REGION Network 8: START CYCLE LAMP
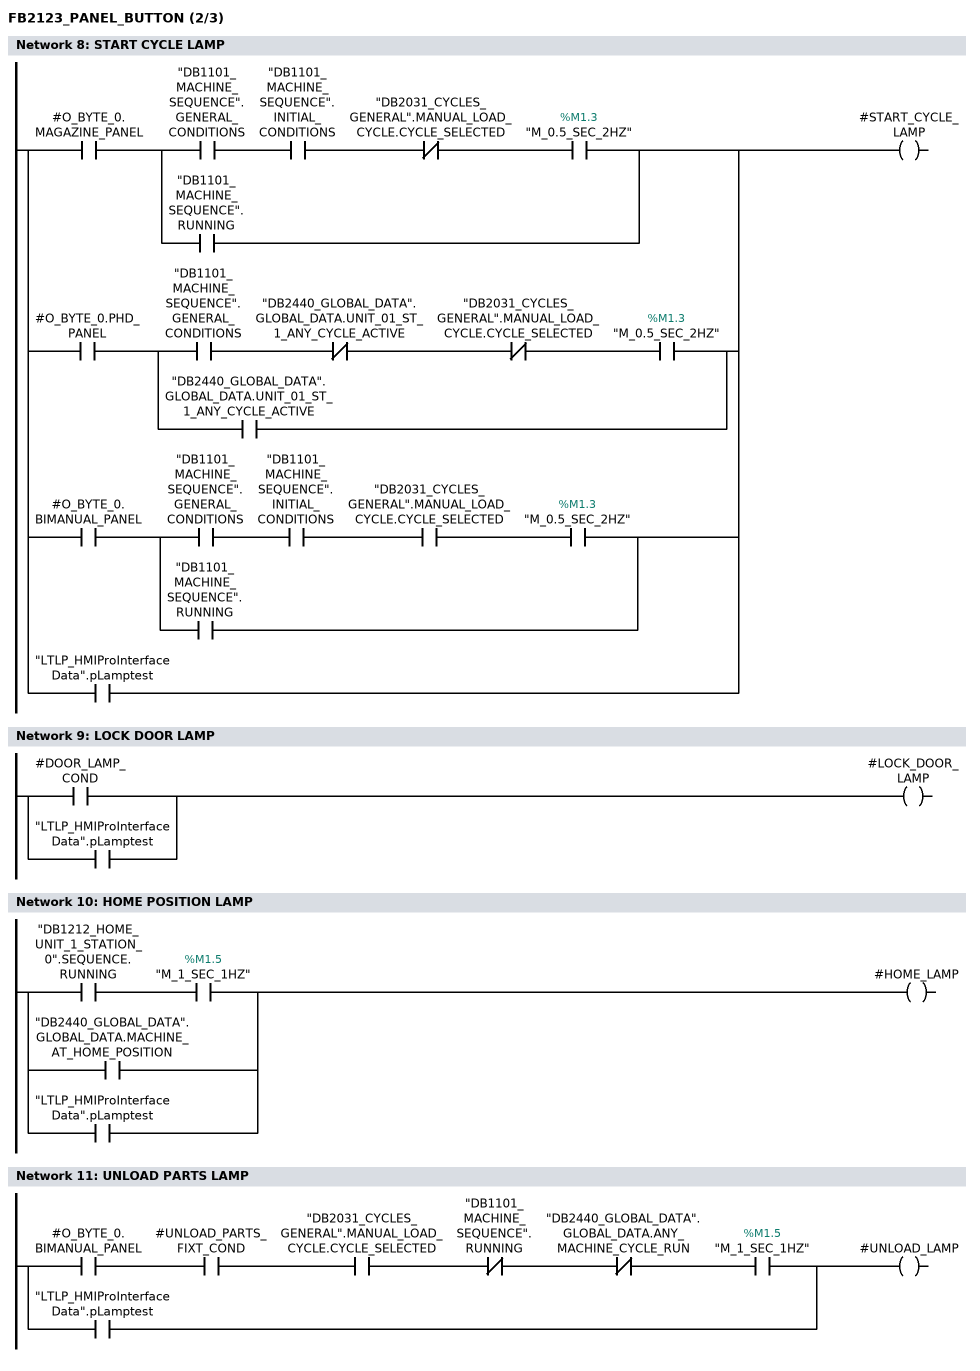
   RUNG wire#powerrail
      Contact( #O_BYTE_0.MAGAZINE_PANEL )
      wire#w1
      Contact( "DB1101_MACHINE_SEQUENCE".GENERAL_CONDITIONS )
      Contact( "DB1101_MACHINE_SEQUENCE".INITIAL_CONDITIONS )
      I_Contact( "DB2031_CYCLES_GENERAL".MANUAL_LOAD_CYCLE.CYCLE_SELECTED )
      Contact( "M_0.5_SEC_2HZ" )
      wire#w2
      Coil( #START_CYCLE_LAMP )
   END_RUNG
   RUNG wire#w1
      Contact( "DB1101_MACHINE_SEQUENCE".RUNNING )
   END_RUNG wire#w2
   RUNG wire#powerrail
      Contact( #O_BYTE_0.PHD_PANEL )
      wire#w3
      Contact( "DB1101_MACHINE_SEQUENCE".GENERAL_CONDITIONS )
      I_Contact( "DB2440_GLOBAL_DATA".GLOBAL_DATA.UNIT_01_ST_1_ANY_CYCLE_ACTIVE )
      I_Contact( "DB2031_CYCLES_GENERAL".MANUAL_LOAD_CYCLE.CYCLE_SELECTED )
      Contact( "M_0.5_SEC_2HZ" )
   END_RUNG wire#w2
   RUNG wire#w3
      Contact( "DB2440_GLOBAL_DATA".GLOBAL_DATA.UNIT_01_ST_1_ANY_CYCLE_ACTIVE )
   END_RUNG wire#w2
   RUNG wire#powerrail
      Contact( #O_BYTE_0.BIMANUAL_PANEL )
      wire#w4
      Contact( "DB1101_MACHINE_SEQUENCE".GENERAL_CONDITIONS )
      Contact( "DB1101_MACHINE_SEQUENCE".INITIAL_CONDITIONS )
      Contact( "DB2031_CYCLES_GENERAL".MANUAL_LOAD_CYCLE.CYCLE_SELECTED )
      Contact( "M_0.5_SEC_2HZ" )
   END_RUNG wire#w2
   RUNG wire#w4
      Contact( "DB1101_MACHINE_SEQUENCE".RUNNING )
   END_RUNG wire#w2
   RUNG wire#powerrail
      Contact( "LTLP_HMIProInterfaceData".pLamptest )
   END_RUNG wire#w2
   // the same network as SCL:
   #START_CYCLE_LAMP := (#O_BYTE_0.MAGAZINE_PANEL AND (("DB1101_MACHINE_SEQUENCE".GENERAL_CONDITIONS AND "DB1101_MACHINE_SEQUENCE".INITIAL_CONDITIONS AND NOT "DB2031_CYCLES_GENERAL".MANUAL_LOAD_CYCLE.CYCLE_SELECTED AND "M_0.5_SEC_2HZ") OR "DB1101_MACHINE_SEQUENCE".RUNNING)) OR (#O_BYTE_0.PHD_PANEL AND (("DB1101_MACHINE_SEQUENCE".GENERAL_CONDITIONS AND NOT "DB2440_GLOBAL_DATA".GLOBAL_DATA.UNIT_01_ST_1_ANY_CYCLE_ACTIVE AND NOT "DB2031_CYCLES_GENERAL".MANUAL_LOAD_CYCLE.CYCLE_SELECTED AND "M_0.5_SEC_2HZ") OR "DB2440_GLOBAL_DATA".GLOBAL_DATA.UNIT_01_ST_1_ANY_CYCLE_ACTIVE)) OR (#O_BYTE_0.BIMANUAL_PANEL AND (("DB1101_MACHINE_SEQUENCE".GENERAL_CONDITIONS AND "DB1101_MACHINE_SEQUENCE".INITIAL_CONDITIONS AND "DB2031_CYCLES_GENERAL".MANUAL_LOAD_CYCLE.CYCLE_SELECTED AND "M_0.5_SEC_2HZ") OR "DB1101_MACHINE_SEQUENCE".RUNNING)) OR "LTLP_HMIProInterfaceData".pLamptest;
END_REGION

REGION Network 9: LOCK DOOR LAMP
   RUNG wire#powerrail
      Contact( #DOOR_LAMP_COND )
      wire#w1
      Coil( #LOCK_DOOR_LAMP )
   END_RUNG
   RUNG wire#powerrail
      Contact( "LTLP_HMIProInterfaceData".pLamptest )
   END_RUNG wire#w1
   // the same network as SCL:
   #LOCK_DOOR_LAMP := #DOOR_LAMP_COND OR "LTLP_HMIProInterfaceData".pLamptest;
END_REGION

REGION Network 10: HOME POSITION LAMP
   RUNG wire#powerrail
      Contact( "DB1212_HOME_UNIT_1_STATION_0".SEQUENCE.RUNNING )
      Contact( "M_1_SEC_1HZ" )
      wire#w1
      Coil( #HOME_LAMP )
   END_RUNG
   RUNG wire#powerrail
      Contact( "DB2440_GLOBAL_DATA".GLOBAL_DATA.MACHINE_AT_HOME_POSITION )
   END_RUNG wire#w1
   RUNG wire#powerrail
      Contact( "LTLP_HMIProInterfaceData".pLamptest )
   END_RUNG wire#w1
   // the same network as SCL:
   #HOME_LAMP := ("DB1212_HOME_UNIT_1_STATION_0".SEQUENCE.RUNNING AND "M_1_SEC_1HZ") OR "DB2440_GLOBAL_DATA".GLOBAL_DATA.MACHINE_AT_HOME_POSITION OR "LTLP_HMIProInterfaceData".pLamptest;
END_REGION

REGION Network 11: UNLOAD PARTS LAMP
   RUNG wire#powerrail
      Contact( #O_BYTE_0.BIMANUAL_PANEL )
      Contact( #UNLOAD_PARTS_FIXT_COND )
      Contact( "DB2031_CYCLES_GENERAL".MANUAL_LOAD_CYCLE.CYCLE_SELECTED )
      I_Contact( "DB1101_MACHINE_SEQUENCE".RUNNING )
      I_Contact( "DB2440_GLOBAL_DATA".GLOBAL_DATA.ANY_MACHINE_CYCLE_RUN )
      Contact( "M_1_SEC_1HZ" )
      wire#w1
      Coil( #UNLOAD_LAMP )
   END_RUNG
   RUNG wire#powerrail
      Contact( "LTLP_HMIProInterfaceData".pLamptest )
   END_RUNG wire#w1
   // the same network as SCL:
   #UNLOAD_LAMP := (#O_BYTE_0.BIMANUAL_PANEL AND #UNLOAD_PARTS_FIXT_COND AND "DB2031_CYCLES_GENERAL".MANUAL_LOAD_CYCLE.CYCLE_SELECTED AND NOT "DB1101_MACHINE_SEQUENCE".RUNNING AND NOT "DB2440_GLOBAL_DATA".GLOBAL_DATA.ANY_MACHINE_CYCLE_RUN AND "M_1_SEC_1HZ") OR "LTLP_HMIProInterfaceData".pLamptest;
END_REGION

REGION Network 12: LOAD PARTS LAMP
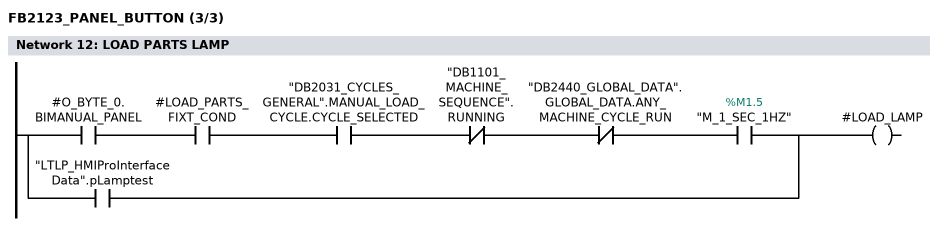
   RUNG wire#powerrail
      Contact( #O_BYTE_0.BIMANUAL_PANEL )
      Contact( #LOAD_PARTS_FIXT_COND )
      Contact( "DB2031_CYCLES_GENERAL".MANUAL_LOAD_CYCLE.CYCLE_SELECTED )
      I_Contact( "DB1101_MACHINE_SEQUENCE".RUNNING )
      I_Contact( "DB2440_GLOBAL_DATA".GLOBAL_DATA.ANY_MACHINE_CYCLE_RUN )
      Contact( "M_1_SEC_1HZ" )
      wire#w1
      Coil( #LOAD_LAMP )
   END_RUNG
   RUNG wire#powerrail
      Contact( "LTLP_HMIProInterfaceData".pLamptest )
   END_RUNG wire#w1
   // the same network as SCL:
   #LOAD_LAMP := (#O_BYTE_0.BIMANUAL_PANEL AND #LOAD_PARTS_FIXT_COND AND "DB2031_CYCLES_GENERAL".MANUAL_LOAD_CYCLE.CYCLE_SELECTED AND NOT "DB1101_MACHINE_SEQUENCE".RUNNING AND NOT "DB2440_GLOBAL_DATA".GLOBAL_DATA.ANY_MACHINE_CYCLE_RUN AND "M_1_SEC_1HZ") OR "LTLP_HMIProInterfaceData".pLamptest;
END_REGION
END_FUNCTION_BLOCK

FUNCTION "FC2101_LINE_CONTACTOR" : Void   // FC2101, LAD
{ S7_Optimized_Access := 'FALSE' }
AUTHOR : ETXETAR
VERSION : 1.0
// stored: AutoNumber false, IsIECCheckEnabled false, SetENOAutomatically false, UDAEnableTagReadback false
   VAR CONSTANT
      FC_NUMBER : DInt := 2101;   // FC NUMBER
   END_VAR
   VAR_TEMP   // added for the SCL form of the ladder/FBD networks
      _w1 : Bool;
      _w2 : Bool;
   END_VAR
BEGIN

REGION Network 1: OPTIONS OFF
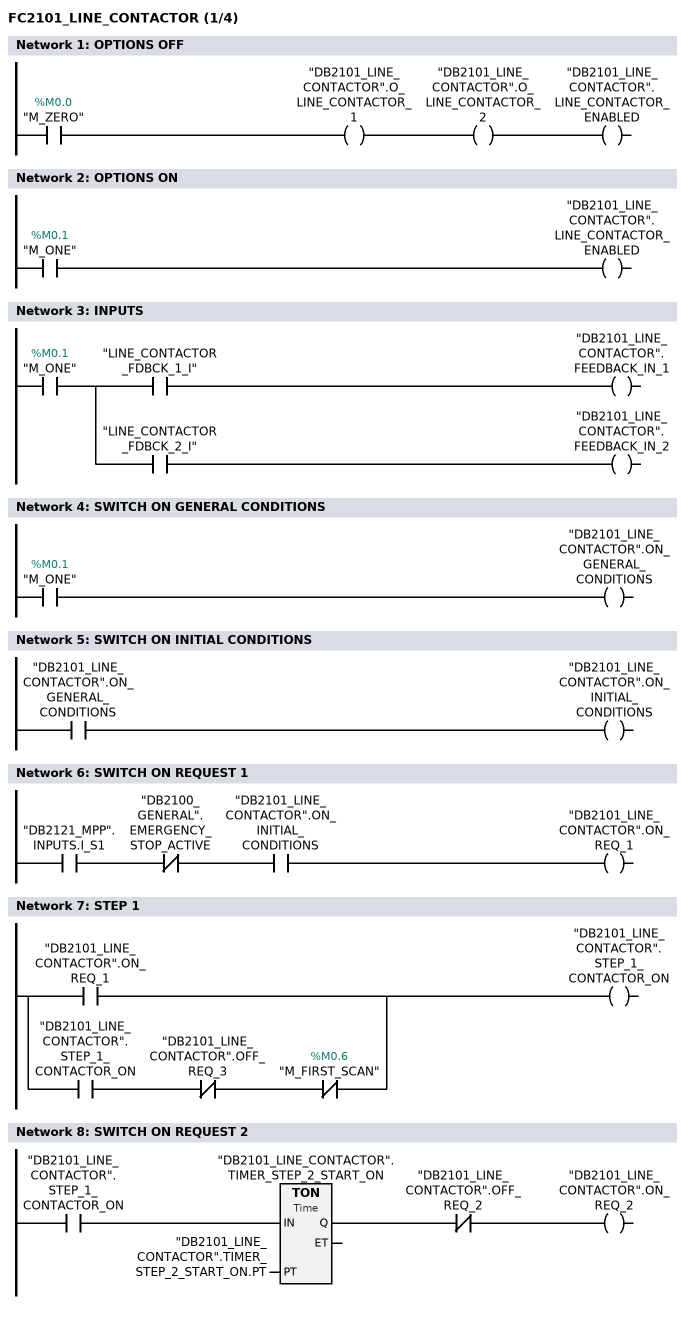
   RUNG wire#powerrail
      Contact( "M_ZERO" )
      Coil( "DB2101_LINE_CONTACTOR".O_LINE_CONTACTOR_1 )
      Coil( "DB2101_LINE_CONTACTOR".O_LINE_CONTACTOR_2 )
      Coil( "DB2101_LINE_CONTACTOR".LINE_CONTACTOR_ENABLED )
   END_RUNG
   // the same network as SCL:
   "DB2101_LINE_CONTACTOR".O_LINE_CONTACTOR_1 := "M_ZERO";
   "DB2101_LINE_CONTACTOR".O_LINE_CONTACTOR_2 := "M_ZERO";
   "DB2101_LINE_CONTACTOR".LINE_CONTACTOR_ENABLED := "M_ZERO";
END_REGION

REGION Network 2: OPTIONS ON
   RUNG wire#powerrail
      Contact( "M_ONE" )
      Coil( "DB2101_LINE_CONTACTOR".LINE_CONTACTOR_ENABLED )
   END_RUNG
   // the same network as SCL:
   "DB2101_LINE_CONTACTOR".LINE_CONTACTOR_ENABLED := "M_ONE";
END_REGION

REGION Network 3: INPUTS
   RUNG wire#powerrail
      Contact( "M_ONE" )
      wire#w1
      Contact( "LINE_CONTACTOR_FDBCK_1_I" )
      Coil( "DB2101_LINE_CONTACTOR".FEEDBACK_IN_1 )
   END_RUNG
   RUNG wire#w1
      Contact( "LINE_CONTACTOR_FDBCK_2_I" )
      Coil( "DB2101_LINE_CONTACTOR".FEEDBACK_IN_2 )
   END_RUNG
   // the same network as SCL:
   "DB2101_LINE_CONTACTOR".FEEDBACK_IN_1 := "M_ONE" AND "LINE_CONTACTOR_FDBCK_1_I";
   "DB2101_LINE_CONTACTOR".FEEDBACK_IN_2 := "M_ONE" AND "LINE_CONTACTOR_FDBCK_2_I";
END_REGION

REGION Network 4: SWITCH ON GENERAL CONDITIONS
   RUNG wire#powerrail
      Contact( "M_ONE" )
      Coil( "DB2101_LINE_CONTACTOR".ON_GENERAL_CONDITIONS )
   END_RUNG
   // the same network as SCL:
   "DB2101_LINE_CONTACTOR".ON_GENERAL_CONDITIONS := "M_ONE";
END_REGION

REGION Network 5: SWITCH ON INITIAL CONDITIONS
   RUNG wire#powerrail
      Contact( "DB2101_LINE_CONTACTOR".ON_GENERAL_CONDITIONS )
      Coil( "DB2101_LINE_CONTACTOR".ON_INITIAL_CONDITIONS )
   END_RUNG
   // the same network as SCL:
   "DB2101_LINE_CONTACTOR".ON_INITIAL_CONDITIONS := "DB2101_LINE_CONTACTOR".ON_GENERAL_CONDITIONS;
END_REGION

REGION Network 6: SWITCH ON REQUEST 1
   RUNG wire#powerrail
      Contact( "DB2121_MPP".INPUTS.I_S1 )
      I_Contact( "DB2100_GENERAL".EMERGENCY_STOP_ACTIVE )
      Contact( "DB2101_LINE_CONTACTOR".ON_INITIAL_CONDITIONS )
      Coil( "DB2101_LINE_CONTACTOR".ON_REQ_1 )
   END_RUNG
   // the same network as SCL:
   "DB2101_LINE_CONTACTOR".ON_REQ_1 := "DB2121_MPP".INPUTS.I_S1 AND NOT "DB2100_GENERAL".EMERGENCY_STOP_ACTIVE AND "DB2101_LINE_CONTACTOR".ON_INITIAL_CONDITIONS;
END_REGION

REGION Network 7: STEP 1
   RUNG wire#powerrail
      Contact( "DB2101_LINE_CONTACTOR".ON_REQ_1 )
      wire#w1
      Coil( "DB2101_LINE_CONTACTOR".STEP_1_CONTACTOR_ON )
   END_RUNG
   RUNG wire#powerrail
      Contact( "DB2101_LINE_CONTACTOR".STEP_1_CONTACTOR_ON )
      I_Contact( "DB2101_LINE_CONTACTOR".OFF_REQ_3 )
      I_Contact( "M_FIRST_SCAN" )
   END_RUNG wire#w1
   // the same network as SCL:
   "DB2101_LINE_CONTACTOR".STEP_1_CONTACTOR_ON := "DB2101_LINE_CONTACTOR".ON_REQ_1 OR ("DB2101_LINE_CONTACTOR".STEP_1_CONTACTOR_ON AND NOT "DB2101_LINE_CONTACTOR".OFF_REQ_3 AND NOT "M_FIRST_SCAN");
END_REGION

REGION Network 8: SWITCH ON REQUEST 2
   RUNG wire#powerrail
      Contact( "DB2101_LINE_CONTACTOR".STEP_1_CONTACTOR_ON )
      { S7_Templates := "time_type := Time" } "DB2101_LINE_CONTACTOR".TIMER_STEP_2_START_ON.TON(pt := "DB2101_LINE_CONTACTOR".TIMER_STEP_2_START_ON.PT, et =>)
      I_Contact( "DB2101_LINE_CONTACTOR".OFF_REQ_2 )
      Coil( "DB2101_LINE_CONTACTOR".ON_REQ_2 )
   END_RUNG
   // the same network as SCL:
   "DB2101_LINE_CONTACTOR".TIMER_STEP_2_START_ON.TON(IN := "DB2101_LINE_CONTACTOR".STEP_1_CONTACTOR_ON,
                           PT := "DB2101_LINE_CONTACTOR".TIMER_STEP_2_START_ON.PT);
   "DB2101_LINE_CONTACTOR".ON_REQ_2 := "DB2101_LINE_CONTACTOR".TIMER_STEP_2_START_ON.Q AND NOT "DB2101_LINE_CONTACTOR".OFF_REQ_2;
END_REGION

REGION Network 9: STEP 2
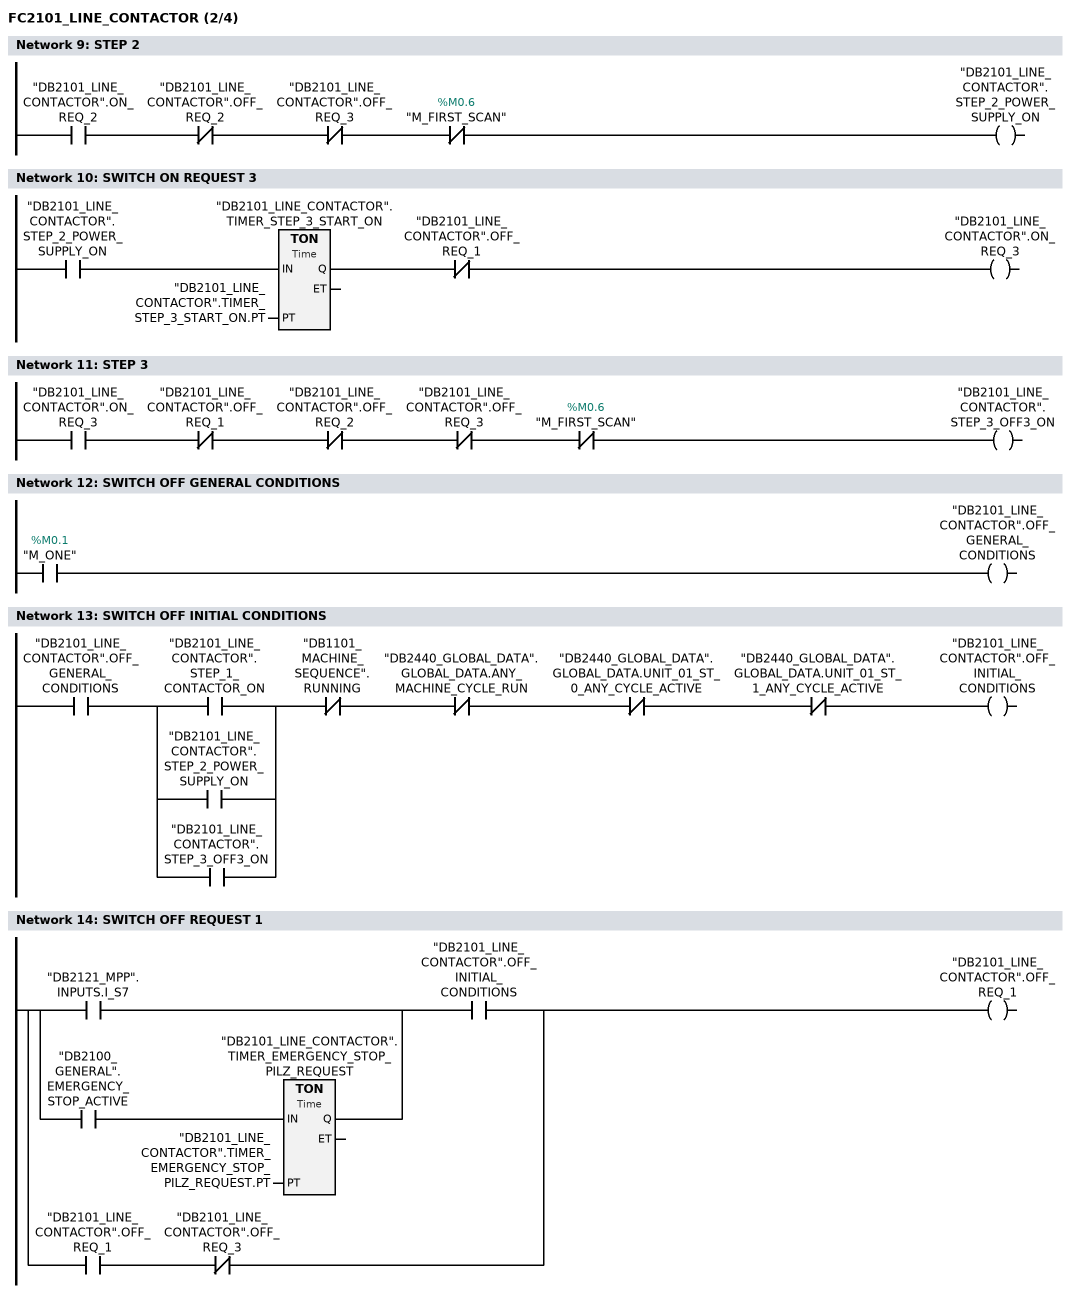
   RUNG wire#powerrail
      Contact( "DB2101_LINE_CONTACTOR".ON_REQ_2 )
      I_Contact( "DB2101_LINE_CONTACTOR".OFF_REQ_2 )
      I_Contact( "DB2101_LINE_CONTACTOR".OFF_REQ_3 )
      I_Contact( "M_FIRST_SCAN" )
      Coil( "DB2101_LINE_CONTACTOR".STEP_2_POWER_SUPPLY_ON )
   END_RUNG
   // the same network as SCL:
   "DB2101_LINE_CONTACTOR".STEP_2_POWER_SUPPLY_ON := "DB2101_LINE_CONTACTOR".ON_REQ_2 AND NOT "DB2101_LINE_CONTACTOR".OFF_REQ_2 AND NOT "DB2101_LINE_CONTACTOR".OFF_REQ_3 AND NOT "M_FIRST_SCAN";
END_REGION

REGION Network 10: SWITCH ON REQUEST 3
   RUNG wire#powerrail
      Contact( "DB2101_LINE_CONTACTOR".STEP_2_POWER_SUPPLY_ON )
      { S7_Templates := "time_type := Time" } "DB2101_LINE_CONTACTOR".TIMER_STEP_3_START_ON.TON(pt := "DB2101_LINE_CONTACTOR".TIMER_STEP_3_START_ON.PT, et =>)
      I_Contact( "DB2101_LINE_CONTACTOR".OFF_REQ_1 )
      Coil( "DB2101_LINE_CONTACTOR".ON_REQ_3 )
   END_RUNG
   // the same network as SCL:
   "DB2101_LINE_CONTACTOR".TIMER_STEP_3_START_ON.TON(IN := "DB2101_LINE_CONTACTOR".STEP_2_POWER_SUPPLY_ON,
                           PT := "DB2101_LINE_CONTACTOR".TIMER_STEP_3_START_ON.PT);
   "DB2101_LINE_CONTACTOR".ON_REQ_3 := "DB2101_LINE_CONTACTOR".TIMER_STEP_3_START_ON.Q AND NOT "DB2101_LINE_CONTACTOR".OFF_REQ_1;
END_REGION

REGION Network 11: STEP 3
   RUNG wire#powerrail
      Contact( "DB2101_LINE_CONTACTOR".ON_REQ_3 )
      I_Contact( "DB2101_LINE_CONTACTOR".OFF_REQ_1 )
      I_Contact( "DB2101_LINE_CONTACTOR".OFF_REQ_2 )
      I_Contact( "DB2101_LINE_CONTACTOR".OFF_REQ_3 )
      I_Contact( "M_FIRST_SCAN" )
      Coil( "DB2101_LINE_CONTACTOR".STEP_3_OFF3_ON )
   END_RUNG
   // the same network as SCL:
   "DB2101_LINE_CONTACTOR".STEP_3_OFF3_ON := "DB2101_LINE_CONTACTOR".ON_REQ_3 AND NOT "DB2101_LINE_CONTACTOR".OFF_REQ_1 AND NOT "DB2101_LINE_CONTACTOR".OFF_REQ_2 AND NOT "DB2101_LINE_CONTACTOR".OFF_REQ_3 AND NOT "M_FIRST_SCAN";
END_REGION

REGION Network 12: SWITCH OFF GENERAL CONDITIONS
   RUNG wire#powerrail
      Contact( "M_ONE" )
      Coil( "DB2101_LINE_CONTACTOR".OFF_GENERAL_CONDITIONS )
   END_RUNG
   // the same network as SCL:
   "DB2101_LINE_CONTACTOR".OFF_GENERAL_CONDITIONS := "M_ONE";
END_REGION

REGION Network 13: SWITCH OFF INITIAL CONDITIONS
   RUNG wire#powerrail
      Contact( "DB2101_LINE_CONTACTOR".OFF_GENERAL_CONDITIONS )
      wire#w1
      Contact( "DB2101_LINE_CONTACTOR".STEP_1_CONTACTOR_ON )
      wire#w2
      I_Contact( "DB1101_MACHINE_SEQUENCE".RUNNING )
      I_Contact( "DB2440_GLOBAL_DATA".GLOBAL_DATA.ANY_MACHINE_CYCLE_RUN )
      I_Contact( "DB2440_GLOBAL_DATA".GLOBAL_DATA.UNIT_01_ST_0_ANY_CYCLE_ACTIVE )
      I_Contact( "DB2440_GLOBAL_DATA".GLOBAL_DATA.UNIT_01_ST_1_ANY_CYCLE_ACTIVE )
      Coil( "DB2101_LINE_CONTACTOR".OFF_INITIAL_CONDITIONS )
   END_RUNG
   RUNG wire#w1
      Contact( "DB2101_LINE_CONTACTOR".STEP_2_POWER_SUPPLY_ON )
   END_RUNG wire#w2
   RUNG wire#w1
      Contact( "DB2101_LINE_CONTACTOR".STEP_3_OFF3_ON )
   END_RUNG wire#w2
   // the same network as SCL:
   "DB2101_LINE_CONTACTOR".OFF_INITIAL_CONDITIONS := "DB2101_LINE_CONTACTOR".OFF_GENERAL_CONDITIONS AND ("DB2101_LINE_CONTACTOR".STEP_1_CONTACTOR_ON OR "DB2101_LINE_CONTACTOR".STEP_2_POWER_SUPPLY_ON OR "DB2101_LINE_CONTACTOR".STEP_3_OFF3_ON) AND NOT "DB1101_MACHINE_SEQUENCE".RUNNING AND NOT "DB2440_GLOBAL_DATA".GLOBAL_DATA.ANY_MACHINE_CYCLE_RUN AND NOT "DB2440_GLOBAL_DATA".GLOBAL_DATA.UNIT_01_ST_0_ANY_CYCLE_ACTIVE AND NOT "DB2440_GLOBAL_DATA".GLOBAL_DATA.UNIT_01_ST_1_ANY_CYCLE_ACTIVE;
END_REGION

REGION Network 14: SWITCH OFF REQUEST 1
   RUNG wire#powerrail
      Contact( "DB2121_MPP".INPUTS.I_S7 )
      wire#w1
      Contact( "DB2101_LINE_CONTACTOR".OFF_INITIAL_CONDITIONS )
      wire#w2
      Coil( "DB2101_LINE_CONTACTOR".OFF_REQ_1 )
   END_RUNG
   RUNG wire#powerrail
      Contact( "DB2100_GENERAL".EMERGENCY_STOP_ACTIVE )
      { S7_Templates := "time_type := Time" } "DB2101_LINE_CONTACTOR".TIMER_EMERGENCY_STOP_PILZ_REQUEST.TON(pt := "DB2101_LINE_CONTACTOR".TIMER_EMERGENCY_STOP_PILZ_REQUEST.PT, et =>)
   END_RUNG wire#w1
   RUNG wire#powerrail
      Contact( "DB2101_LINE_CONTACTOR".OFF_REQ_1 )
      I_Contact( "DB2101_LINE_CONTACTOR".OFF_REQ_3 )
   END_RUNG wire#w2
   // the same network as SCL:
   "DB2101_LINE_CONTACTOR".TIMER_EMERGENCY_STOP_PILZ_REQUEST.TON(IN := "DB2100_GENERAL".EMERGENCY_STOP_ACTIVE,
                           PT := "DB2101_LINE_CONTACTOR".TIMER_EMERGENCY_STOP_PILZ_REQUEST.PT);
   "DB2101_LINE_CONTACTOR".OFF_REQ_1 := (("DB2121_MPP".INPUTS.I_S7 OR "DB2101_LINE_CONTACTOR".TIMER_EMERGENCY_STOP_PILZ_REQUEST.Q) AND "DB2101_LINE_CONTACTOR".OFF_INITIAL_CONDITIONS) OR ("DB2101_LINE_CONTACTOR".OFF_REQ_1 AND NOT "DB2101_LINE_CONTACTOR".OFF_REQ_3);
END_REGION

REGION Network 15: SWITCH OFF REQUEST 2
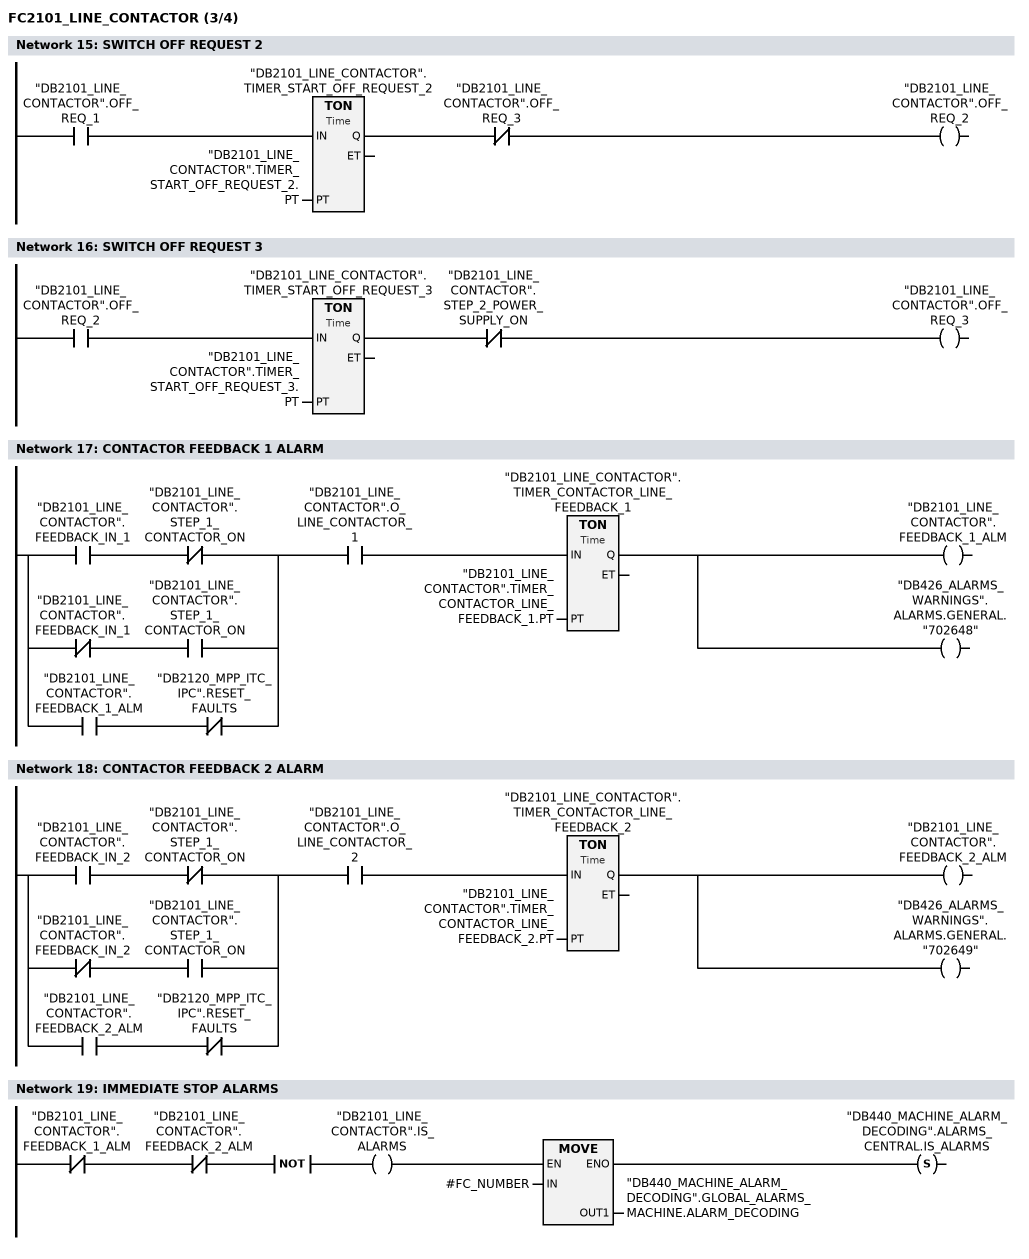
   RUNG wire#powerrail
      Contact( "DB2101_LINE_CONTACTOR".OFF_REQ_1 )
      { S7_Templates := "time_type := Time" } "DB2101_LINE_CONTACTOR".TIMER_START_OFF_REQUEST_2.TON(pt := "DB2101_LINE_CONTACTOR".TIMER_START_OFF_REQUEST_2.PT, et =>)
      I_Contact( "DB2101_LINE_CONTACTOR".OFF_REQ_3 )
      Coil( "DB2101_LINE_CONTACTOR".OFF_REQ_2 )
   END_RUNG
   // the same network as SCL:
   "DB2101_LINE_CONTACTOR".TIMER_START_OFF_REQUEST_2.TON(IN := "DB2101_LINE_CONTACTOR".OFF_REQ_1,
                           PT := "DB2101_LINE_CONTACTOR".TIMER_START_OFF_REQUEST_2.PT);
   "DB2101_LINE_CONTACTOR".OFF_REQ_2 := "DB2101_LINE_CONTACTOR".TIMER_START_OFF_REQUEST_2.Q AND NOT "DB2101_LINE_CONTACTOR".OFF_REQ_3;
END_REGION

REGION Network 16: SWITCH OFF REQUEST 3
   RUNG wire#powerrail
      Contact( "DB2101_LINE_CONTACTOR".OFF_REQ_2 )
      { S7_Templates := "time_type := Time" } "DB2101_LINE_CONTACTOR".TIMER_START_OFF_REQUEST_3.TON(pt := "DB2101_LINE_CONTACTOR".TIMER_START_OFF_REQUEST_3.PT, et =>)
      I_Contact( "DB2101_LINE_CONTACTOR".STEP_2_POWER_SUPPLY_ON )
      Coil( "DB2101_LINE_CONTACTOR".OFF_REQ_3 )
   END_RUNG
   // the same network as SCL:
   "DB2101_LINE_CONTACTOR".TIMER_START_OFF_REQUEST_3.TON(IN := "DB2101_LINE_CONTACTOR".OFF_REQ_2,
                           PT := "DB2101_LINE_CONTACTOR".TIMER_START_OFF_REQUEST_3.PT);
   "DB2101_LINE_CONTACTOR".OFF_REQ_3 := "DB2101_LINE_CONTACTOR".TIMER_START_OFF_REQUEST_3.Q AND NOT "DB2101_LINE_CONTACTOR".STEP_2_POWER_SUPPLY_ON;
END_REGION

REGION Network 17: CONTACTOR FEEDBACK 1 ALARM
   RUNG wire#powerrail
      Contact( "DB2101_LINE_CONTACTOR".FEEDBACK_IN_1 )
      I_Contact( "DB2101_LINE_CONTACTOR".STEP_1_CONTACTOR_ON )
      wire#w1
      Contact( "DB2101_LINE_CONTACTOR".O_LINE_CONTACTOR_1 )
      { S7_Templates := "time_type := Time" } "DB2101_LINE_CONTACTOR".TIMER_CONTACTOR_LINE_FEEDBACK_1.TON(pt := "DB2101_LINE_CONTACTOR".TIMER_CONTACTOR_LINE_FEEDBACK_1.PT, et =>)
      wire#w2
      Coil( "DB2101_LINE_CONTACTOR".FEEDBACK_1_ALM )
   END_RUNG
   RUNG wire#powerrail
      I_Contact( "DB2101_LINE_CONTACTOR".FEEDBACK_IN_1 )
      Contact( "DB2101_LINE_CONTACTOR".STEP_1_CONTACTOR_ON )
   END_RUNG wire#w1
   RUNG wire#powerrail
      Contact( "DB2101_LINE_CONTACTOR".FEEDBACK_1_ALM )
      I_Contact( "DB2120_MPP_ITC_IPC".RESET_FAULTS )
   END_RUNG wire#w1
   RUNG wire#w2
      Coil( "DB426_ALARMS_WARNINGS".ALARMS.GENERAL."702648" )
   END_RUNG
   // the same network as SCL:
   "DB2101_LINE_CONTACTOR".TIMER_CONTACTOR_LINE_FEEDBACK_1.TON(IN := (("DB2101_LINE_CONTACTOR".FEEDBACK_IN_1 AND NOT "DB2101_LINE_CONTACTOR".STEP_1_CONTACTOR_ON) OR (NOT "DB2101_LINE_CONTACTOR".FEEDBACK_IN_1 AND "DB2101_LINE_CONTACTOR".STEP_1_CONTACTOR_ON) OR ("DB2101_LINE_CONTACTOR".FEEDBACK_1_ALM AND NOT "DB2120_MPP_ITC_IPC".RESET_FAULTS)) AND "DB2101_LINE_CONTACTOR".O_LINE_CONTACTOR_1,
                           PT := "DB2101_LINE_CONTACTOR".TIMER_CONTACTOR_LINE_FEEDBACK_1.PT);
   "DB2101_LINE_CONTACTOR".FEEDBACK_1_ALM := "DB2101_LINE_CONTACTOR".TIMER_CONTACTOR_LINE_FEEDBACK_1.Q;
   "DB426_ALARMS_WARNINGS".ALARMS.GENERAL."702648" := "DB2101_LINE_CONTACTOR".TIMER_CONTACTOR_LINE_FEEDBACK_1.Q;
END_REGION

REGION Network 18: CONTACTOR FEEDBACK 2 ALARM
   RUNG wire#powerrail
      Contact( "DB2101_LINE_CONTACTOR".FEEDBACK_IN_2 )
      I_Contact( "DB2101_LINE_CONTACTOR".STEP_1_CONTACTOR_ON )
      wire#w1
      Contact( "DB2101_LINE_CONTACTOR".O_LINE_CONTACTOR_2 )
      { S7_Templates := "time_type := Time" } "DB2101_LINE_CONTACTOR".TIMER_CONTACTOR_LINE_FEEDBACK_2.TON(pt := "DB2101_LINE_CONTACTOR".TIMER_CONTACTOR_LINE_FEEDBACK_2.PT, et =>)
      wire#w2
      Coil( "DB2101_LINE_CONTACTOR".FEEDBACK_2_ALM )
   END_RUNG
   RUNG wire#powerrail
      I_Contact( "DB2101_LINE_CONTACTOR".FEEDBACK_IN_2 )
      Contact( "DB2101_LINE_CONTACTOR".STEP_1_CONTACTOR_ON )
   END_RUNG wire#w1
   RUNG wire#powerrail
      Contact( "DB2101_LINE_CONTACTOR".FEEDBACK_2_ALM )
      I_Contact( "DB2120_MPP_ITC_IPC".RESET_FAULTS )
   END_RUNG wire#w1
   RUNG wire#w2
      Coil( "DB426_ALARMS_WARNINGS".ALARMS.GENERAL."702649" )
   END_RUNG
   // the same network as SCL:
   "DB2101_LINE_CONTACTOR".TIMER_CONTACTOR_LINE_FEEDBACK_2.TON(IN := (("DB2101_LINE_CONTACTOR".FEEDBACK_IN_2 AND NOT "DB2101_LINE_CONTACTOR".STEP_1_CONTACTOR_ON) OR (NOT "DB2101_LINE_CONTACTOR".FEEDBACK_IN_2 AND "DB2101_LINE_CONTACTOR".STEP_1_CONTACTOR_ON) OR ("DB2101_LINE_CONTACTOR".FEEDBACK_2_ALM AND NOT "DB2120_MPP_ITC_IPC".RESET_FAULTS)) AND "DB2101_LINE_CONTACTOR".O_LINE_CONTACTOR_2,
                           PT := "DB2101_LINE_CONTACTOR".TIMER_CONTACTOR_LINE_FEEDBACK_2.PT);
   "DB2101_LINE_CONTACTOR".FEEDBACK_2_ALM := "DB2101_LINE_CONTACTOR".TIMER_CONTACTOR_LINE_FEEDBACK_2.Q;
   "DB426_ALARMS_WARNINGS".ALARMS.GENERAL."702649" := "DB2101_LINE_CONTACTOR".TIMER_CONTACTOR_LINE_FEEDBACK_2.Q;
END_REGION

REGION Network 19: IMMEDIATE STOP ALARMS
   RUNG wire#powerrail
      I_Contact( "DB2101_LINE_CONTACTOR".FEEDBACK_1_ALM )
      I_Contact( "DB2101_LINE_CONTACTOR".FEEDBACK_2_ALM )
      Not()
      Coil( "DB2101_LINE_CONTACTOR".IS_ALARMS )
      Move(in := #FC_NUMBER, out1 => "DB440_MACHINE_ALARM_DECODING".GLOBAL_ALARMS_MACHINE.ALARM_DECODING)
      S_Coil( "DB440_MACHINE_ALARM_DECODING".ALARMS_CENTRAL.IS_ALARMS )
   END_RUNG
   // the same network as SCL:
   "DB2101_LINE_CONTACTOR".IS_ALARMS := NOT (NOT "DB2101_LINE_CONTACTOR".FEEDBACK_1_ALM AND NOT "DB2101_LINE_CONTACTOR".FEEDBACK_2_ALM);
   IF "DB2101_LINE_CONTACTOR".IS_ALARMS THEN
       "DB440_MACHINE_ALARM_DECODING".GLOBAL_ALARMS_MACHINE.ALARM_DECODING := #FC_NUMBER;
       "DB440_MACHINE_ALARM_DECODING".ALARMS_CENTRAL.IS_ALARMS := TRUE;
   END_IF;
END_REGION

REGION Network 20: PROGRESSIVE STOP POWDER ALARMS
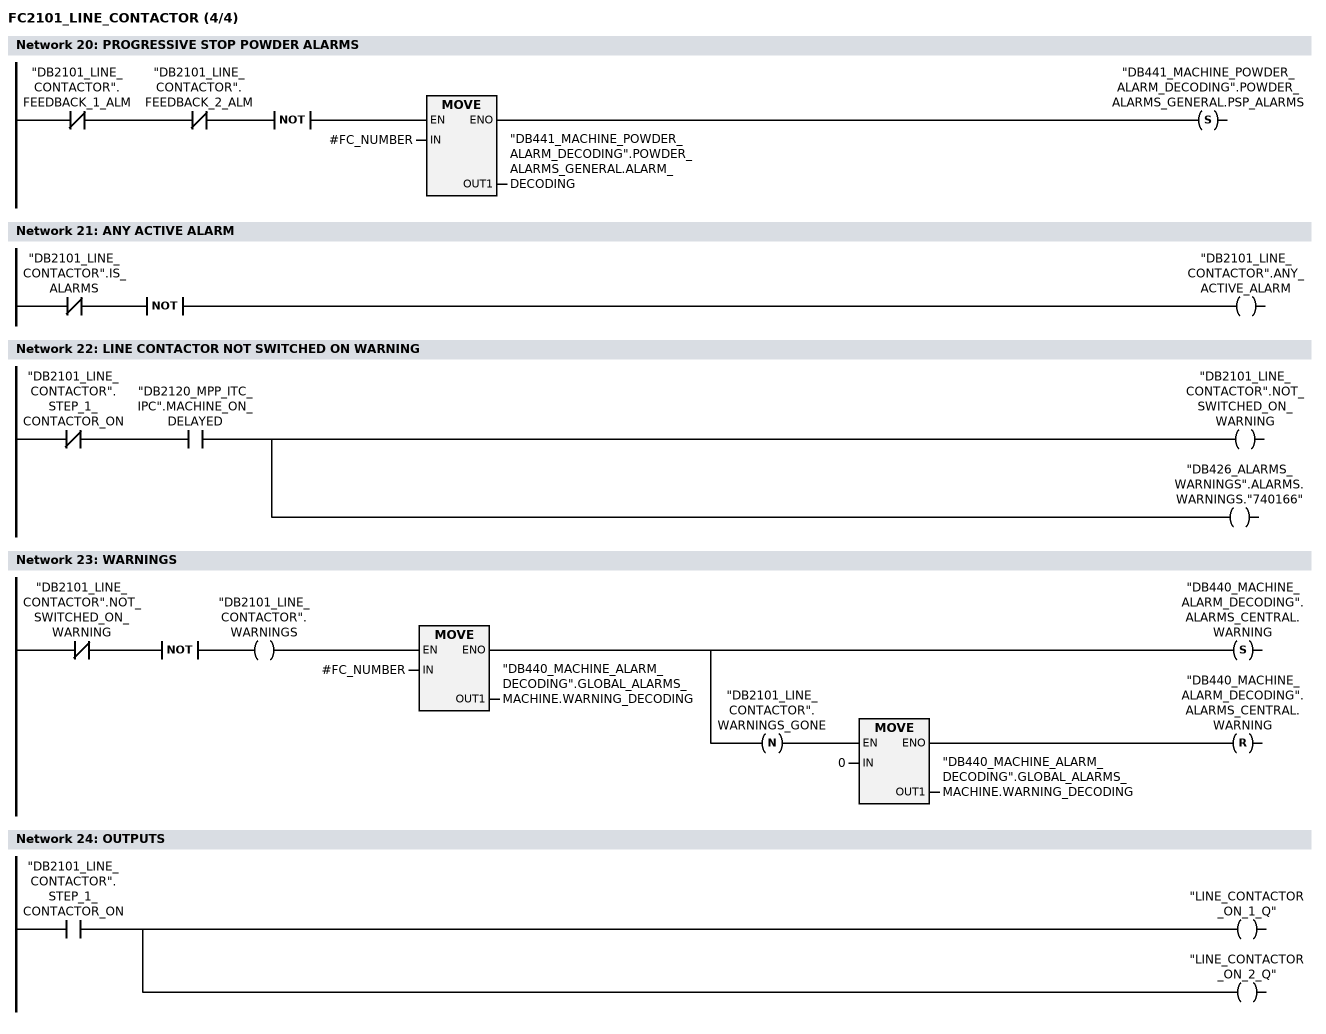
   RUNG wire#powerrail
      I_Contact( "DB2101_LINE_CONTACTOR".FEEDBACK_1_ALM )
      I_Contact( "DB2101_LINE_CONTACTOR".FEEDBACK_2_ALM )
      Not()
      Move(in := #FC_NUMBER, out1 => "DB441_MACHINE_POWDER_ALARM_DECODING".POWDER_ALARMS_GENERAL.ALARM_DECODING)
      S_Coil( "DB441_MACHINE_POWDER_ALARM_DECODING".POWDER_ALARMS_GENERAL.PSP_ALARMS )
   END_RUNG
   // the same network as SCL:
   IF NOT (NOT "DB2101_LINE_CONTACTOR".FEEDBACK_1_ALM AND NOT "DB2101_LINE_CONTACTOR".FEEDBACK_2_ALM) THEN
       "DB441_MACHINE_POWDER_ALARM_DECODING".POWDER_ALARMS_GENERAL.ALARM_DECODING := #FC_NUMBER;
       "DB441_MACHINE_POWDER_ALARM_DECODING".POWDER_ALARMS_GENERAL.PSP_ALARMS := TRUE;
   END_IF;
END_REGION

REGION Network 21: ANY ACTIVE ALARM
   RUNG wire#powerrail
      I_Contact( "DB2101_LINE_CONTACTOR".IS_ALARMS )
      Not()
      Coil( "DB2101_LINE_CONTACTOR".ANY_ACTIVE_ALARM )
   END_RUNG
   // the same network as SCL:
   "DB2101_LINE_CONTACTOR".ANY_ACTIVE_ALARM := NOT (NOT "DB2101_LINE_CONTACTOR".IS_ALARMS);
END_REGION

REGION Network 22: LINE CONTACTOR NOT SWITCHED ON WARNING
   RUNG wire#powerrail
      I_Contact( "DB2101_LINE_CONTACTOR".STEP_1_CONTACTOR_ON )
      Contact( "DB2120_MPP_ITC_IPC".MACHINE_ON_DELAYED )
      wire#w1
      Coil( "DB2101_LINE_CONTACTOR".NOT_SWITCHED_ON_WARNING )
   END_RUNG
   RUNG wire#w1
      Coil( "DB426_ALARMS_WARNINGS".ALARMS.WARNINGS."740166" )
   END_RUNG
   // the same network as SCL:
   "DB2101_LINE_CONTACTOR".NOT_SWITCHED_ON_WARNING := NOT "DB2101_LINE_CONTACTOR".STEP_1_CONTACTOR_ON AND "DB2120_MPP_ITC_IPC".MACHINE_ON_DELAYED;
   "DB426_ALARMS_WARNINGS".ALARMS.WARNINGS."740166" := "DB2101_LINE_CONTACTOR".NOT_SWITCHED_ON_WARNING;
END_REGION

REGION Network 23: WARNINGS
   RUNG wire#powerrail
      I_Contact( "DB2101_LINE_CONTACTOR".NOT_SWITCHED_ON_WARNING )
      Not()
      Coil( "DB2101_LINE_CONTACTOR".WARNINGS )
      Move(in := #FC_NUMBER, out1 => "DB440_MACHINE_ALARM_DECODING".GLOBAL_ALARMS_MACHINE.WARNING_DECODING)
      wire#w1
      S_Coil( "DB440_MACHINE_ALARM_DECODING".ALARMS_CENTRAL.WARNING )
   END_RUNG
   RUNG wire#w1
      N_Trig( "DB2101_LINE_CONTACTOR".WARNINGS_GONE )
      Move(in := 0, out1 => "DB440_MACHINE_ALARM_DECODING".GLOBAL_ALARMS_MACHINE.WARNING_DECODING)
      R_Coil( "DB440_MACHINE_ALARM_DECODING".ALARMS_CENTRAL.WARNING )
   END_RUNG
   // the same network as SCL:
   "DB2101_LINE_CONTACTOR".WARNINGS := NOT (NOT "DB2101_LINE_CONTACTOR".NOT_SWITCHED_ON_WARNING);
   #_w1 := NOT (NOT "DB2101_LINE_CONTACTOR".NOT_SWITCHED_ON_WARNING);
   IF #_w1 THEN
       "DB440_MACHINE_ALARM_DECODING".GLOBAL_ALARMS_MACHINE.WARNING_DECODING := #FC_NUMBER;
       "DB440_MACHINE_ALARM_DECODING".ALARMS_CENTRAL.WARNING := TRUE;
   END_IF;
   #_w2 := NOT #_w1 AND "DB2101_LINE_CONTACTOR".WARNINGS_GONE;   // falling edge
   "DB2101_LINE_CONTACTOR".WARNINGS_GONE := #_w1;
   IF #_w2 THEN
       "DB440_MACHINE_ALARM_DECODING".GLOBAL_ALARMS_MACHINE.WARNING_DECODING := 0;
       "DB440_MACHINE_ALARM_DECODING".ALARMS_CENTRAL.WARNING := FALSE;
   END_IF;
END_REGION

REGION Network 24: OUTPUTS
   RUNG wire#powerrail
      Contact( "DB2101_LINE_CONTACTOR".STEP_1_CONTACTOR_ON )
      wire#w1
      Coil( "LINE_CONTACTOR_ON_1_Q" )
   END_RUNG
   RUNG wire#w1
      Coil( "LINE_CONTACTOR_ON_2_Q" )
   END_RUNG
   // the same network as SCL:
   "LINE_CONTACTOR_ON_1_Q" := "DB2101_LINE_CONTACTOR".STEP_1_CONTACTOR_ON;
   "LINE_CONTACTOR_ON_2_Q" := "DB2101_LINE_CONTACTOR".STEP_1_CONTACTOR_ON;
END_REGION
END_FUNCTION

FUNCTION "FC2102_INFEED_MODULE" : Void   // FC2102, LAD
{ S7_Optimized_Access := 'FALSE' }
AUTHOR : ETXETAR
VERSION : 1.0
// stored: AutoNumber false, IsIECCheckEnabled false, SetENOAutomatically false, UDAEnableTagReadback false
   VAR_TEMP
      O_BYTE_0 : Struct   // OPTIONS BYTE 0
         POWER_SUPPLY_2 : Bool;   // POWER SUPPLY 2 OPTION
      END_STRUCT;
   END_VAR
   VAR CONSTANT
      FC_NUMBER : DInt := 2102;
   END_VAR
   VAR_TEMP   // added for the SCL form of the ladder/FBD networks
      _w1 : Bool;
   END_VAR
BEGIN

REGION Network 1: OPTIONS OFF
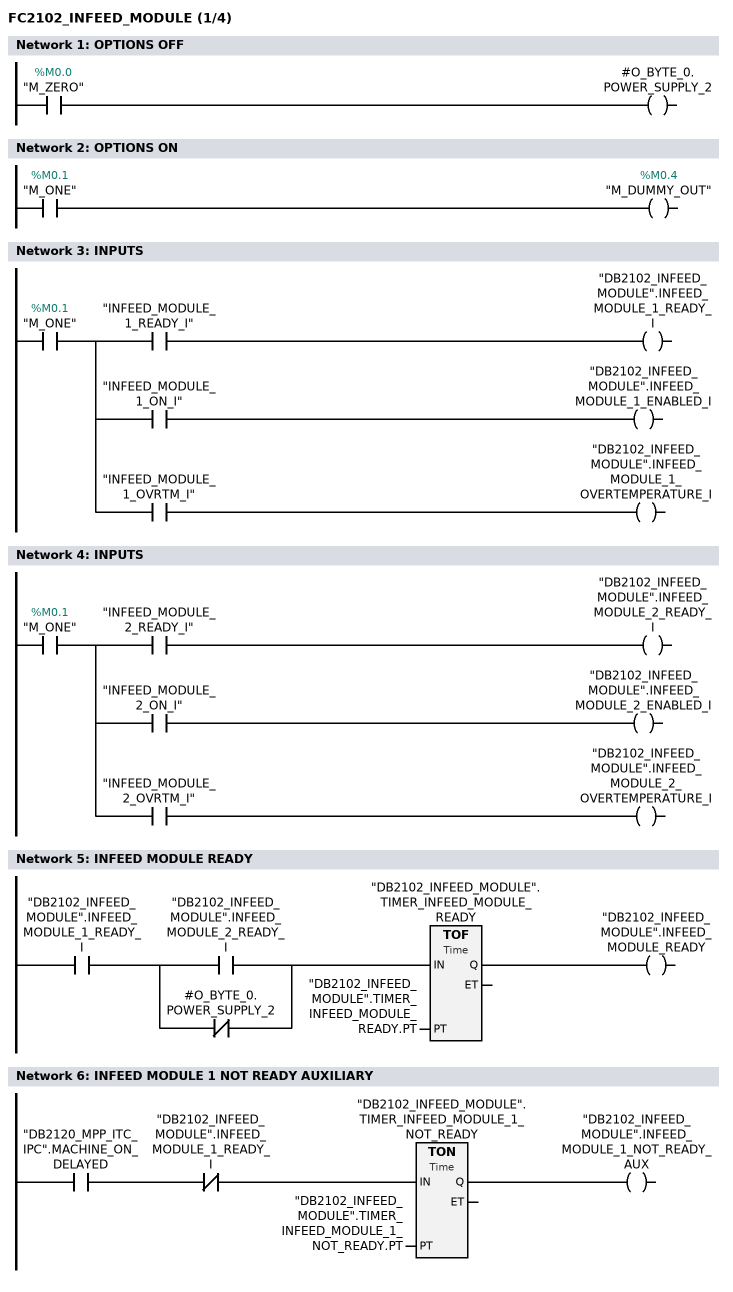
   RUNG wire#powerrail
      Contact( "M_ZERO" )
      Coil( #O_BYTE_0.POWER_SUPPLY_2 )
   END_RUNG
   // the same network as SCL:
   #O_BYTE_0.POWER_SUPPLY_2 := "M_ZERO";
END_REGION

REGION Network 2: OPTIONS ON
   RUNG wire#powerrail
      Contact( "M_ONE" )
      Coil( "M_DUMMY_OUT" )
   END_RUNG
   // the same network as SCL:
   "M_DUMMY_OUT" := "M_ONE";
END_REGION

REGION Network 3: INPUTS
   RUNG wire#powerrail
      Contact( "M_ONE" )
      wire#w1
      Contact( "INFEED_MODULE_1_READY_I" )
      Coil( "DB2102_INFEED_MODULE".INFEED_MODULE_1_READY_I )
   END_RUNG
   RUNG wire#w1
      Contact( "INFEED_MODULE_1_ON_I" )
      Coil( "DB2102_INFEED_MODULE".INFEED_MODULE_1_ENABLED_I )
   END_RUNG
   RUNG wire#w1
      Contact( "INFEED_MODULE_1_OVRTM_I" )
      Coil( "DB2102_INFEED_MODULE".INFEED_MODULE_1_OVERTEMPERATURE_I )
   END_RUNG
   // the same network as SCL:
   "DB2102_INFEED_MODULE".INFEED_MODULE_1_READY_I := "M_ONE" AND "INFEED_MODULE_1_READY_I";
   "DB2102_INFEED_MODULE".INFEED_MODULE_1_ENABLED_I := "M_ONE" AND "INFEED_MODULE_1_ON_I";
   "DB2102_INFEED_MODULE".INFEED_MODULE_1_OVERTEMPERATURE_I := "M_ONE" AND "INFEED_MODULE_1_OVRTM_I";
END_REGION

REGION Network 4: INPUTS
   RUNG wire#powerrail
      Contact( "M_ONE" )
      wire#w1
      Contact( "INFEED_MODULE_2_READY_I" )
      Coil( "DB2102_INFEED_MODULE".INFEED_MODULE_2_READY_I )
   END_RUNG
   RUNG wire#w1
      Contact( "INFEED_MODULE_2_ON_I" )
      Coil( "DB2102_INFEED_MODULE".INFEED_MODULE_2_ENABLED_I )
   END_RUNG
   RUNG wire#w1
      Contact( "INFEED_MODULE_2_OVRTM_I" )
      Coil( "DB2102_INFEED_MODULE".INFEED_MODULE_2_OVERTEMPERATURE_I )
   END_RUNG
   // the same network as SCL:
   "DB2102_INFEED_MODULE".INFEED_MODULE_2_READY_I := "M_ONE" AND "INFEED_MODULE_2_READY_I";
   "DB2102_INFEED_MODULE".INFEED_MODULE_2_ENABLED_I := "M_ONE" AND "INFEED_MODULE_2_ON_I";
   "DB2102_INFEED_MODULE".INFEED_MODULE_2_OVERTEMPERATURE_I := "M_ONE" AND "INFEED_MODULE_2_OVRTM_I";
END_REGION

REGION Network 5: INFEED MODULE READY
   RUNG wire#powerrail
      Contact( "DB2102_INFEED_MODULE".INFEED_MODULE_1_READY_I )
      wire#w1
      Contact( "DB2102_INFEED_MODULE".INFEED_MODULE_2_READY_I )
      wire#w2
      { S7_Templates := "time_type := Time" } "DB2102_INFEED_MODULE".TIMER_INFEED_MODULE_READY.TOF(pt := "DB2102_INFEED_MODULE".TIMER_INFEED_MODULE_READY.PT, et =>)
      Coil( "DB2102_INFEED_MODULE".INFEED_MODULE_READY )
   END_RUNG
   RUNG wire#w1
      I_Contact( #O_BYTE_0.POWER_SUPPLY_2 )
   END_RUNG wire#w2
   // the same network as SCL:
   "DB2102_INFEED_MODULE".TIMER_INFEED_MODULE_READY.TOF(IN := "DB2102_INFEED_MODULE".INFEED_MODULE_1_READY_I AND ("DB2102_INFEED_MODULE".INFEED_MODULE_2_READY_I OR NOT #O_BYTE_0.POWER_SUPPLY_2),
                           PT := "DB2102_INFEED_MODULE".TIMER_INFEED_MODULE_READY.PT);
   "DB2102_INFEED_MODULE".INFEED_MODULE_READY := "DB2102_INFEED_MODULE".TIMER_INFEED_MODULE_READY.Q;
END_REGION

REGION Network 6: INFEED MODULE 1 NOT READY AUXILIARY
   RUNG wire#powerrail
      Contact( "DB2120_MPP_ITC_IPC".MACHINE_ON_DELAYED )
      I_Contact( "DB2102_INFEED_MODULE".INFEED_MODULE_1_READY_I )
      { S7_Templates := "time_type := Time" } "DB2102_INFEED_MODULE".TIMER_INFEED_MODULE_1_NOT_READY.TON(pt := "DB2102_INFEED_MODULE".TIMER_INFEED_MODULE_1_NOT_READY.PT, et =>)
      Coil( "DB2102_INFEED_MODULE".INFEED_MODULE_1_NOT_READY_AUX )
   END_RUNG
   // the same network as SCL:
   "DB2102_INFEED_MODULE".TIMER_INFEED_MODULE_1_NOT_READY.TON(IN := "DB2120_MPP_ITC_IPC".MACHINE_ON_DELAYED AND NOT "DB2102_INFEED_MODULE".INFEED_MODULE_1_READY_I,
                           PT := "DB2102_INFEED_MODULE".TIMER_INFEED_MODULE_1_NOT_READY.PT);
   "DB2102_INFEED_MODULE".INFEED_MODULE_1_NOT_READY_AUX := "DB2102_INFEED_MODULE".TIMER_INFEED_MODULE_1_NOT_READY.Q;
END_REGION

REGION Network 7: INFEED MODULE 1 NOT READY ALARM
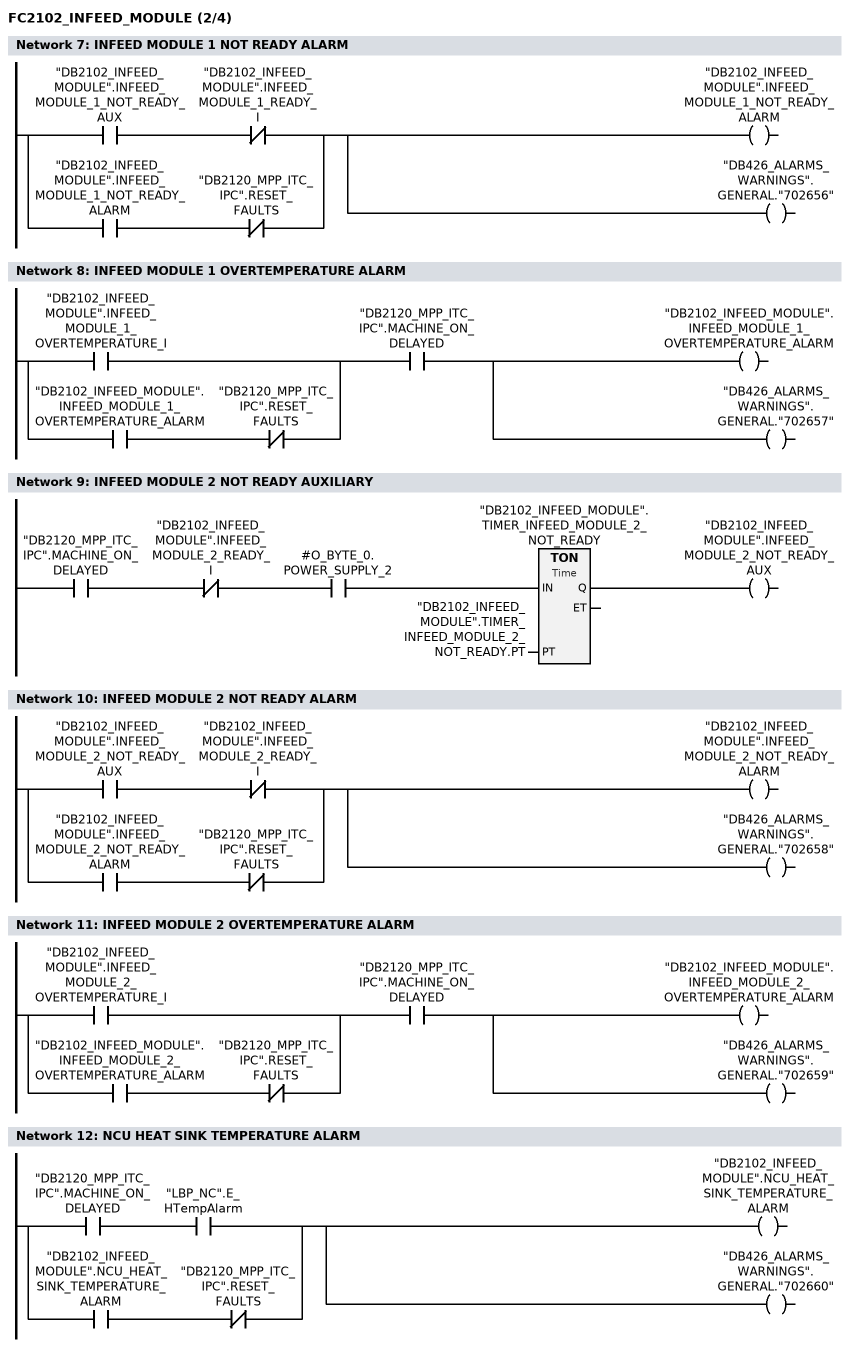
   RUNG wire#powerrail
      Contact( "DB2102_INFEED_MODULE".INFEED_MODULE_1_NOT_READY_AUX )
      I_Contact( "DB2102_INFEED_MODULE".INFEED_MODULE_1_READY_I )
      wire#w1
      Coil( "DB2102_INFEED_MODULE".INFEED_MODULE_1_NOT_READY_ALARM )
   END_RUNG
   RUNG wire#powerrail
      Contact( "DB2102_INFEED_MODULE".INFEED_MODULE_1_NOT_READY_ALARM )
      I_Contact( "DB2120_MPP_ITC_IPC".RESET_FAULTS )
   END_RUNG wire#w1
   RUNG wire#w1
      Coil( "DB426_ALARMS_WARNINGS".GENERAL."702656" )
   END_RUNG
   // the same network as SCL:
   "DB2102_INFEED_MODULE".INFEED_MODULE_1_NOT_READY_ALARM := ("DB2102_INFEED_MODULE".INFEED_MODULE_1_NOT_READY_AUX AND NOT "DB2102_INFEED_MODULE".INFEED_MODULE_1_READY_I) OR ("DB2102_INFEED_MODULE".INFEED_MODULE_1_NOT_READY_ALARM AND NOT "DB2120_MPP_ITC_IPC".RESET_FAULTS);
   "DB426_ALARMS_WARNINGS".GENERAL."702656" := "DB2102_INFEED_MODULE".INFEED_MODULE_1_NOT_READY_ALARM;
END_REGION

REGION Network 8: INFEED MODULE 1 OVERTEMPERATURE ALARM
   RUNG wire#powerrail
      Contact( "DB2102_INFEED_MODULE".INFEED_MODULE_1_OVERTEMPERATURE_I )
      wire#w1
      Contact( "DB2120_MPP_ITC_IPC".MACHINE_ON_DELAYED )
      wire#w2
      Coil( "DB2102_INFEED_MODULE".INFEED_MODULE_1_OVERTEMPERATURE_ALARM )
   END_RUNG
   RUNG wire#powerrail
      Contact( "DB2102_INFEED_MODULE".INFEED_MODULE_1_OVERTEMPERATURE_ALARM )
      I_Contact( "DB2120_MPP_ITC_IPC".RESET_FAULTS )
   END_RUNG wire#w1
   RUNG wire#w2
      Coil( "DB426_ALARMS_WARNINGS".GENERAL."702657" )
   END_RUNG
   // the same network as SCL:
   "DB2102_INFEED_MODULE".INFEED_MODULE_1_OVERTEMPERATURE_ALARM := ("DB2102_INFEED_MODULE".INFEED_MODULE_1_OVERTEMPERATURE_I OR ("DB2102_INFEED_MODULE".INFEED_MODULE_1_OVERTEMPERATURE_ALARM AND NOT "DB2120_MPP_ITC_IPC".RESET_FAULTS)) AND "DB2120_MPP_ITC_IPC".MACHINE_ON_DELAYED;
   "DB426_ALARMS_WARNINGS".GENERAL."702657" := "DB2102_INFEED_MODULE".INFEED_MODULE_1_OVERTEMPERATURE_ALARM;
END_REGION

REGION Network 9: INFEED MODULE 2 NOT READY AUXILIARY
   RUNG wire#powerrail
      Contact( "DB2120_MPP_ITC_IPC".MACHINE_ON_DELAYED )
      I_Contact( "DB2102_INFEED_MODULE".INFEED_MODULE_2_READY_I )
      Contact( #O_BYTE_0.POWER_SUPPLY_2 )
      { S7_Templates := "time_type := Time" } "DB2102_INFEED_MODULE".TIMER_INFEED_MODULE_2_NOT_READY.TON(pt := "DB2102_INFEED_MODULE".TIMER_INFEED_MODULE_2_NOT_READY.PT, et =>)
      Coil( "DB2102_INFEED_MODULE".INFEED_MODULE_2_NOT_READY_AUX )
   END_RUNG
   // the same network as SCL:
   "DB2102_INFEED_MODULE".TIMER_INFEED_MODULE_2_NOT_READY.TON(IN := "DB2120_MPP_ITC_IPC".MACHINE_ON_DELAYED AND NOT "DB2102_INFEED_MODULE".INFEED_MODULE_2_READY_I AND #O_BYTE_0.POWER_SUPPLY_2,
                           PT := "DB2102_INFEED_MODULE".TIMER_INFEED_MODULE_2_NOT_READY.PT);
   "DB2102_INFEED_MODULE".INFEED_MODULE_2_NOT_READY_AUX := "DB2102_INFEED_MODULE".TIMER_INFEED_MODULE_2_NOT_READY.Q;
END_REGION

REGION Network 10: INFEED MODULE 2 NOT READY ALARM
   RUNG wire#powerrail
      Contact( "DB2102_INFEED_MODULE".INFEED_MODULE_2_NOT_READY_AUX )
      I_Contact( "DB2102_INFEED_MODULE".INFEED_MODULE_2_READY_I )
      wire#w1
      Coil( "DB2102_INFEED_MODULE".INFEED_MODULE_2_NOT_READY_ALARM )
   END_RUNG
   RUNG wire#powerrail
      Contact( "DB2102_INFEED_MODULE".INFEED_MODULE_2_NOT_READY_ALARM )
      I_Contact( "DB2120_MPP_ITC_IPC".RESET_FAULTS )
   END_RUNG wire#w1
   RUNG wire#w1
      Coil( "DB426_ALARMS_WARNINGS".GENERAL."702658" )
   END_RUNG
   // the same network as SCL:
   "DB2102_INFEED_MODULE".INFEED_MODULE_2_NOT_READY_ALARM := ("DB2102_INFEED_MODULE".INFEED_MODULE_2_NOT_READY_AUX AND NOT "DB2102_INFEED_MODULE".INFEED_MODULE_2_READY_I) OR ("DB2102_INFEED_MODULE".INFEED_MODULE_2_NOT_READY_ALARM AND NOT "DB2120_MPP_ITC_IPC".RESET_FAULTS);
   "DB426_ALARMS_WARNINGS".GENERAL."702658" := "DB2102_INFEED_MODULE".INFEED_MODULE_2_NOT_READY_ALARM;
END_REGION

REGION Network 11: INFEED MODULE 2 OVERTEMPERATURE ALARM
   RUNG wire#powerrail
      Contact( "DB2102_INFEED_MODULE".INFEED_MODULE_2_OVERTEMPERATURE_I )
      wire#w1
      Contact( "DB2120_MPP_ITC_IPC".MACHINE_ON_DELAYED )
      wire#w2
      Coil( "DB2102_INFEED_MODULE".INFEED_MODULE_2_OVERTEMPERATURE_ALARM )
   END_RUNG
   RUNG wire#powerrail
      Contact( "DB2102_INFEED_MODULE".INFEED_MODULE_2_OVERTEMPERATURE_ALARM )
      I_Contact( "DB2120_MPP_ITC_IPC".RESET_FAULTS )
   END_RUNG wire#w1
   RUNG wire#w2
      Coil( "DB426_ALARMS_WARNINGS".GENERAL."702659" )
   END_RUNG
   // the same network as SCL:
   "DB2102_INFEED_MODULE".INFEED_MODULE_2_OVERTEMPERATURE_ALARM := ("DB2102_INFEED_MODULE".INFEED_MODULE_2_OVERTEMPERATURE_I OR ("DB2102_INFEED_MODULE".INFEED_MODULE_2_OVERTEMPERATURE_ALARM AND NOT "DB2120_MPP_ITC_IPC".RESET_FAULTS)) AND "DB2120_MPP_ITC_IPC".MACHINE_ON_DELAYED;
   "DB426_ALARMS_WARNINGS".GENERAL."702659" := "DB2102_INFEED_MODULE".INFEED_MODULE_2_OVERTEMPERATURE_ALARM;
END_REGION

REGION Network 12: NCU HEAT SINK TEMPERATURE ALARM
   RUNG wire#powerrail
      Contact( "DB2120_MPP_ITC_IPC".MACHINE_ON_DELAYED )
      Contact( "LBP_NC".E_HTempAlarm )
      wire#w1
      Coil( "DB2102_INFEED_MODULE".NCU_HEAT_SINK_TEMPERATURE_ALARM )
   END_RUNG
   RUNG wire#powerrail
      Contact( "DB2102_INFEED_MODULE".NCU_HEAT_SINK_TEMPERATURE_ALARM )
      I_Contact( "DB2120_MPP_ITC_IPC".RESET_FAULTS )
   END_RUNG wire#w1
   RUNG wire#w1
      Coil( "DB426_ALARMS_WARNINGS".GENERAL."702660" )
   END_RUNG
   // the same network as SCL:
   "DB2102_INFEED_MODULE".NCU_HEAT_SINK_TEMPERATURE_ALARM := ("DB2120_MPP_ITC_IPC".MACHINE_ON_DELAYED AND "LBP_NC".E_HTempAlarm) OR ("DB2102_INFEED_MODULE".NCU_HEAT_SINK_TEMPERATURE_ALARM AND NOT "DB2120_MPP_ITC_IPC".RESET_FAULTS);
   "DB426_ALARMS_WARNINGS".GENERAL."702660" := "DB2102_INFEED_MODULE".NCU_HEAT_SINK_TEMPERATURE_ALARM;
END_REGION

REGION Network 13: NCU LOW BATTERY ALARM
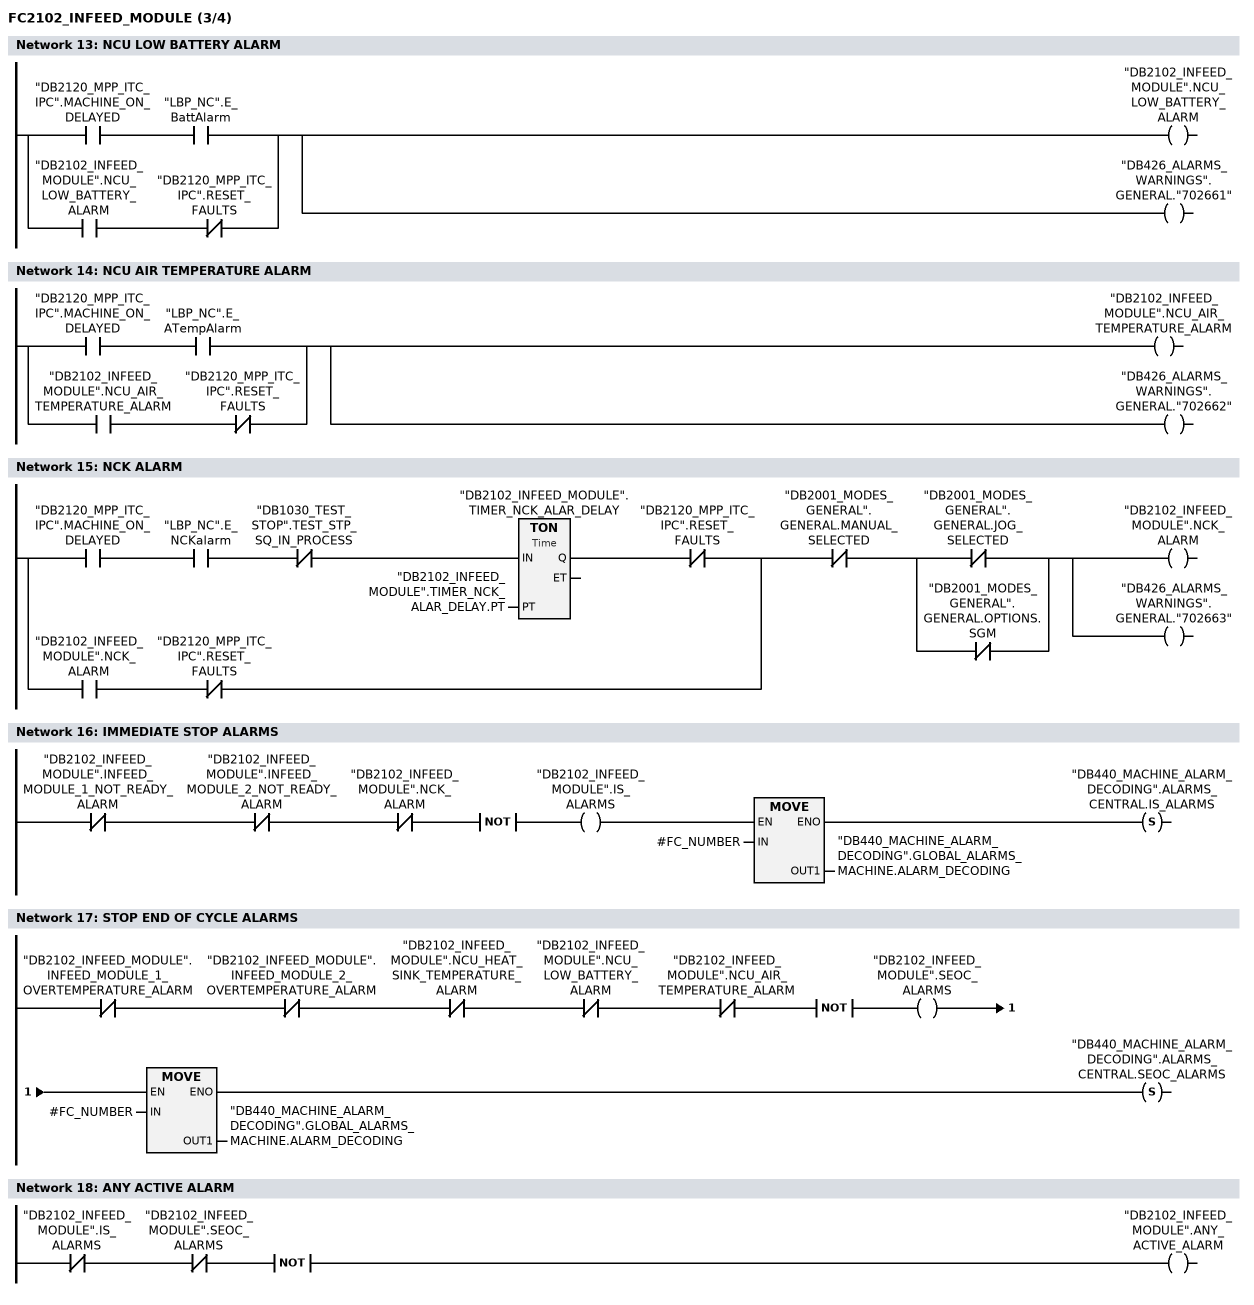
   RUNG wire#powerrail
      Contact( "DB2120_MPP_ITC_IPC".MACHINE_ON_DELAYED )
      Contact( "LBP_NC".E_BattAlarm )
      wire#w1
      Coil( "DB2102_INFEED_MODULE".NCU_LOW_BATTERY_ALARM )
   END_RUNG
   RUNG wire#powerrail
      Contact( "DB2102_INFEED_MODULE".NCU_LOW_BATTERY_ALARM )
      I_Contact( "DB2120_MPP_ITC_IPC".RESET_FAULTS )
   END_RUNG wire#w1
   RUNG wire#w1
      Coil( "DB426_ALARMS_WARNINGS".GENERAL."702661" )
   END_RUNG
   // the same network as SCL:
   "DB2102_INFEED_MODULE".NCU_LOW_BATTERY_ALARM := ("DB2120_MPP_ITC_IPC".MACHINE_ON_DELAYED AND "LBP_NC".E_BattAlarm) OR ("DB2102_INFEED_MODULE".NCU_LOW_BATTERY_ALARM AND NOT "DB2120_MPP_ITC_IPC".RESET_FAULTS);
   "DB426_ALARMS_WARNINGS".GENERAL."702661" := "DB2102_INFEED_MODULE".NCU_LOW_BATTERY_ALARM;
END_REGION

REGION Network 14: NCU AIR TEMPERATURE ALARM
   RUNG wire#powerrail
      Contact( "DB2120_MPP_ITC_IPC".MACHINE_ON_DELAYED )
      Contact( "LBP_NC".E_ATempAlarm )
      wire#w1
      Coil( "DB2102_INFEED_MODULE".NCU_AIR_TEMPERATURE_ALARM )
   END_RUNG
   RUNG wire#powerrail
      Contact( "DB2102_INFEED_MODULE".NCU_AIR_TEMPERATURE_ALARM )
      I_Contact( "DB2120_MPP_ITC_IPC".RESET_FAULTS )
   END_RUNG wire#w1
   RUNG wire#w1
      Coil( "DB426_ALARMS_WARNINGS".GENERAL."702662" )
   END_RUNG
   // the same network as SCL:
   "DB2102_INFEED_MODULE".NCU_AIR_TEMPERATURE_ALARM := ("DB2120_MPP_ITC_IPC".MACHINE_ON_DELAYED AND "LBP_NC".E_ATempAlarm) OR ("DB2102_INFEED_MODULE".NCU_AIR_TEMPERATURE_ALARM AND NOT "DB2120_MPP_ITC_IPC".RESET_FAULTS);
   "DB426_ALARMS_WARNINGS".GENERAL."702662" := "DB2102_INFEED_MODULE".NCU_AIR_TEMPERATURE_ALARM;
END_REGION

REGION Network 15: NCK ALARM
   RUNG wire#powerrail
      Contact( "DB2120_MPP_ITC_IPC".MACHINE_ON_DELAYED )
      Contact( "LBP_NC".E_NCKalarm )
      I_Contact( "DB1030_TEST_STOP".TEST_STP_SQ_IN_PROCESS )
      { S7_Templates := "time_type := Time" } "DB2102_INFEED_MODULE".TIMER_NCK_ALAR_DELAY.TON(pt := "DB2102_INFEED_MODULE".TIMER_NCK_ALAR_DELAY.PT, et =>)
      I_Contact( "DB2120_MPP_ITC_IPC".RESET_FAULTS )
      wire#w1
      I_Contact( "DB2001_MODES_GENERAL".GENERAL.MANUAL_SELECTED )
      wire#w2
      I_Contact( "DB2001_MODES_GENERAL".GENERAL.JOG_SELECTED )
      wire#w3
      Coil( "DB2102_INFEED_MODULE".NCK_ALARM )
   END_RUNG
   RUNG wire#powerrail
      Contact( "DB2102_INFEED_MODULE".NCK_ALARM )
      I_Contact( "DB2120_MPP_ITC_IPC".RESET_FAULTS )
   END_RUNG wire#w1
   RUNG wire#w2
      I_Contact( "DB2001_MODES_GENERAL".GENERAL.OPTIONS.SGM )
   END_RUNG wire#w3
   RUNG wire#w3
      Coil( "DB426_ALARMS_WARNINGS".GENERAL."702663" )
   END_RUNG
   // the same network as SCL:
   "DB2102_INFEED_MODULE".TIMER_NCK_ALAR_DELAY.TON(IN := "DB2120_MPP_ITC_IPC".MACHINE_ON_DELAYED AND "LBP_NC".E_NCKalarm AND NOT "DB1030_TEST_STOP".TEST_STP_SQ_IN_PROCESS,
                           PT := "DB2102_INFEED_MODULE".TIMER_NCK_ALAR_DELAY.PT);
   "DB2102_INFEED_MODULE".NCK_ALARM := (("DB2102_INFEED_MODULE".TIMER_NCK_ALAR_DELAY.Q AND NOT "DB2120_MPP_ITC_IPC".RESET_FAULTS) OR ("DB2102_INFEED_MODULE".NCK_ALARM AND NOT "DB2120_MPP_ITC_IPC".RESET_FAULTS)) AND NOT "DB2001_MODES_GENERAL".GENERAL.MANUAL_SELECTED AND (NOT "DB2001_MODES_GENERAL".GENERAL.JOG_SELECTED OR NOT "DB2001_MODES_GENERAL".GENERAL.OPTIONS.SGM);
   "DB426_ALARMS_WARNINGS".GENERAL."702663" := "DB2102_INFEED_MODULE".NCK_ALARM;
END_REGION

REGION Network 16: IMMEDIATE STOP ALARMS
   RUNG wire#powerrail
      I_Contact( "DB2102_INFEED_MODULE".INFEED_MODULE_1_NOT_READY_ALARM )
      I_Contact( "DB2102_INFEED_MODULE".INFEED_MODULE_2_NOT_READY_ALARM )
      I_Contact( "DB2102_INFEED_MODULE".NCK_ALARM )
      Not()
      Coil( "DB2102_INFEED_MODULE".IS_ALARMS )
      { S7_GenerateENO := "TRUE" } Move(in := #FC_NUMBER, out1 => "DB440_MACHINE_ALARM_DECODING".GLOBAL_ALARMS_MACHINE.ALARM_DECODING)
      S_Coil( "DB440_MACHINE_ALARM_DECODING".ALARMS_CENTRAL.IS_ALARMS )
   END_RUNG
   // the same network as SCL:
   // ENO of a box is taken as its EN; it also drops when the box reports an error
   "DB2102_INFEED_MODULE".IS_ALARMS := NOT (NOT "DB2102_INFEED_MODULE".INFEED_MODULE_1_NOT_READY_ALARM AND NOT "DB2102_INFEED_MODULE".INFEED_MODULE_2_NOT_READY_ALARM AND NOT "DB2102_INFEED_MODULE".NCK_ALARM);
   IF "DB2102_INFEED_MODULE".IS_ALARMS THEN
       "DB440_MACHINE_ALARM_DECODING".GLOBAL_ALARMS_MACHINE.ALARM_DECODING := #FC_NUMBER;
       "DB440_MACHINE_ALARM_DECODING".ALARMS_CENTRAL.IS_ALARMS := TRUE;
   END_IF;
END_REGION

REGION Network 17: STOP END OF CYCLE ALARMS
   RUNG wire#powerrail
      I_Contact( "DB2102_INFEED_MODULE".INFEED_MODULE_1_OVERTEMPERATURE_ALARM )
      I_Contact( "DB2102_INFEED_MODULE".INFEED_MODULE_2_OVERTEMPERATURE_ALARM )
      I_Contact( "DB2102_INFEED_MODULE".NCU_HEAT_SINK_TEMPERATURE_ALARM )
      I_Contact( "DB2102_INFEED_MODULE".NCU_LOW_BATTERY_ALARM )
      I_Contact( "DB2102_INFEED_MODULE".NCU_AIR_TEMPERATURE_ALARM )
      Not()
      Coil( "DB2102_INFEED_MODULE".SEOC_ALARMS )
      { S7_GenerateENO := "TRUE" } Move(in := #FC_NUMBER, out1 => "DB440_MACHINE_ALARM_DECODING".GLOBAL_ALARMS_MACHINE.ALARM_DECODING)
      S_Coil( "DB440_MACHINE_ALARM_DECODING".ALARMS_CENTRAL.SEOC_ALARMS )
   END_RUNG
   // the same network as SCL:
   // ENO of a box is taken as its EN; it also drops when the box reports an error
   "DB2102_INFEED_MODULE".SEOC_ALARMS := NOT (NOT "DB2102_INFEED_MODULE".INFEED_MODULE_1_OVERTEMPERATURE_ALARM AND NOT "DB2102_INFEED_MODULE".INFEED_MODULE_2_OVERTEMPERATURE_ALARM AND NOT "DB2102_INFEED_MODULE".NCU_HEAT_SINK_TEMPERATURE_ALARM AND NOT "DB2102_INFEED_MODULE".NCU_LOW_BATTERY_ALARM AND NOT "DB2102_INFEED_MODULE".NCU_AIR_TEMPERATURE_ALARM);
   IF "DB2102_INFEED_MODULE".SEOC_ALARMS THEN
       "DB440_MACHINE_ALARM_DECODING".GLOBAL_ALARMS_MACHINE.ALARM_DECODING := #FC_NUMBER;
       "DB440_MACHINE_ALARM_DECODING".ALARMS_CENTRAL.SEOC_ALARMS := TRUE;
   END_IF;
END_REGION

REGION Network 18: ANY ACTIVE ALARM
   RUNG wire#powerrail
      I_Contact( "DB2102_INFEED_MODULE".IS_ALARMS )
      I_Contact( "DB2102_INFEED_MODULE".SEOC_ALARMS )
      Not()
      Coil( "DB2102_INFEED_MODULE".ANY_ACTIVE_ALARM )
   END_RUNG
   // the same network as SCL:
   "DB2102_INFEED_MODULE".ANY_ACTIVE_ALARM := NOT (NOT "DB2102_INFEED_MODULE".IS_ALARMS AND NOT "DB2102_INFEED_MODULE".SEOC_ALARMS);
END_REGION

REGION Network 19: INFEED MODULE OFF 3 OUTPUT
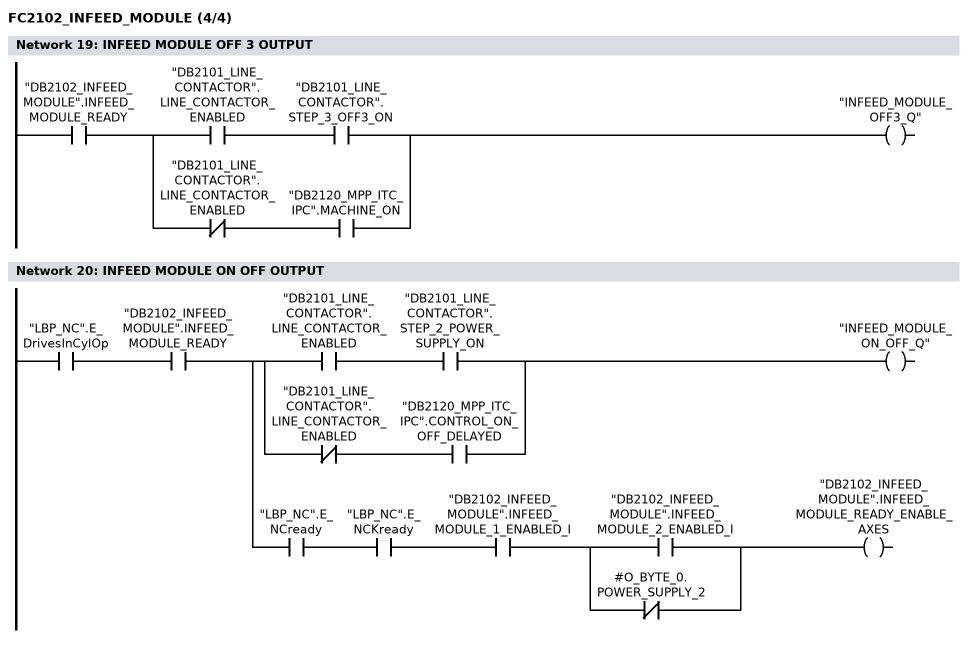
   RUNG wire#powerrail
      Contact( "DB2102_INFEED_MODULE".INFEED_MODULE_READY )
      wire#w1
      Contact( "DB2101_LINE_CONTACTOR".LINE_CONTACTOR_ENABLED )
      Contact( "DB2101_LINE_CONTACTOR".STEP_3_OFF3_ON )
      wire#w2
      Coil( "INFEED_MODULE_OFF3_Q" )
   END_RUNG
   RUNG wire#w1
      I_Contact( "DB2101_LINE_CONTACTOR".LINE_CONTACTOR_ENABLED )
      Contact( "DB2120_MPP_ITC_IPC".MACHINE_ON )
   END_RUNG wire#w2
   // the same network as SCL:
   "INFEED_MODULE_OFF3_Q" := "DB2102_INFEED_MODULE".INFEED_MODULE_READY AND (("DB2101_LINE_CONTACTOR".LINE_CONTACTOR_ENABLED AND "DB2101_LINE_CONTACTOR".STEP_3_OFF3_ON) OR (NOT "DB2101_LINE_CONTACTOR".LINE_CONTACTOR_ENABLED AND "DB2120_MPP_ITC_IPC".MACHINE_ON));
END_REGION

REGION Network 20: INFEED MODULE ON OFF OUTPUT
   RUNG wire#powerrail
      Contact( "LBP_NC".E_DrivesInCylOp )
      Contact( "DB2102_INFEED_MODULE".INFEED_MODULE_READY )
      wire#w1
      Contact( "DB2101_LINE_CONTACTOR".LINE_CONTACTOR_ENABLED )
      Contact( "DB2101_LINE_CONTACTOR".STEP_2_POWER_SUPPLY_ON )
      wire#w2
      Coil( "INFEED_MODULE_ON_OFF_Q" )
   END_RUNG
   RUNG wire#w1
      I_Contact( "DB2101_LINE_CONTACTOR".LINE_CONTACTOR_ENABLED )
      Contact( "DB2120_MPP_ITC_IPC".CONTROL_ON_OFF_DELAYED )
   END_RUNG wire#w2
   RUNG wire#w1
      Contact( "LBP_NC".E_NCready )
      Contact( "LBP_NC".E_NCKready )
      Contact( "DB2102_INFEED_MODULE".INFEED_MODULE_1_ENABLED_I )
      wire#w3
      Contact( "DB2102_INFEED_MODULE".INFEED_MODULE_2_ENABLED_I )
      wire#w4
      Coil( "DB2102_INFEED_MODULE".INFEED_MODULE_READY_ENABLE_AXES )
   END_RUNG
   RUNG wire#w3
      I_Contact( #O_BYTE_0.POWER_SUPPLY_2 )
   END_RUNG wire#w4
   // the same network as SCL:
   #_w1 := "LBP_NC".E_DrivesInCylOp AND "DB2102_INFEED_MODULE".INFEED_MODULE_READY;
   "INFEED_MODULE_ON_OFF_Q" := #_w1 AND (("DB2101_LINE_CONTACTOR".LINE_CONTACTOR_ENABLED AND "DB2101_LINE_CONTACTOR".STEP_2_POWER_SUPPLY_ON) OR (NOT "DB2101_LINE_CONTACTOR".LINE_CONTACTOR_ENABLED AND "DB2120_MPP_ITC_IPC".CONTROL_ON_OFF_DELAYED));
   "DB2102_INFEED_MODULE".INFEED_MODULE_READY_ENABLE_AXES := #_w1 AND "LBP_NC".E_NCready AND "LBP_NC".E_NCKready AND "DB2102_INFEED_MODULE".INFEED_MODULE_1_ENABLED_I AND ("DB2102_INFEED_MODULE".INFEED_MODULE_2_ENABLED_I OR NOT #O_BYTE_0.POWER_SUPPLY_2);
END_REGION
END_FUNCTION

FUNCTION "FC2106_SIGNAL_TOWER" : Void   // FC2106, LAD
{ S7_Optimized_Access := 'FALSE' }
AUTHOR : ETXETAR
VERSION : 1.0
// stored: AutoNumber false, IsIECCheckEnabled false, SetENOAutomatically false, UDAEnableTagReadback false
BEGIN

REGION Network 1: SIGNAL TOWER GREEN LIGHT OUTPUT / SIGNAL TOWER, GREEN LIGHT
   // GREEN LIGHT
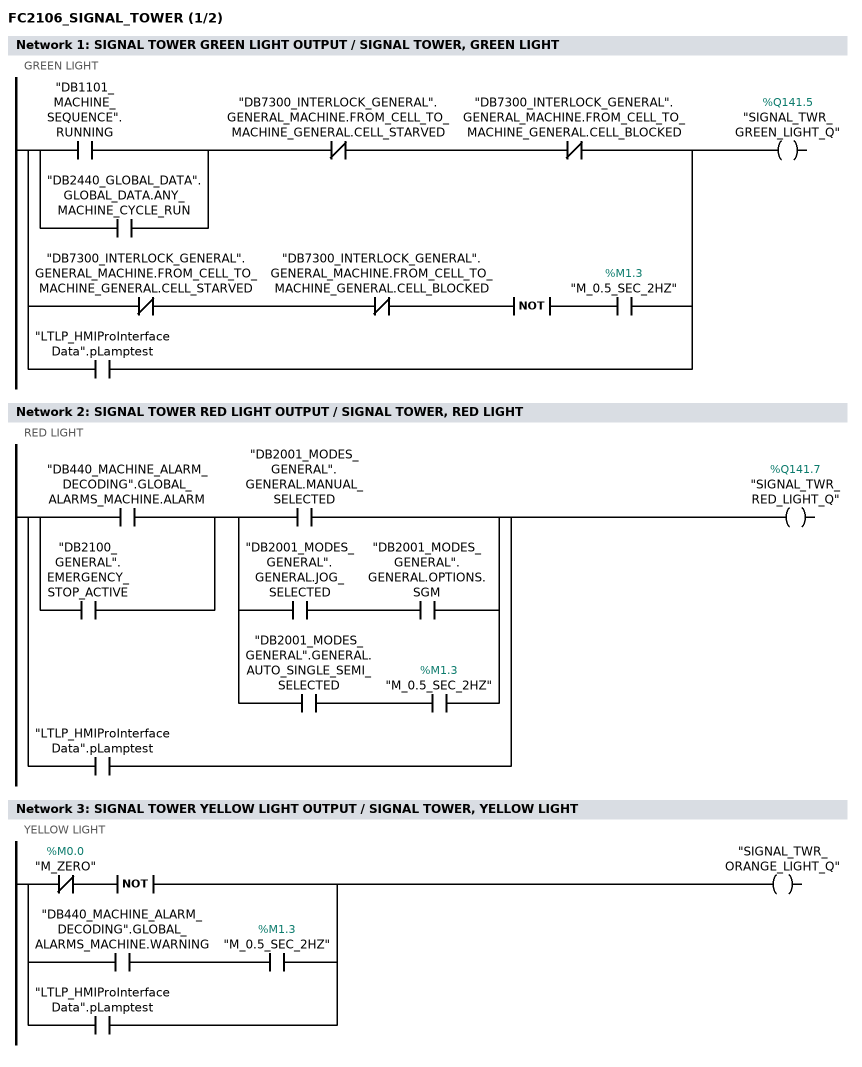
   RUNG wire#powerrail
      Contact( "DB1101_MACHINE_SEQUENCE".RUNNING )
      wire#w1
      I_Contact( "DB7300_INTERLOCK_GENERAL".GENERAL_MACHINE.FROM_CELL_TO_MACHINE_GENERAL.CELL_STARVED )
      I_Contact( "DB7300_INTERLOCK_GENERAL".GENERAL_MACHINE.FROM_CELL_TO_MACHINE_GENERAL.CELL_BLOCKED )
      wire#w2
      Coil( "SIGNAL_TWR_GREEN_LIGHT_Q" )
   END_RUNG
   RUNG wire#powerrail
      Contact( "DB2440_GLOBAL_DATA".GLOBAL_DATA.ANY_MACHINE_CYCLE_RUN )
   END_RUNG wire#w1
   RUNG wire#powerrail
      I_Contact( "DB7300_INTERLOCK_GENERAL".GENERAL_MACHINE.FROM_CELL_TO_MACHINE_GENERAL.CELL_STARVED )
      I_Contact( "DB7300_INTERLOCK_GENERAL".GENERAL_MACHINE.FROM_CELL_TO_MACHINE_GENERAL.CELL_BLOCKED )
      Not()
      Contact( "M_0.5_SEC_2HZ" )
   END_RUNG wire#w2
   RUNG wire#powerrail
      Contact( "LTLP_HMIProInterfaceData".pLamptest )
   END_RUNG wire#w2
   // the same network as SCL:
   "SIGNAL_TWR_GREEN_LIGHT_Q" := (("DB1101_MACHINE_SEQUENCE".RUNNING OR "DB2440_GLOBAL_DATA".GLOBAL_DATA.ANY_MACHINE_CYCLE_RUN) AND NOT "DB7300_INTERLOCK_GENERAL".GENERAL_MACHINE.FROM_CELL_TO_MACHINE_GENERAL.CELL_STARVED AND NOT "DB7300_INTERLOCK_GENERAL".GENERAL_MACHINE.FROM_CELL_TO_MACHINE_GENERAL.CELL_BLOCKED) OR (NOT (NOT "DB7300_INTERLOCK_GENERAL".GENERAL_MACHINE.FROM_CELL_TO_MACHINE_GENERAL.CELL_STARVED AND NOT "DB7300_INTERLOCK_GENERAL".GENERAL_MACHINE.FROM_CELL_TO_MACHINE_GENERAL.CELL_BLOCKED) AND "M_0.5_SEC_2HZ") OR "LTLP_HMIProInterfaceData".pLamptest;
END_REGION

REGION Network 2: SIGNAL TOWER RED LIGHT OUTPUT / SIGNAL TOWER, RED LIGHT
   // RED LIGHT
   RUNG wire#powerrail
      Contact( "DB440_MACHINE_ALARM_DECODING".GLOBAL_ALARMS_MACHINE.ALARM )
      wire#w1
      Contact( "DB2001_MODES_GENERAL".GENERAL.MANUAL_SELECTED )
      wire#w2
      Coil( "SIGNAL_TWR_RED_LIGHT_Q" )
   END_RUNG
   RUNG wire#powerrail
      Contact( "DB2100_GENERAL".EMERGENCY_STOP_ACTIVE )
   END_RUNG wire#w1
   RUNG wire#w1
      Contact( "DB2001_MODES_GENERAL".GENERAL.JOG_SELECTED )
      Contact( "DB2001_MODES_GENERAL".GENERAL.OPTIONS.SGM )
   END_RUNG wire#w2
   RUNG wire#w1
      Contact( "DB2001_MODES_GENERAL".GENERAL.AUTO_SINGLE_SEMI_SELECTED )
      Contact( "M_0.5_SEC_2HZ" )
   END_RUNG wire#w2
   RUNG wire#powerrail
      Contact( "LTLP_HMIProInterfaceData".pLamptest )
   END_RUNG wire#w2
   // the same network as SCL:
   "SIGNAL_TWR_RED_LIGHT_Q" := (("DB440_MACHINE_ALARM_DECODING".GLOBAL_ALARMS_MACHINE.ALARM OR "DB2100_GENERAL".EMERGENCY_STOP_ACTIVE) AND ("DB2001_MODES_GENERAL".GENERAL.MANUAL_SELECTED OR ("DB2001_MODES_GENERAL".GENERAL.JOG_SELECTED AND "DB2001_MODES_GENERAL".GENERAL.OPTIONS.SGM) OR ("DB2001_MODES_GENERAL".GENERAL.AUTO_SINGLE_SEMI_SELECTED AND "M_0.5_SEC_2HZ"))) OR "LTLP_HMIProInterfaceData".pLamptest;
END_REGION

REGION Network 3: SIGNAL TOWER YELLOW LIGHT OUTPUT / SIGNAL TOWER, YELLOW LIGHT
   // YELLOW LIGHT
   RUNG wire#powerrail
      I_Contact( "M_ZERO" )
      Not()
      wire#w1
      Coil( "SIGNAL_TWR_ORANGE_LIGHT_Q" )
   END_RUNG
   RUNG wire#powerrail
      Contact( "DB440_MACHINE_ALARM_DECODING".GLOBAL_ALARMS_MACHINE.WARNING )
      Contact( "M_0.5_SEC_2HZ" )
   END_RUNG wire#w1
   RUNG wire#powerrail
      Contact( "LTLP_HMIProInterfaceData".pLamptest )
   END_RUNG wire#w1
   // the same network as SCL:
   "SIGNAL_TWR_ORANGE_LIGHT_Q" := NOT (NOT "M_ZERO") OR ("DB440_MACHINE_ALARM_DECODING".GLOBAL_ALARMS_MACHINE.WARNING AND "M_0.5_SEC_2HZ") OR "LTLP_HMIProInterfaceData".pLamptest;
END_REGION

REGION Network 4: SIGNAL TOWER BLUE LIGHT OUTPUT / SIGNAL TOWER, BLUE LED
   // Blue Light
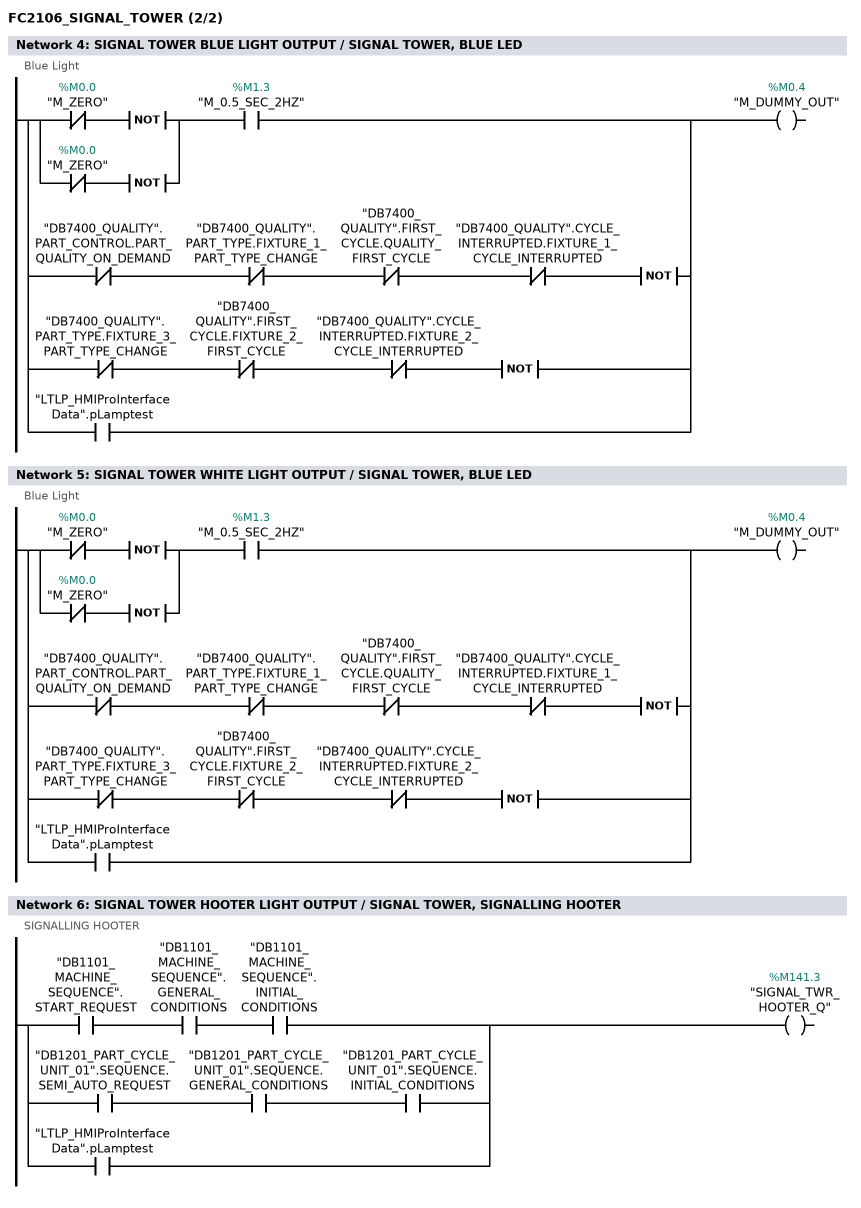
   RUNG wire#powerrail
      I_Contact( "M_ZERO" )
      Not()
      wire#w1
      Contact( "M_0.5_SEC_2HZ" )
      wire#w2
      Coil( "M_DUMMY_OUT" )
   END_RUNG
   RUNG wire#powerrail
      I_Contact( "M_ZERO" )
      Not()
   END_RUNG wire#w1
   RUNG wire#powerrail
      I_Contact( "DB7400_QUALITY".PART_CONTROL.PART_QUALITY_ON_DEMAND )
      I_Contact( "DB7400_QUALITY".PART_TYPE.FIXTURE_1_PART_TYPE_CHANGE )
      I_Contact( "DB7400_QUALITY".FIRST_CYCLE.QUALITY_FIRST_CYCLE )
      I_Contact( "DB7400_QUALITY".CYCLE_INTERRUPTED.FIXTURE_1_CYCLE_INTERRUPTED )
      Not()
   END_RUNG wire#w2
   RUNG wire#powerrail
      I_Contact( "DB7400_QUALITY".PART_TYPE.FIXTURE_3_PART_TYPE_CHANGE )
      I_Contact( "DB7400_QUALITY".FIRST_CYCLE.FIXTURE_2_FIRST_CYCLE )
      I_Contact( "DB7400_QUALITY".CYCLE_INTERRUPTED.FIXTURE_2_CYCLE_INTERRUPTED )
      Not()
   END_RUNG wire#w2
   RUNG wire#powerrail
      Contact( "LTLP_HMIProInterfaceData".pLamptest )
   END_RUNG wire#w2
   // the same network as SCL:
   "M_DUMMY_OUT" := ((NOT (NOT "M_ZERO") OR NOT (NOT "M_ZERO")) AND "M_0.5_SEC_2HZ") OR NOT (NOT "DB7400_QUALITY".PART_CONTROL.PART_QUALITY_ON_DEMAND AND NOT "DB7400_QUALITY".PART_TYPE.FIXTURE_1_PART_TYPE_CHANGE AND NOT "DB7400_QUALITY".FIRST_CYCLE.QUALITY_FIRST_CYCLE AND NOT "DB7400_QUALITY".CYCLE_INTERRUPTED.FIXTURE_1_CYCLE_INTERRUPTED) OR NOT (NOT "DB7400_QUALITY".PART_TYPE.FIXTURE_3_PART_TYPE_CHANGE AND NOT "DB7400_QUALITY".FIRST_CYCLE.FIXTURE_2_FIRST_CYCLE AND NOT "DB7400_QUALITY".CYCLE_INTERRUPTED.FIXTURE_2_CYCLE_INTERRUPTED) OR "LTLP_HMIProInterfaceData".pLamptest;
END_REGION

REGION Network 5: SIGNAL TOWER WHITE LIGHT OUTPUT / SIGNAL TOWER, BLUE LED
   // Blue Light
   RUNG wire#powerrail
      I_Contact( "M_ZERO" )
      Not()
      wire#w1
      Contact( "M_0.5_SEC_2HZ" )
      wire#w2
      Coil( "M_DUMMY_OUT" )
   END_RUNG
   RUNG wire#powerrail
      I_Contact( "M_ZERO" )
      Not()
   END_RUNG wire#w1
   RUNG wire#powerrail
      I_Contact( "DB7400_QUALITY".PART_CONTROL.PART_QUALITY_ON_DEMAND )
      I_Contact( "DB7400_QUALITY".PART_TYPE.FIXTURE_1_PART_TYPE_CHANGE )
      I_Contact( "DB7400_QUALITY".FIRST_CYCLE.QUALITY_FIRST_CYCLE )
      I_Contact( "DB7400_QUALITY".CYCLE_INTERRUPTED.FIXTURE_1_CYCLE_INTERRUPTED )
      Not()
   END_RUNG wire#w2
   RUNG wire#powerrail
      I_Contact( "DB7400_QUALITY".PART_TYPE.FIXTURE_3_PART_TYPE_CHANGE )
      I_Contact( "DB7400_QUALITY".FIRST_CYCLE.FIXTURE_2_FIRST_CYCLE )
      I_Contact( "DB7400_QUALITY".CYCLE_INTERRUPTED.FIXTURE_2_CYCLE_INTERRUPTED )
      Not()
   END_RUNG wire#w2
   RUNG wire#powerrail
      Contact( "LTLP_HMIProInterfaceData".pLamptest )
   END_RUNG wire#w2
   // the same network as SCL:
   "M_DUMMY_OUT" := ((NOT (NOT "M_ZERO") OR NOT (NOT "M_ZERO")) AND "M_0.5_SEC_2HZ") OR NOT (NOT "DB7400_QUALITY".PART_CONTROL.PART_QUALITY_ON_DEMAND AND NOT "DB7400_QUALITY".PART_TYPE.FIXTURE_1_PART_TYPE_CHANGE AND NOT "DB7400_QUALITY".FIRST_CYCLE.QUALITY_FIRST_CYCLE AND NOT "DB7400_QUALITY".CYCLE_INTERRUPTED.FIXTURE_1_CYCLE_INTERRUPTED) OR NOT (NOT "DB7400_QUALITY".PART_TYPE.FIXTURE_3_PART_TYPE_CHANGE AND NOT "DB7400_QUALITY".FIRST_CYCLE.FIXTURE_2_FIRST_CYCLE AND NOT "DB7400_QUALITY".CYCLE_INTERRUPTED.FIXTURE_2_CYCLE_INTERRUPTED) OR "LTLP_HMIProInterfaceData".pLamptest;
END_REGION

REGION Network 6: SIGNAL TOWER HOOTER LIGHT OUTPUT / SIGNAL TOWER, SIGNALLING HOOTER
   // SIGNALLING HOOTER
   RUNG wire#powerrail
      Contact( "DB1101_MACHINE_SEQUENCE".START_REQUEST )
      Contact( "DB1101_MACHINE_SEQUENCE".GENERAL_CONDITIONS )
      Contact( "DB1101_MACHINE_SEQUENCE".INITIAL_CONDITIONS )
      wire#w1
      Coil( "SIGNAL_TWR_HOOTER_Q" )
   END_RUNG
   RUNG wire#powerrail
      Contact( "DB1201_PART_CYCLE_UNIT_01".SEQUENCE.SEMI_AUTO_REQUEST )
      Contact( "DB1201_PART_CYCLE_UNIT_01".SEQUENCE.GENERAL_CONDITIONS )
      Contact( "DB1201_PART_CYCLE_UNIT_01".SEQUENCE.INITIAL_CONDITIONS )
   END_RUNG wire#w1
   RUNG wire#powerrail
      Contact( "LTLP_HMIProInterfaceData".pLamptest )
   END_RUNG wire#w1
   // the same network as SCL:
   "SIGNAL_TWR_HOOTER_Q" := ("DB1101_MACHINE_SEQUENCE".START_REQUEST AND "DB1101_MACHINE_SEQUENCE".GENERAL_CONDITIONS AND "DB1101_MACHINE_SEQUENCE".INITIAL_CONDITIONS) OR ("DB1201_PART_CYCLE_UNIT_01".SEQUENCE.SEMI_AUTO_REQUEST AND "DB1201_PART_CYCLE_UNIT_01".SEQUENCE.GENERAL_CONDITIONS AND "DB1201_PART_CYCLE_UNIT_01".SEQUENCE.INITIAL_CONDITIONS) OR "LTLP_HMIProInterfaceData".pLamptest;
END_REGION
END_FUNCTION

FUNCTION "FC2107_MACHINE_LIGHT" : Void   // FC2107, LAD
{ S7_Optimized_Access := 'FALSE' }
AUTHOR : ETXETAR
VERSION : 1.0
// stored: AutoNumber false, IsIECCheckEnabled false, SetENOAutomatically false, UDAEnableTagReadback false
BEGIN

REGION Network 1: MACHINE LIGHT
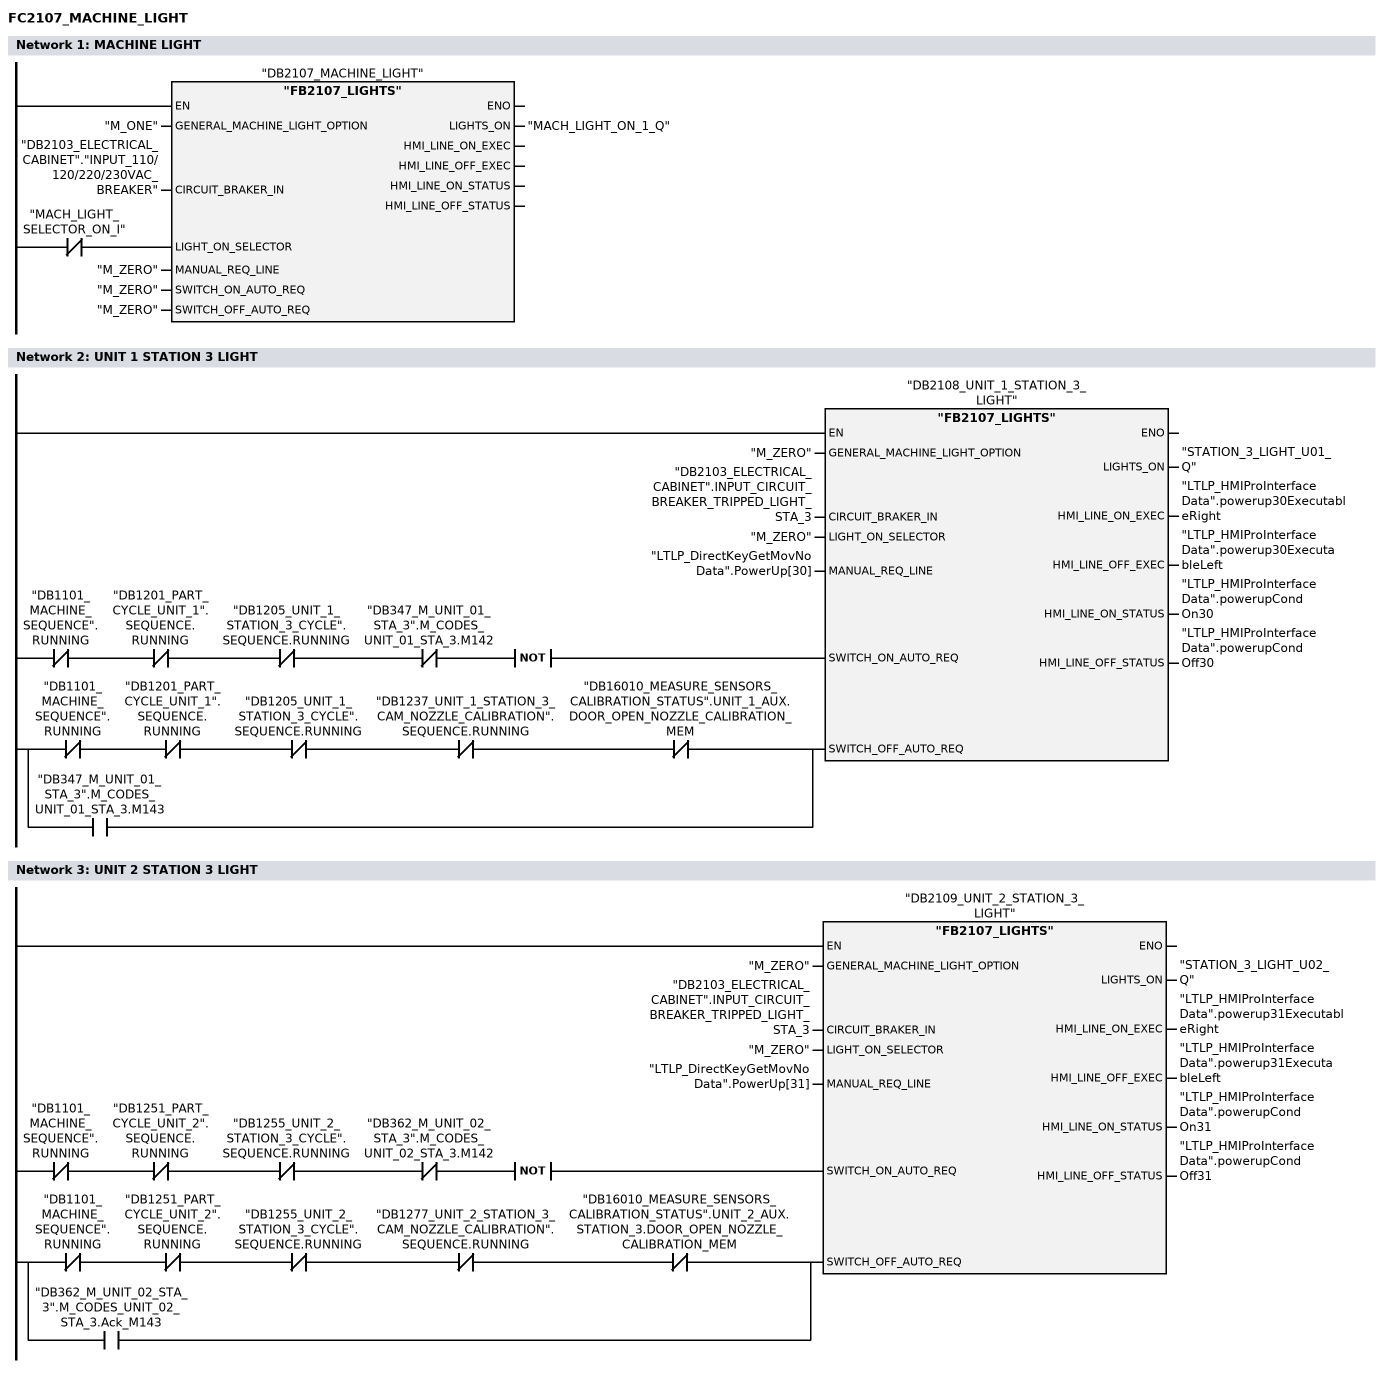
   RUNG wire#powerrail
      "DB2107_MACHINE_LIGHT"(LIGHT_ON_SELECTOR := wire#w1, GENERAL_MACHINE_LIGHT_OPTION := "M_ONE", CIRCUIT_BRAKER_IN := "DB2103_ELECTRICAL_CABINET"."INPUT_110/120/220/230VAC_BREAKER", MANUAL_REQ_LINE := "M_ZERO", SWITCH_ON_AUTO_REQ := "M_ZERO", SWITCH_OFF_AUTO_REQ := "M_ZERO", LIGHTS_ON => "MACH_LIGHT_ON_1_Q", HMI_LINE_ON_EXEC =>, HMI_LINE_OFF_EXEC =>, HMI_LINE_ON_STATUS =>, HMI_LINE_OFF_STATUS =>)
   END_RUNG
   RUNG wire#powerrail
      I_Contact( "MACH_LIGHT_SELECTOR_ON_I" )
   END_RUNG wire#w1
   // the same network as SCL:
   "DB2107_MACHINE_LIGHT"(GENERAL_MACHINE_LIGHT_OPTION := "M_ONE",   // "FB2107_LIGHTS"
                          CIRCUIT_BRAKER_IN := "DB2103_ELECTRICAL_CABINET"."INPUT_110/120/220/230VAC_BREAKER",
                          LIGHT_ON_SELECTOR := NOT "MACH_LIGHT_SELECTOR_ON_I",
                          MANUAL_REQ_LINE := "M_ZERO",
                          SWITCH_ON_AUTO_REQ := "M_ZERO",
                          SWITCH_OFF_AUTO_REQ := "M_ZERO",
                          LIGHTS_ON => "MACH_LIGHT_ON_1_Q");
END_REGION

REGION Network 2: UNIT 1 STATION 3 LIGHT
   RUNG wire#powerrail
      "DB2108_UNIT_1_STATION_3_LIGHT"(SWITCH_ON_AUTO_REQ := wire#w1, SWITCH_OFF_AUTO_REQ := wire#w2, GENERAL_MACHINE_LIGHT_OPTION := "M_ZERO", CIRCUIT_BRAKER_IN := "DB2103_ELECTRICAL_CABINET".INPUT_CIRCUIT_BREAKER_TRIPPED_LIGHT_STA_3, LIGHT_ON_SELECTOR := "M_ZERO", MANUAL_REQ_LINE := "LTLP_DirectKeyGetMovNoData".PowerUp[30], LIGHTS_ON => "STATION_3_LIGHT_U01_Q", HMI_LINE_ON_EXEC => "LTLP_HMIProInterfaceData".powerup30ExecutableRight, HMI_LINE_OFF_EXEC => "LTLP_HMIProInterfaceData".powerup30ExecutableLeft, HMI_LINE_ON_STATUS => "LTLP_HMIProInterfaceData".powerupCondOn30, HMI_LINE_OFF_STATUS => "LTLP_HMIProInterfaceData".powerupCondOff30)
   END_RUNG
   RUNG wire#powerrail
      I_Contact( "DB1101_MACHINE_SEQUENCE".RUNNING )
      I_Contact( "DB1201_PART_CYCLE_UNIT_1".SEQUENCE.RUNNING )
      I_Contact( "DB1205_UNIT_1_STATION_3_CYCLE".SEQUENCE.RUNNING )
      I_Contact( "DB347_M_UNIT_01_STA_3".M_CODES_UNIT_01_STA_3.M142 )
      Not()
   END_RUNG wire#w1
   RUNG wire#powerrail
      I_Contact( "DB1101_MACHINE_SEQUENCE".RUNNING )
      I_Contact( "DB1201_PART_CYCLE_UNIT_1".SEQUENCE.RUNNING )
      I_Contact( "DB1205_UNIT_1_STATION_3_CYCLE".SEQUENCE.RUNNING )
      I_Contact( "DB1237_UNIT_1_STATION_3_CAM_NOZZLE_CALIBRATION".SEQUENCE.RUNNING )
      I_Contact( "DB16010_MEASURE_SENSORS_CALIBRATION_STATUS".UNIT_1_AUX.DOOR_OPEN_NOZZLE_CALIBRATION_MEM )
   END_RUNG wire#w2
   RUNG wire#powerrail
      Contact( "DB347_M_UNIT_01_STA_3".M_CODES_UNIT_01_STA_3.M143 )
   END_RUNG wire#w2
   // the same network as SCL:
   "DB2108_UNIT_1_STATION_3_LIGHT"(GENERAL_MACHINE_LIGHT_OPTION := "M_ZERO",   // "FB2107_LIGHTS"
                           CIRCUIT_BRAKER_IN := "DB2103_ELECTRICAL_CABINET".INPUT_CIRCUIT_BREAKER_TRIPPED_LIGHT_STA_3,
                           LIGHT_ON_SELECTOR := "M_ZERO",
                           MANUAL_REQ_LINE := "LTLP_DirectKeyGetMovNoData".PowerUp[30],
                           SWITCH_ON_AUTO_REQ := NOT (NOT "DB1101_MACHINE_SEQUENCE".RUNNING AND NOT "DB1201_PART_CYCLE_UNIT_1".SEQUENCE.RUNNING AND NOT "DB1205_UNIT_1_STATION_3_CYCLE".SEQUENCE.RUNNING AND NOT "DB347_M_UNIT_01_STA_3".M_CODES_UNIT_01_STA_3.M142),
                           SWITCH_OFF_AUTO_REQ := (NOT "DB1101_MACHINE_SEQUENCE".RUNNING AND NOT "DB1201_PART_CYCLE_UNIT_1".SEQUENCE.RUNNING AND NOT "DB1205_UNIT_1_STATION_3_CYCLE".SEQUENCE.RUNNING AND NOT "DB1237_UNIT_1_STATION_3_CAM_NOZZLE_CALIBRATION".SEQUENCE.RUNNING AND NOT "DB16010_MEASURE_SENSORS_CALIBRATION_STATUS".UNIT_1_AUX.DOOR_OPEN_NOZZLE_CALIBRATION_MEM) OR "DB347_M_UNIT_01_STA_3".M_CODES_UNIT_01_STA_3.M143,
                           LIGHTS_ON => "STATION_3_LIGHT_U01_Q",
                           HMI_LINE_ON_EXEC => "LTLP_HMIProInterfaceData".powerup30ExecutableRight,
                           HMI_LINE_OFF_EXEC => "LTLP_HMIProInterfaceData".powerup30ExecutableLeft,
                           HMI_LINE_ON_STATUS => "LTLP_HMIProInterfaceData".powerupCondOn30,
                           HMI_LINE_OFF_STATUS => "LTLP_HMIProInterfaceData".powerupCondOff30);
END_REGION

REGION Network 3: UNIT 2 STATION 3 LIGHT
   RUNG wire#powerrail
      "DB2109_UNIT_2_STATION_3_LIGHT"(SWITCH_ON_AUTO_REQ := wire#w1, SWITCH_OFF_AUTO_REQ := wire#w2, GENERAL_MACHINE_LIGHT_OPTION := "M_ZERO", CIRCUIT_BRAKER_IN := "DB2103_ELECTRICAL_CABINET".INPUT_CIRCUIT_BREAKER_TRIPPED_LIGHT_STA_3, LIGHT_ON_SELECTOR := "M_ZERO", MANUAL_REQ_LINE := "LTLP_DirectKeyGetMovNoData".PowerUp[31], LIGHTS_ON => "STATION_3_LIGHT_U02_Q", HMI_LINE_ON_EXEC => "LTLP_HMIProInterfaceData".powerup31ExecutableRight, HMI_LINE_OFF_EXEC => "LTLP_HMIProInterfaceData".powerup31ExecutableLeft, HMI_LINE_ON_STATUS => "LTLP_HMIProInterfaceData".powerupCondOn31, HMI_LINE_OFF_STATUS => "LTLP_HMIProInterfaceData".powerupCondOff31)
   END_RUNG
   RUNG wire#powerrail
      I_Contact( "DB1101_MACHINE_SEQUENCE".RUNNING )
      I_Contact( "DB1251_PART_CYCLE_UNIT_2".SEQUENCE.RUNNING )
      I_Contact( "DB1255_UNIT_2_STATION_3_CYCLE".SEQUENCE.RUNNING )
      I_Contact( "DB362_M_UNIT_02_STA_3".M_CODES_UNIT_02_STA_3.M142 )
      Not()
   END_RUNG wire#w1
   RUNG wire#powerrail
      I_Contact( "DB1101_MACHINE_SEQUENCE".RUNNING )
      I_Contact( "DB1251_PART_CYCLE_UNIT_2".SEQUENCE.RUNNING )
      I_Contact( "DB1255_UNIT_2_STATION_3_CYCLE".SEQUENCE.RUNNING )
      I_Contact( "DB1277_UNIT_2_STATION_3_CAM_NOZZLE_CALIBRATION".SEQUENCE.RUNNING )
      I_Contact( "DB16010_MEASURE_SENSORS_CALIBRATION_STATUS".UNIT_2_AUX.STATION_3.DOOR_OPEN_NOZZLE_CALIBRATION_MEM )
   END_RUNG wire#w2
   RUNG wire#powerrail
      Contact( "DB362_M_UNIT_02_STA_3".M_CODES_UNIT_02_STA_3.Ack_M143 )
   END_RUNG wire#w2
   // the same network as SCL:
   "DB2109_UNIT_2_STATION_3_LIGHT"(GENERAL_MACHINE_LIGHT_OPTION := "M_ZERO",   // "FB2107_LIGHTS"
                           CIRCUIT_BRAKER_IN := "DB2103_ELECTRICAL_CABINET".INPUT_CIRCUIT_BREAKER_TRIPPED_LIGHT_STA_3,
                           LIGHT_ON_SELECTOR := "M_ZERO",
                           MANUAL_REQ_LINE := "LTLP_DirectKeyGetMovNoData".PowerUp[31],
                           SWITCH_ON_AUTO_REQ := NOT (NOT "DB1101_MACHINE_SEQUENCE".RUNNING AND NOT "DB1251_PART_CYCLE_UNIT_2".SEQUENCE.RUNNING AND NOT "DB1255_UNIT_2_STATION_3_CYCLE".SEQUENCE.RUNNING AND NOT "DB362_M_UNIT_02_STA_3".M_CODES_UNIT_02_STA_3.M142),
                           SWITCH_OFF_AUTO_REQ := (NOT "DB1101_MACHINE_SEQUENCE".RUNNING AND NOT "DB1251_PART_CYCLE_UNIT_2".SEQUENCE.RUNNING AND NOT "DB1255_UNIT_2_STATION_3_CYCLE".SEQUENCE.RUNNING AND NOT "DB1277_UNIT_2_STATION_3_CAM_NOZZLE_CALIBRATION".SEQUENCE.RUNNING AND NOT "DB16010_MEASURE_SENSORS_CALIBRATION_STATUS".UNIT_2_AUX.STATION_3.DOOR_OPEN_NOZZLE_CALIBRATION_MEM) OR "DB362_M_UNIT_02_STA_3".M_CODES_UNIT_02_STA_3.Ack_M143,
                           LIGHTS_ON => "STATION_3_LIGHT_U02_Q",
                           HMI_LINE_ON_EXEC => "LTLP_HMIProInterfaceData".powerup31ExecutableRight,
                           HMI_LINE_OFF_EXEC => "LTLP_HMIProInterfaceData".powerup31ExecutableLeft,
                           HMI_LINE_ON_STATUS => "LTLP_HMIProInterfaceData".powerupCondOn31,
                           HMI_LINE_OFF_STATUS => "LTLP_HMIProInterfaceData".powerupCondOff31);
END_REGION
END_FUNCTION

FUNCTION "FC2108_MACHINE_CONTROL_ON" : Void   // FC2108, LAD
{ S7_Optimized_Access := 'FALSE' }
AUTHOR : ETXETAR
VERSION : 1.0
// stored: AutoNumber false, IsIECCheckEnabled false, SetENOAutomatically false, UDAEnableTagReadback false
   VAR_TEMP
      O_BYTE_0 : Struct   // OPTIONS BYTE 0
         GM_COOLANT_PUMP_OFF_DELAY : Bool;   // GM COOLANT PUMP POWER OFF DELAY OPTION
      END_STRUCT;
   END_VAR
   VAR CONSTANT
      FC_NUMBER : DInt := 2108;   // FC NUMBER
   END_VAR
   VAR_TEMP   // added for the SCL form of the ladder/FBD networks
      _w1 : Bool;
   END_VAR
BEGIN

REGION Network 1: OPTIONS
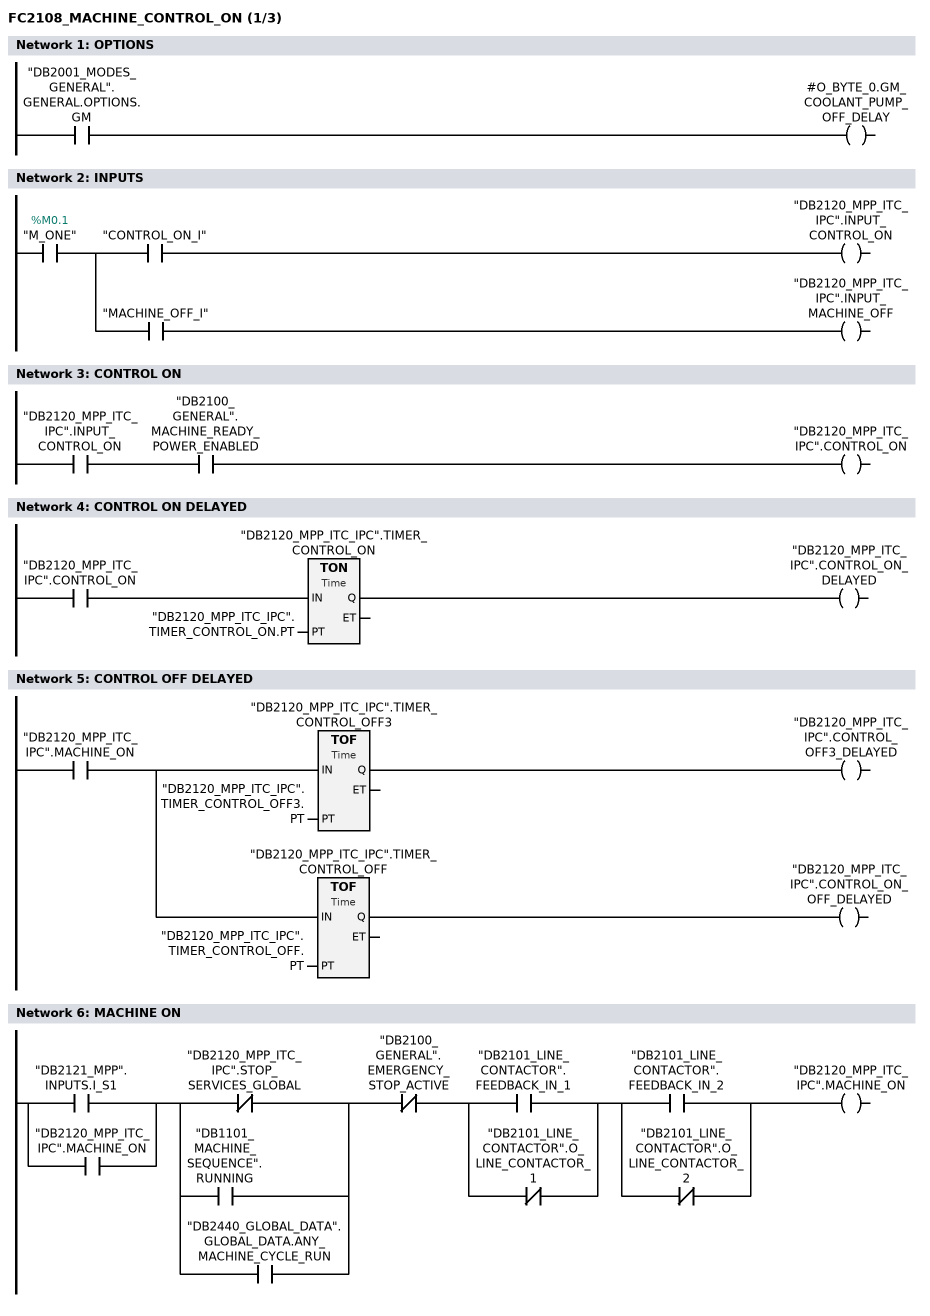
   RUNG wire#powerrail
      Contact( "DB2001_MODES_GENERAL".GENERAL.OPTIONS.GM )
      Coil( #O_BYTE_0.GM_COOLANT_PUMP_OFF_DELAY )
   END_RUNG
   // the same network as SCL:
   #O_BYTE_0.GM_COOLANT_PUMP_OFF_DELAY := "DB2001_MODES_GENERAL".GENERAL.OPTIONS.GM;
END_REGION

REGION Network 2: INPUTS
   RUNG wire#powerrail
      Contact( "M_ONE" )
      wire#w1
      Contact( "CONTROL_ON_I" )
      Coil( "DB2120_MPP_ITC_IPC".INPUT_CONTROL_ON )
   END_RUNG
   RUNG wire#w1
      Contact( "MACHINE_OFF_I" )
      Coil( "DB2120_MPP_ITC_IPC".INPUT_MACHINE_OFF )
   END_RUNG
   // the same network as SCL:
   "DB2120_MPP_ITC_IPC".INPUT_CONTROL_ON := "M_ONE" AND "CONTROL_ON_I";
   "DB2120_MPP_ITC_IPC".INPUT_MACHINE_OFF := "M_ONE" AND "MACHINE_OFF_I";
END_REGION

REGION Network 3: CONTROL ON
   RUNG wire#powerrail
      Contact( "DB2120_MPP_ITC_IPC".INPUT_CONTROL_ON )
      Contact( "DB2100_GENERAL".MACHINE_READY_POWER_ENABLED )
      Coil( "DB2120_MPP_ITC_IPC".CONTROL_ON )
   END_RUNG
   // the same network as SCL:
   "DB2120_MPP_ITC_IPC".CONTROL_ON := "DB2120_MPP_ITC_IPC".INPUT_CONTROL_ON AND "DB2100_GENERAL".MACHINE_READY_POWER_ENABLED;
END_REGION

REGION Network 4: CONTROL ON DELAYED
   RUNG wire#powerrail
      Contact( "DB2120_MPP_ITC_IPC".CONTROL_ON )
      { S7_Templates := "time_type := Time" } "DB2120_MPP_ITC_IPC".TIMER_CONTROL_ON.TON(pt := "DB2120_MPP_ITC_IPC".TIMER_CONTROL_ON.PT, et =>)
      Coil( "DB2120_MPP_ITC_IPC".CONTROL_ON_DELAYED )
   END_RUNG
   // the same network as SCL:
   "DB2120_MPP_ITC_IPC".TIMER_CONTROL_ON.TON(IN := "DB2120_MPP_ITC_IPC".CONTROL_ON,
                           PT := "DB2120_MPP_ITC_IPC".TIMER_CONTROL_ON.PT);
   "DB2120_MPP_ITC_IPC".CONTROL_ON_DELAYED := "DB2120_MPP_ITC_IPC".TIMER_CONTROL_ON.Q;
END_REGION

REGION Network 5: CONTROL OFF DELAYED
   RUNG wire#powerrail
      Contact( "DB2120_MPP_ITC_IPC".MACHINE_ON )
      wire#w1
      { S7_Templates := "time_type := Time" } "DB2120_MPP_ITC_IPC".TIMER_CONTROL_OFF3.TOF(pt := "DB2120_MPP_ITC_IPC".TIMER_CONTROL_OFF3.PT, et =>)
      Coil( "DB2120_MPP_ITC_IPC".CONTROL_OFF3_DELAYED )
   END_RUNG
   RUNG wire#w1
      { S7_Templates := "time_type := Time" } "DB2120_MPP_ITC_IPC".TIMER_CONTROL_OFF.TOF(pt := "DB2120_MPP_ITC_IPC".TIMER_CONTROL_OFF.PT, et =>)
      Coil( "DB2120_MPP_ITC_IPC".CONTROL_ON_OFF_DELAYED )
   END_RUNG
   // the same network as SCL:
   "DB2120_MPP_ITC_IPC".TIMER_CONTROL_OFF3.TOF(IN := "DB2120_MPP_ITC_IPC".MACHINE_ON,
                           PT := "DB2120_MPP_ITC_IPC".TIMER_CONTROL_OFF3.PT);
   "DB2120_MPP_ITC_IPC".CONTROL_OFF3_DELAYED := "DB2120_MPP_ITC_IPC".TIMER_CONTROL_OFF3.Q;
   "DB2120_MPP_ITC_IPC".TIMER_CONTROL_OFF.TOF(IN := "DB2120_MPP_ITC_IPC".MACHINE_ON,
                           PT := "DB2120_MPP_ITC_IPC".TIMER_CONTROL_OFF.PT);
   "DB2120_MPP_ITC_IPC".CONTROL_ON_OFF_DELAYED := "DB2120_MPP_ITC_IPC".TIMER_CONTROL_OFF.Q;
END_REGION

REGION Network 6: MACHINE ON
   RUNG wire#powerrail
      Contact( "DB2121_MPP".INPUTS.I_S1 )
      wire#w1
      I_Contact( "DB2120_MPP_ITC_IPC".STOP_SERVICES_GLOBAL )
      wire#w2
      I_Contact( "DB2100_GENERAL".EMERGENCY_STOP_ACTIVE )
      wire#w3
      Contact( "DB2101_LINE_CONTACTOR".FEEDBACK_IN_1 )
      wire#w4
      Contact( "DB2101_LINE_CONTACTOR".FEEDBACK_IN_2 )
      wire#w5
      Coil( "DB2120_MPP_ITC_IPC".MACHINE_ON )
   END_RUNG
   RUNG wire#powerrail
      Contact( "DB2120_MPP_ITC_IPC".MACHINE_ON )
   END_RUNG wire#w1
   RUNG wire#w1
      Contact( "DB1101_MACHINE_SEQUENCE".RUNNING )
   END_RUNG wire#w2
   RUNG wire#w1
      Contact( "DB2440_GLOBAL_DATA".GLOBAL_DATA.ANY_MACHINE_CYCLE_RUN )
   END_RUNG wire#w2
   RUNG wire#w3
      I_Contact( "DB2101_LINE_CONTACTOR".O_LINE_CONTACTOR_1 )
   END_RUNG wire#w4
   RUNG wire#w4
      I_Contact( "DB2101_LINE_CONTACTOR".O_LINE_CONTACTOR_2 )
   END_RUNG wire#w5
   // the same network as SCL:
   "DB2120_MPP_ITC_IPC".MACHINE_ON := ("DB2121_MPP".INPUTS.I_S1 OR "DB2120_MPP_ITC_IPC".MACHINE_ON) AND (NOT "DB2120_MPP_ITC_IPC".STOP_SERVICES_GLOBAL OR "DB1101_MACHINE_SEQUENCE".RUNNING OR "DB2440_GLOBAL_DATA".GLOBAL_DATA.ANY_MACHINE_CYCLE_RUN) AND NOT "DB2100_GENERAL".EMERGENCY_STOP_ACTIVE AND ("DB2101_LINE_CONTACTOR".FEEDBACK_IN_1 OR NOT "DB2101_LINE_CONTACTOR".O_LINE_CONTACTOR_1) AND ("DB2101_LINE_CONTACTOR".FEEDBACK_IN_2 OR NOT "DB2101_LINE_CONTACTOR".O_LINE_CONTACTOR_2);
END_REGION

REGION Network 7: MACHINE ON DELAYED
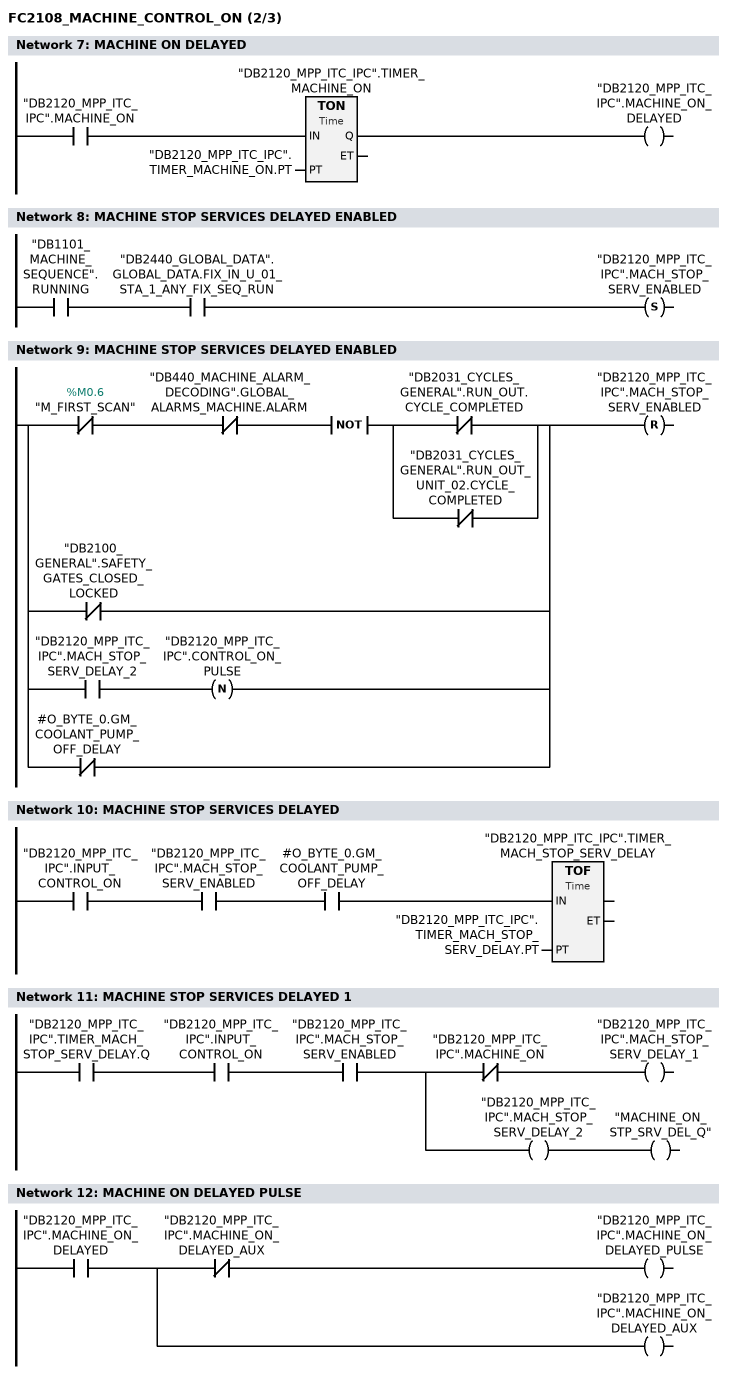
   RUNG wire#powerrail
      Contact( "DB2120_MPP_ITC_IPC".MACHINE_ON )
      { S7_Templates := "time_type := Time" } "DB2120_MPP_ITC_IPC".TIMER_MACHINE_ON.TON(pt := "DB2120_MPP_ITC_IPC".TIMER_MACHINE_ON.PT, et =>)
      Coil( "DB2120_MPP_ITC_IPC".MACHINE_ON_DELAYED )
   END_RUNG
   // the same network as SCL:
   "DB2120_MPP_ITC_IPC".TIMER_MACHINE_ON.TON(IN := "DB2120_MPP_ITC_IPC".MACHINE_ON,
                           PT := "DB2120_MPP_ITC_IPC".TIMER_MACHINE_ON.PT);
   "DB2120_MPP_ITC_IPC".MACHINE_ON_DELAYED := "DB2120_MPP_ITC_IPC".TIMER_MACHINE_ON.Q;
END_REGION

REGION Network 8: MACHINE STOP SERVICES DELAYED ENABLED
   RUNG wire#powerrail
      Contact( "DB1101_MACHINE_SEQUENCE".RUNNING )
      Contact( "DB2440_GLOBAL_DATA".GLOBAL_DATA.FIX_IN_U_01_STA_1_ANY_FIX_SEQ_RUN )
      S_Coil( "DB2120_MPP_ITC_IPC".MACH_STOP_SERV_ENABLED )
   END_RUNG
   // the same network as SCL:
   IF "DB1101_MACHINE_SEQUENCE".RUNNING AND "DB2440_GLOBAL_DATA".GLOBAL_DATA.FIX_IN_U_01_STA_1_ANY_FIX_SEQ_RUN THEN
       "DB2120_MPP_ITC_IPC".MACH_STOP_SERV_ENABLED := TRUE;
   END_IF;
END_REGION

REGION Network 9: MACHINE STOP SERVICES DELAYED ENABLED
   RUNG wire#powerrail
      I_Contact( "M_FIRST_SCAN" )
      I_Contact( "DB440_MACHINE_ALARM_DECODING".GLOBAL_ALARMS_MACHINE.ALARM )
      Not()
      wire#w1
      I_Contact( "DB2031_CYCLES_GENERAL".RUN_OUT.CYCLE_COMPLETED )
      wire#w2
      R_Coil( "DB2120_MPP_ITC_IPC".MACH_STOP_SERV_ENABLED )
   END_RUNG
   RUNG wire#w1
      I_Contact( "DB2031_CYCLES_GENERAL".RUN_OUT_UNIT_02.CYCLE_COMPLETED )
   END_RUNG wire#w2
   RUNG wire#powerrail
      I_Contact( "DB2100_GENERAL".SAFETY_GATES_CLOSED_LOCKED )
   END_RUNG wire#w2
   RUNG wire#powerrail
      Contact( "DB2120_MPP_ITC_IPC".MACH_STOP_SERV_DELAY_2 )
      N_Trig( "DB2120_MPP_ITC_IPC".CONTROL_ON_PULSE )
   END_RUNG wire#w2
   RUNG wire#powerrail
      I_Contact( #O_BYTE_0.GM_COOLANT_PUMP_OFF_DELAY )
   END_RUNG wire#w2
   // the same network as SCL:
   #_w1 := NOT "DB2120_MPP_ITC_IPC".MACH_STOP_SERV_DELAY_2 AND "DB2120_MPP_ITC_IPC".CONTROL_ON_PULSE;   // falling edge
   "DB2120_MPP_ITC_IPC".CONTROL_ON_PULSE := "DB2120_MPP_ITC_IPC".MACH_STOP_SERV_DELAY_2;
   IF (NOT (NOT "M_FIRST_SCAN" AND NOT "DB440_MACHINE_ALARM_DECODING".GLOBAL_ALARMS_MACHINE.ALARM) AND (NOT "DB2031_CYCLES_GENERAL".RUN_OUT.CYCLE_COMPLETED OR NOT "DB2031_CYCLES_GENERAL".RUN_OUT_UNIT_02.CYCLE_COMPLETED)) OR NOT "DB2100_GENERAL".SAFETY_GATES_CLOSED_LOCKED OR #_w1 OR NOT #O_BYTE_0.GM_COOLANT_PUMP_OFF_DELAY THEN
       "DB2120_MPP_ITC_IPC".MACH_STOP_SERV_ENABLED := FALSE;
   END_IF;
END_REGION

REGION Network 10: MACHINE STOP SERVICES DELAYED
   RUNG wire#powerrail
      Contact( "DB2120_MPP_ITC_IPC".INPUT_CONTROL_ON )
      Contact( "DB2120_MPP_ITC_IPC".MACH_STOP_SERV_ENABLED )
      Contact( #O_BYTE_0.GM_COOLANT_PUMP_OFF_DELAY )
      { S7_Templates := "time_type := Time" } "DB2120_MPP_ITC_IPC".TIMER_MACH_STOP_SERV_DELAY.TOF(pt := "DB2120_MPP_ITC_IPC".TIMER_MACH_STOP_SERV_DELAY.PT, et =>)
   END_RUNG
   // the same network as SCL:
   "DB2120_MPP_ITC_IPC".TIMER_MACH_STOP_SERV_DELAY.TOF(IN := "DB2120_MPP_ITC_IPC".INPUT_CONTROL_ON AND "DB2120_MPP_ITC_IPC".MACH_STOP_SERV_ENABLED AND #O_BYTE_0.GM_COOLANT_PUMP_OFF_DELAY,
                           PT := "DB2120_MPP_ITC_IPC".TIMER_MACH_STOP_SERV_DELAY.PT);
END_REGION

REGION Network 11: MACHINE STOP SERVICES DELAYED 1
   RUNG wire#powerrail
      Contact( "DB2120_MPP_ITC_IPC".TIMER_MACH_STOP_SERV_DELAY.Q )
      Contact( "DB2120_MPP_ITC_IPC".INPUT_CONTROL_ON )
      Contact( "DB2120_MPP_ITC_IPC".MACH_STOP_SERV_ENABLED )
      wire#w1
      I_Contact( "DB2120_MPP_ITC_IPC".MACHINE_ON )
      Coil( "DB2120_MPP_ITC_IPC".MACH_STOP_SERV_DELAY_1 )
   END_RUNG
   RUNG wire#w1
      Coil( "DB2120_MPP_ITC_IPC".MACH_STOP_SERV_DELAY_2 )
      Coil( "MACHINE_ON_STP_SRV_DEL_Q" )
   END_RUNG
   // the same network as SCL:
   #_w1 := "DB2120_MPP_ITC_IPC".TIMER_MACH_STOP_SERV_DELAY.Q AND "DB2120_MPP_ITC_IPC".INPUT_CONTROL_ON AND "DB2120_MPP_ITC_IPC".MACH_STOP_SERV_ENABLED;
   "DB2120_MPP_ITC_IPC".MACH_STOP_SERV_DELAY_1 := #_w1 AND NOT "DB2120_MPP_ITC_IPC".MACHINE_ON;
   "DB2120_MPP_ITC_IPC".MACH_STOP_SERV_DELAY_2 := #_w1;
   "MACHINE_ON_STP_SRV_DEL_Q" := #_w1;
END_REGION

REGION Network 12: MACHINE ON DELAYED PULSE
   RUNG wire#powerrail
      Contact( "DB2120_MPP_ITC_IPC".MACHINE_ON_DELAYED )
      wire#w1
      I_Contact( "DB2120_MPP_ITC_IPC".MACHINE_ON_DELAYED_AUX )
      Coil( "DB2120_MPP_ITC_IPC".MACHINE_ON_DELAYED_PULSE )
   END_RUNG
   RUNG wire#w1
      Coil( "DB2120_MPP_ITC_IPC".MACHINE_ON_DELAYED_AUX )
   END_RUNG
   // the same network as SCL:
   "DB2120_MPP_ITC_IPC".MACHINE_ON_DELAYED_PULSE := "DB2120_MPP_ITC_IPC".MACHINE_ON_DELAYED AND NOT "DB2120_MPP_ITC_IPC".MACHINE_ON_DELAYED_AUX;
   "DB2120_MPP_ITC_IPC".MACHINE_ON_DELAYED_AUX := "DB2120_MPP_ITC_IPC".MACHINE_ON_DELAYED;
END_REGION

REGION Network 13: MACHINE OFF DELAYED
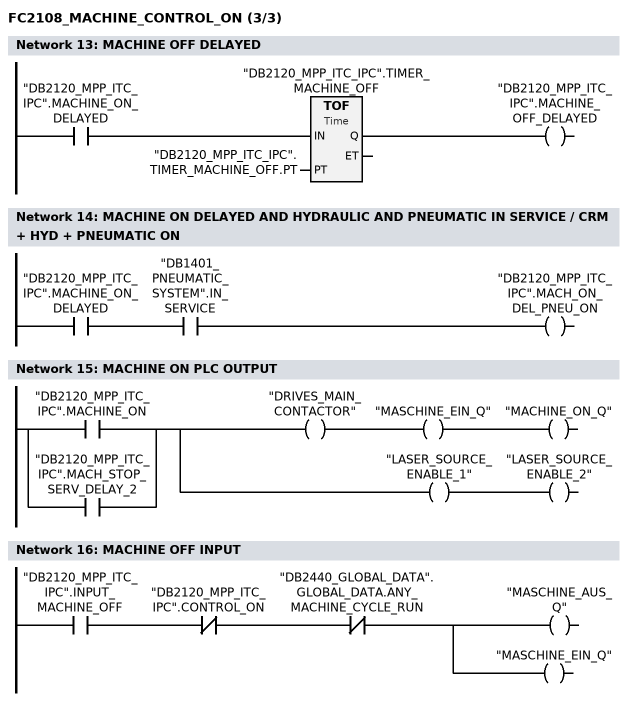
   RUNG wire#powerrail
      Contact( "DB2120_MPP_ITC_IPC".MACHINE_ON_DELAYED )
      { S7_Templates := "time_type := Time" } "DB2120_MPP_ITC_IPC".TIMER_MACHINE_OFF.TOF(pt := "DB2120_MPP_ITC_IPC".TIMER_MACHINE_OFF.PT, et =>)
      Coil( "DB2120_MPP_ITC_IPC".MACHINE_OFF_DELAYED )
   END_RUNG
   // the same network as SCL:
   "DB2120_MPP_ITC_IPC".TIMER_MACHINE_OFF.TOF(IN := "DB2120_MPP_ITC_IPC".MACHINE_ON_DELAYED,
                           PT := "DB2120_MPP_ITC_IPC".TIMER_MACHINE_OFF.PT);
   "DB2120_MPP_ITC_IPC".MACHINE_OFF_DELAYED := "DB2120_MPP_ITC_IPC".TIMER_MACHINE_OFF.Q;
END_REGION

REGION Network 14: MACHINE ON DELAYED AND HYDRAULIC AND PNEUMATIC IN SERVICE / CRM + HYD + PNEUMATIC ON
   RUNG wire#powerrail
      Contact( "DB2120_MPP_ITC_IPC".MACHINE_ON_DELAYED )
      Contact( "DB1401_PNEUMATIC_SYSTEM".IN_SERVICE )
      Coil( "DB2120_MPP_ITC_IPC".MACH_ON_DEL_PNEU_ON )
   END_RUNG
   // the same network as SCL:
   "DB2120_MPP_ITC_IPC".MACH_ON_DEL_PNEU_ON := "DB2120_MPP_ITC_IPC".MACHINE_ON_DELAYED AND "DB1401_PNEUMATIC_SYSTEM".IN_SERVICE;
END_REGION

REGION Network 15: MACHINE ON PLC OUTPUT
   RUNG wire#powerrail
      Contact( "DB2120_MPP_ITC_IPC".MACHINE_ON )
      wire#w1
      Coil( "DRIVES_MAIN_CONTACTOR" )
      Coil( "MASCHINE_EIN_Q" )
      Coil( "MACHINE_ON_Q" )
   END_RUNG
   RUNG wire#powerrail
      Contact( "DB2120_MPP_ITC_IPC".MACH_STOP_SERV_DELAY_2 )
   END_RUNG wire#w1
   RUNG wire#w1
      Coil( "LASER_SOURCE_ENABLE_1" )
      Coil( "LASER_SOURCE_ENABLE_2" )
   END_RUNG
   // the same network as SCL:
   "DRIVES_MAIN_CONTACTOR" := "DB2120_MPP_ITC_IPC".MACHINE_ON OR "DB2120_MPP_ITC_IPC".MACH_STOP_SERV_DELAY_2;
   "MASCHINE_EIN_Q" := "DRIVES_MAIN_CONTACTOR";
   "MACHINE_ON_Q" := "DRIVES_MAIN_CONTACTOR";
   "LASER_SOURCE_ENABLE_1" := "DRIVES_MAIN_CONTACTOR";
   "LASER_SOURCE_ENABLE_2" := "DRIVES_MAIN_CONTACTOR";
END_REGION

REGION Network 16: MACHINE OFF INPUT
   RUNG wire#powerrail
      Contact( "DB2120_MPP_ITC_IPC".INPUT_MACHINE_OFF )
      I_Contact( "DB2120_MPP_ITC_IPC".CONTROL_ON )
      I_Contact( "DB2440_GLOBAL_DATA".GLOBAL_DATA.ANY_MACHINE_CYCLE_RUN )
      wire#w1
      Coil( "MASCHINE_AUS_Q" )
   END_RUNG
   RUNG wire#w1
      Coil( "MASCHINE_EIN_Q" )
   END_RUNG
   // the same network as SCL:
   "MASCHINE_AUS_Q" := "DB2120_MPP_ITC_IPC".INPUT_MACHINE_OFF AND NOT "DB2120_MPP_ITC_IPC".CONTROL_ON AND NOT "DB2440_GLOBAL_DATA".GLOBAL_DATA.ANY_MACHINE_CYCLE_RUN;
   "MASCHINE_EIN_Q" := "MASCHINE_AUS_Q";
END_REGION
END_FUNCTION

FUNCTION "FC2109_STATION_3_LIGHT_U01" : Void   // FC2109, LAD
{ S7_Optimized_Access := 'FALSE' }
AUTHOR : ETXETAR
VERSION : 1.0
// stored: AutoNumber false, IsIECCheckEnabled false, SetENOAutomatically false, UDAEnableTagReadback false
   VAR_TEMP   // added for the SCL form of the ladder/FBD networks
      _w1 : Bool;
   END_VAR
BEGIN

REGION Network 1: INPUTS
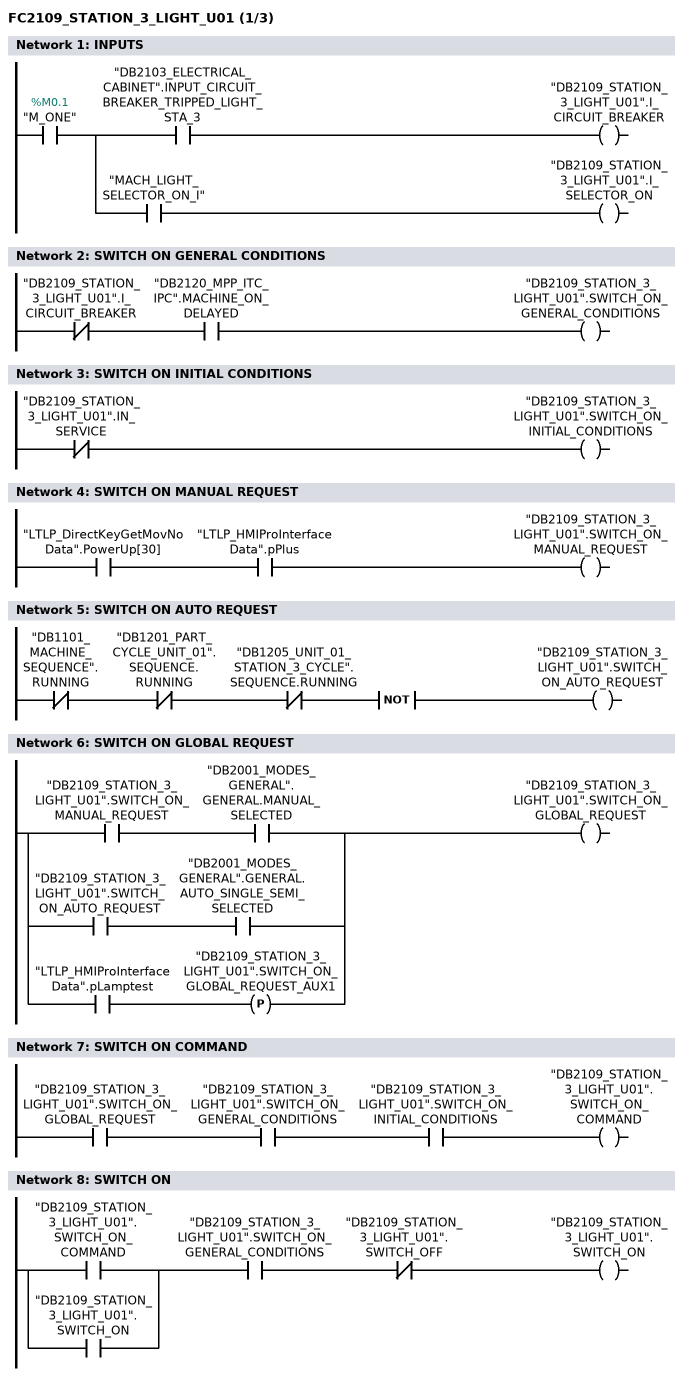
   RUNG wire#powerrail
      Contact( "M_ONE" )
      wire#w1
      Contact( "DB2103_ELECTRICAL_CABINET".INPUT_CIRCUIT_BREAKER_TRIPPED_LIGHT_STA_3 )
      Coil( "DB2109_STATION_3_LIGHT_U01".I_CIRCUIT_BREAKER )
   END_RUNG
   RUNG wire#w1
      Contact( "MACH_LIGHT_SELECTOR_ON_I" )
      Coil( "DB2109_STATION_3_LIGHT_U01".I_SELECTOR_ON )
   END_RUNG
   // the same network as SCL:
   "DB2109_STATION_3_LIGHT_U01".I_CIRCUIT_BREAKER := "M_ONE" AND "DB2103_ELECTRICAL_CABINET".INPUT_CIRCUIT_BREAKER_TRIPPED_LIGHT_STA_3;
   "DB2109_STATION_3_LIGHT_U01".I_SELECTOR_ON := "M_ONE" AND "MACH_LIGHT_SELECTOR_ON_I";
END_REGION

REGION Network 2: SWITCH ON GENERAL CONDITIONS
   RUNG wire#powerrail
      I_Contact( "DB2109_STATION_3_LIGHT_U01".I_CIRCUIT_BREAKER )
      Contact( "DB2120_MPP_ITC_IPC".MACHINE_ON_DELAYED )
      Coil( "DB2109_STATION_3_LIGHT_U01".SWITCH_ON_GENERAL_CONDITIONS )
   END_RUNG
   // the same network as SCL:
   "DB2109_STATION_3_LIGHT_U01".SWITCH_ON_GENERAL_CONDITIONS := NOT "DB2109_STATION_3_LIGHT_U01".I_CIRCUIT_BREAKER AND "DB2120_MPP_ITC_IPC".MACHINE_ON_DELAYED;
END_REGION

REGION Network 3: SWITCH ON INITIAL CONDITIONS
   RUNG wire#powerrail
      I_Contact( "DB2109_STATION_3_LIGHT_U01".IN_SERVICE )
      Coil( "DB2109_STATION_3_LIGHT_U01".SWITCH_ON_INITIAL_CONDITIONS )
   END_RUNG
   // the same network as SCL:
   "DB2109_STATION_3_LIGHT_U01".SWITCH_ON_INITIAL_CONDITIONS := NOT "DB2109_STATION_3_LIGHT_U01".IN_SERVICE;
END_REGION

REGION Network 4: SWITCH ON MANUAL REQUEST
   RUNG wire#powerrail
      Contact( "LTLP_DirectKeyGetMovNoData".PowerUp[30] )
      Contact( "LTLP_HMIProInterfaceData".pPlus )
      Coil( "DB2109_STATION_3_LIGHT_U01".SWITCH_ON_MANUAL_REQUEST )
   END_RUNG
   // the same network as SCL:
   "DB2109_STATION_3_LIGHT_U01".SWITCH_ON_MANUAL_REQUEST := "LTLP_DirectKeyGetMovNoData".PowerUp[30] AND "LTLP_HMIProInterfaceData".pPlus;
END_REGION

REGION Network 5: SWITCH ON AUTO REQUEST
   RUNG wire#powerrail
      I_Contact( "DB1101_MACHINE_SEQUENCE".RUNNING )
      I_Contact( "DB1201_PART_CYCLE_UNIT_01".SEQUENCE.RUNNING )
      I_Contact( "DB1205_UNIT_01_STATION_3_CYCLE".SEQUENCE.RUNNING )
      Not()
      Coil( "DB2109_STATION_3_LIGHT_U01".SWITCH_ON_AUTO_REQUEST )
   END_RUNG
   // the same network as SCL:
   "DB2109_STATION_3_LIGHT_U01".SWITCH_ON_AUTO_REQUEST := NOT (NOT "DB1101_MACHINE_SEQUENCE".RUNNING AND NOT "DB1201_PART_CYCLE_UNIT_01".SEQUENCE.RUNNING AND NOT "DB1205_UNIT_01_STATION_3_CYCLE".SEQUENCE.RUNNING);
END_REGION

REGION Network 6: SWITCH ON GLOBAL REQUEST
   RUNG wire#powerrail
      Contact( "DB2109_STATION_3_LIGHT_U01".SWITCH_ON_MANUAL_REQUEST )
      Contact( "DB2001_MODES_GENERAL".GENERAL.MANUAL_SELECTED )
      wire#w1
      Coil( "DB2109_STATION_3_LIGHT_U01".SWITCH_ON_GLOBAL_REQUEST )
   END_RUNG
   RUNG wire#powerrail
      Contact( "DB2109_STATION_3_LIGHT_U01".SWITCH_ON_AUTO_REQUEST )
      Contact( "DB2001_MODES_GENERAL".GENERAL.AUTO_SINGLE_SEMI_SELECTED )
   END_RUNG wire#w1
   RUNG wire#powerrail
      Contact( "LTLP_HMIProInterfaceData".pLamptest )
      P_Trig( "DB2109_STATION_3_LIGHT_U01".SWITCH_ON_GLOBAL_REQUEST_AUX1 )
   END_RUNG wire#w1
   // the same network as SCL:
   #_w1 := "LTLP_HMIProInterfaceData".pLamptest AND NOT "DB2109_STATION_3_LIGHT_U01".SWITCH_ON_GLOBAL_REQUEST_AUX1;   // rising edge
   "DB2109_STATION_3_LIGHT_U01".SWITCH_ON_GLOBAL_REQUEST_AUX1 := "LTLP_HMIProInterfaceData".pLamptest;
   "DB2109_STATION_3_LIGHT_U01".SWITCH_ON_GLOBAL_REQUEST := ("DB2109_STATION_3_LIGHT_U01".SWITCH_ON_MANUAL_REQUEST AND "DB2001_MODES_GENERAL".GENERAL.MANUAL_SELECTED) OR ("DB2109_STATION_3_LIGHT_U01".SWITCH_ON_AUTO_REQUEST AND "DB2001_MODES_GENERAL".GENERAL.AUTO_SINGLE_SEMI_SELECTED) OR #_w1;
END_REGION

REGION Network 7: SWITCH ON COMMAND
   RUNG wire#powerrail
      Contact( "DB2109_STATION_3_LIGHT_U01".SWITCH_ON_GLOBAL_REQUEST )
      Contact( "DB2109_STATION_3_LIGHT_U01".SWITCH_ON_GENERAL_CONDITIONS )
      Contact( "DB2109_STATION_3_LIGHT_U01".SWITCH_ON_INITIAL_CONDITIONS )
      Coil( "DB2109_STATION_3_LIGHT_U01".SWITCH_ON_COMMAND )
   END_RUNG
   // the same network as SCL:
   "DB2109_STATION_3_LIGHT_U01".SWITCH_ON_COMMAND := "DB2109_STATION_3_LIGHT_U01".SWITCH_ON_GLOBAL_REQUEST AND "DB2109_STATION_3_LIGHT_U01".SWITCH_ON_GENERAL_CONDITIONS AND "DB2109_STATION_3_LIGHT_U01".SWITCH_ON_INITIAL_CONDITIONS;
END_REGION

REGION Network 8: SWITCH ON
   RUNG wire#powerrail
      Contact( "DB2109_STATION_3_LIGHT_U01".SWITCH_ON_COMMAND )
      wire#w1
      Contact( "DB2109_STATION_3_LIGHT_U01".SWITCH_ON_GENERAL_CONDITIONS )
      I_Contact( "DB2109_STATION_3_LIGHT_U01".SWITCH_OFF )
      Coil( "DB2109_STATION_3_LIGHT_U01".SWITCH_ON )
   END_RUNG
   RUNG wire#powerrail
      Contact( "DB2109_STATION_3_LIGHT_U01".SWITCH_ON )
   END_RUNG wire#w1
   // the same network as SCL:
   "DB2109_STATION_3_LIGHT_U01".SWITCH_ON := ("DB2109_STATION_3_LIGHT_U01".SWITCH_ON_COMMAND OR "DB2109_STATION_3_LIGHT_U01".SWITCH_ON) AND "DB2109_STATION_3_LIGHT_U01".SWITCH_ON_GENERAL_CONDITIONS AND NOT "DB2109_STATION_3_LIGHT_U01".SWITCH_OFF;
END_REGION

REGION Network 9: IN SERVICE
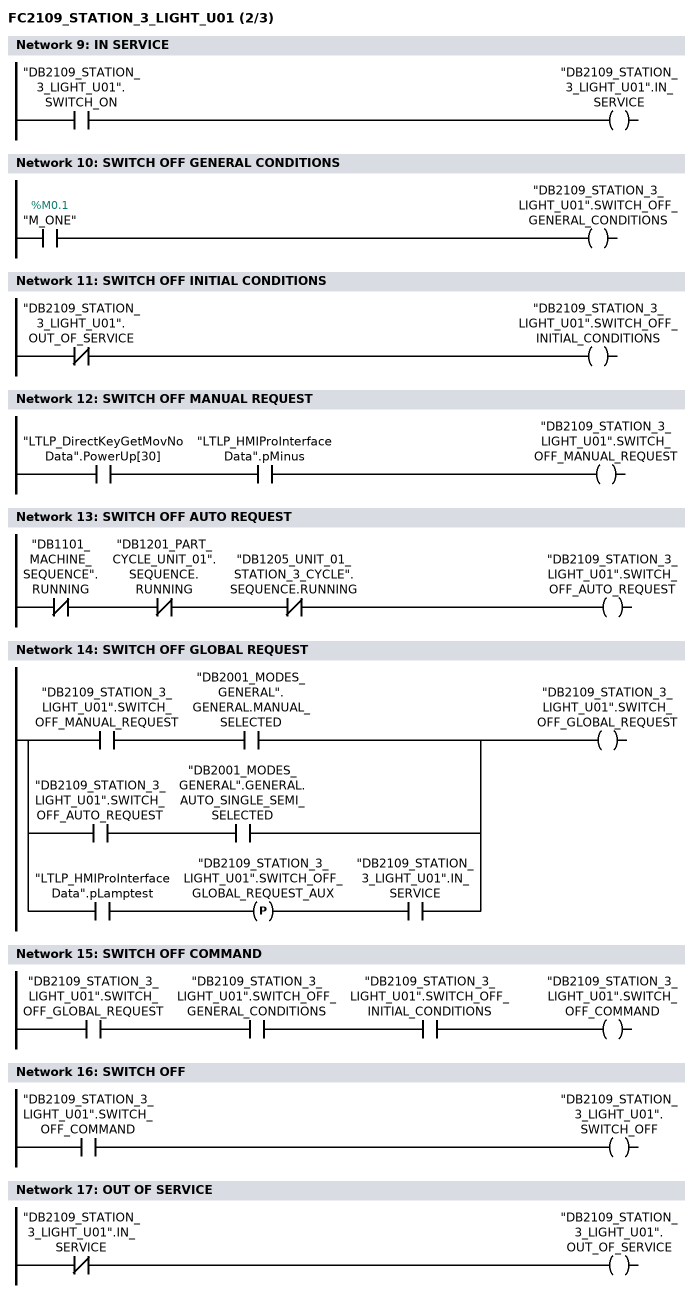
   RUNG wire#powerrail
      Contact( "DB2109_STATION_3_LIGHT_U01".SWITCH_ON )
      Coil( "DB2109_STATION_3_LIGHT_U01".IN_SERVICE )
   END_RUNG
   // the same network as SCL:
   "DB2109_STATION_3_LIGHT_U01".IN_SERVICE := "DB2109_STATION_3_LIGHT_U01".SWITCH_ON;
END_REGION

REGION Network 10: SWITCH OFF GENERAL CONDITIONS
   RUNG wire#powerrail
      Contact( "M_ONE" )
      Coil( "DB2109_STATION_3_LIGHT_U01".SWITCH_OFF_GENERAL_CONDITIONS )
   END_RUNG
   // the same network as SCL:
   "DB2109_STATION_3_LIGHT_U01".SWITCH_OFF_GENERAL_CONDITIONS := "M_ONE";
END_REGION

REGION Network 11: SWITCH OFF INITIAL CONDITIONS
   RUNG wire#powerrail
      I_Contact( "DB2109_STATION_3_LIGHT_U01".OUT_OF_SERVICE )
      Coil( "DB2109_STATION_3_LIGHT_U01".SWITCH_OFF_INITIAL_CONDITIONS )
   END_RUNG
   // the same network as SCL:
   "DB2109_STATION_3_LIGHT_U01".SWITCH_OFF_INITIAL_CONDITIONS := NOT "DB2109_STATION_3_LIGHT_U01".OUT_OF_SERVICE;
END_REGION

REGION Network 12: SWITCH OFF MANUAL REQUEST
   RUNG wire#powerrail
      Contact( "LTLP_DirectKeyGetMovNoData".PowerUp[30] )
      Contact( "LTLP_HMIProInterfaceData".pMinus )
      Coil( "DB2109_STATION_3_LIGHT_U01".SWITCH_OFF_MANUAL_REQUEST )
   END_RUNG
   // the same network as SCL:
   "DB2109_STATION_3_LIGHT_U01".SWITCH_OFF_MANUAL_REQUEST := "LTLP_DirectKeyGetMovNoData".PowerUp[30] AND "LTLP_HMIProInterfaceData".pMinus;
END_REGION

REGION Network 13: SWITCH OFF AUTO REQUEST
   RUNG wire#powerrail
      I_Contact( "DB1101_MACHINE_SEQUENCE".RUNNING )
      I_Contact( "DB1201_PART_CYCLE_UNIT_01".SEQUENCE.RUNNING )
      I_Contact( "DB1205_UNIT_01_STATION_3_CYCLE".SEQUENCE.RUNNING )
      Coil( "DB2109_STATION_3_LIGHT_U01".SWITCH_OFF_AUTO_REQUEST )
   END_RUNG
   // the same network as SCL:
   "DB2109_STATION_3_LIGHT_U01".SWITCH_OFF_AUTO_REQUEST := NOT "DB1101_MACHINE_SEQUENCE".RUNNING AND NOT "DB1201_PART_CYCLE_UNIT_01".SEQUENCE.RUNNING AND NOT "DB1205_UNIT_01_STATION_3_CYCLE".SEQUENCE.RUNNING;
END_REGION

REGION Network 14: SWITCH OFF GLOBAL REQUEST
   RUNG wire#powerrail
      Contact( "DB2109_STATION_3_LIGHT_U01".SWITCH_OFF_MANUAL_REQUEST )
      Contact( "DB2001_MODES_GENERAL".GENERAL.MANUAL_SELECTED )
      wire#w1
      Coil( "DB2109_STATION_3_LIGHT_U01".SWITCH_OFF_GLOBAL_REQUEST )
   END_RUNG
   RUNG wire#powerrail
      Contact( "DB2109_STATION_3_LIGHT_U01".SWITCH_OFF_AUTO_REQUEST )
      Contact( "DB2001_MODES_GENERAL".GENERAL.AUTO_SINGLE_SEMI_SELECTED )
   END_RUNG wire#w1
   RUNG wire#powerrail
      Contact( "LTLP_HMIProInterfaceData".pLamptest )
      P_Trig( "DB2109_STATION_3_LIGHT_U01".SWITCH_OFF_GLOBAL_REQUEST_AUX )
      Contact( "DB2109_STATION_3_LIGHT_U01".IN_SERVICE )
   END_RUNG wire#w1
   // the same network as SCL:
   #_w1 := "LTLP_HMIProInterfaceData".pLamptest AND NOT "DB2109_STATION_3_LIGHT_U01".SWITCH_OFF_GLOBAL_REQUEST_AUX;   // rising edge
   "DB2109_STATION_3_LIGHT_U01".SWITCH_OFF_GLOBAL_REQUEST_AUX := "LTLP_HMIProInterfaceData".pLamptest;
   "DB2109_STATION_3_LIGHT_U01".SWITCH_OFF_GLOBAL_REQUEST := ("DB2109_STATION_3_LIGHT_U01".SWITCH_OFF_MANUAL_REQUEST AND "DB2001_MODES_GENERAL".GENERAL.MANUAL_SELECTED) OR ("DB2109_STATION_3_LIGHT_U01".SWITCH_OFF_AUTO_REQUEST AND "DB2001_MODES_GENERAL".GENERAL.AUTO_SINGLE_SEMI_SELECTED) OR (#_w1 AND "DB2109_STATION_3_LIGHT_U01".IN_SERVICE);
END_REGION

REGION Network 15: SWITCH OFF COMMAND
   RUNG wire#powerrail
      Contact( "DB2109_STATION_3_LIGHT_U01".SWITCH_OFF_GLOBAL_REQUEST )
      Contact( "DB2109_STATION_3_LIGHT_U01".SWITCH_OFF_GENERAL_CONDITIONS )
      Contact( "DB2109_STATION_3_LIGHT_U01".SWITCH_OFF_INITIAL_CONDITIONS )
      Coil( "DB2109_STATION_3_LIGHT_U01".SWITCH_OFF_COMMAND )
   END_RUNG
   // the same network as SCL:
   "DB2109_STATION_3_LIGHT_U01".SWITCH_OFF_COMMAND := "DB2109_STATION_3_LIGHT_U01".SWITCH_OFF_GLOBAL_REQUEST AND "DB2109_STATION_3_LIGHT_U01".SWITCH_OFF_GENERAL_CONDITIONS AND "DB2109_STATION_3_LIGHT_U01".SWITCH_OFF_INITIAL_CONDITIONS;
END_REGION

REGION Network 16: SWITCH OFF
   RUNG wire#powerrail
      Contact( "DB2109_STATION_3_LIGHT_U01".SWITCH_OFF_COMMAND )
      Coil( "DB2109_STATION_3_LIGHT_U01".SWITCH_OFF )
   END_RUNG
   // the same network as SCL:
   "DB2109_STATION_3_LIGHT_U01".SWITCH_OFF := "DB2109_STATION_3_LIGHT_U01".SWITCH_OFF_COMMAND;
END_REGION

REGION Network 17: OUT OF SERVICE
   RUNG wire#powerrail
      I_Contact( "DB2109_STATION_3_LIGHT_U01".IN_SERVICE )
      Coil( "DB2109_STATION_3_LIGHT_U01".OUT_OF_SERVICE )
   END_RUNG
   // the same network as SCL:
   "DB2109_STATION_3_LIGHT_U01".OUT_OF_SERVICE := NOT "DB2109_STATION_3_LIGHT_U01".IN_SERVICE;
END_REGION

REGION Network 18: HMI STATUS
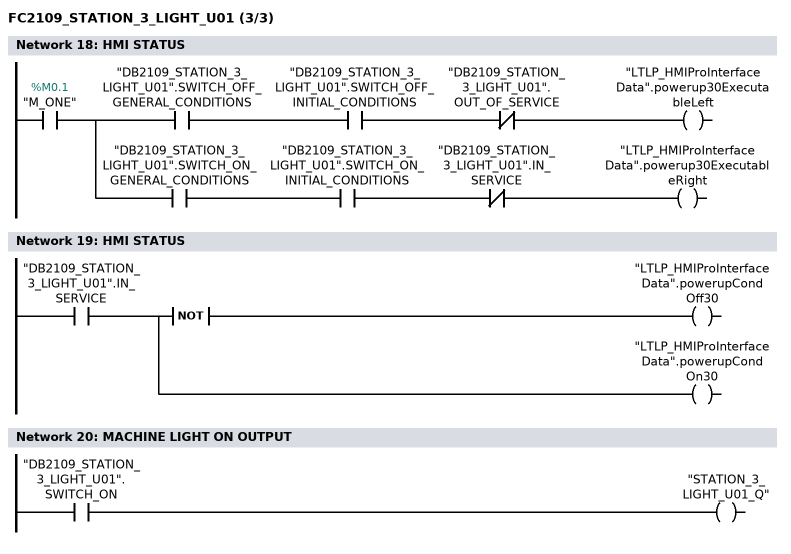
   RUNG wire#powerrail
      Contact( "M_ONE" )
      wire#w1
      Contact( "DB2109_STATION_3_LIGHT_U01".SWITCH_OFF_GENERAL_CONDITIONS )
      Contact( "DB2109_STATION_3_LIGHT_U01".SWITCH_OFF_INITIAL_CONDITIONS )
      I_Contact( "DB2109_STATION_3_LIGHT_U01".OUT_OF_SERVICE )
      Coil( "LTLP_HMIProInterfaceData".powerup30ExecutableLeft )
   END_RUNG
   RUNG wire#w1
      Contact( "DB2109_STATION_3_LIGHT_U01".SWITCH_ON_GENERAL_CONDITIONS )
      Contact( "DB2109_STATION_3_LIGHT_U01".SWITCH_ON_INITIAL_CONDITIONS )
      I_Contact( "DB2109_STATION_3_LIGHT_U01".IN_SERVICE )
      Coil( "LTLP_HMIProInterfaceData".powerup30ExecutableRight )
   END_RUNG
   // the same network as SCL:
   "LTLP_HMIProInterfaceData".powerup30ExecutableLeft := "M_ONE" AND "DB2109_STATION_3_LIGHT_U01".SWITCH_OFF_GENERAL_CONDITIONS AND "DB2109_STATION_3_LIGHT_U01".SWITCH_OFF_INITIAL_CONDITIONS AND NOT "DB2109_STATION_3_LIGHT_U01".OUT_OF_SERVICE;
   "LTLP_HMIProInterfaceData".powerup30ExecutableRight := "M_ONE" AND "DB2109_STATION_3_LIGHT_U01".SWITCH_ON_GENERAL_CONDITIONS AND "DB2109_STATION_3_LIGHT_U01".SWITCH_ON_INITIAL_CONDITIONS AND NOT "DB2109_STATION_3_LIGHT_U01".IN_SERVICE;
END_REGION

REGION Network 19: HMI STATUS
   RUNG wire#powerrail
      Contact( "DB2109_STATION_3_LIGHT_U01".IN_SERVICE )
      wire#w1
      Not()
      Coil( "LTLP_HMIProInterfaceData".powerupCondOff30 )
   END_RUNG
   RUNG wire#w1
      Coil( "LTLP_HMIProInterfaceData".powerupCondOn30 )
   END_RUNG
   // the same network as SCL:
   "LTLP_HMIProInterfaceData".powerupCondOff30 := NOT "DB2109_STATION_3_LIGHT_U01".IN_SERVICE;
   "LTLP_HMIProInterfaceData".powerupCondOn30 := "DB2109_STATION_3_LIGHT_U01".IN_SERVICE;
END_REGION

REGION Network 20: MACHINE LIGHT ON OUTPUT
   RUNG wire#powerrail
      Contact( "DB2109_STATION_3_LIGHT_U01".SWITCH_ON )
      Coil( "STATION_3_LIGHT_U01_Q" )
   END_RUNG
   // the same network as SCL:
   "STATION_3_LIGHT_U01_Q" := "DB2109_STATION_3_LIGHT_U01".SWITCH_ON;
END_REGION
END_FUNCTION

FUNCTION "FC2110_STATION_3_LIGHT_U02" : Void   // FC2110, LAD
{ S7_Optimized_Access := 'FALSE' }
AUTHOR : ETXETAR
VERSION : 1.0
// stored: AutoNumber false, IsIECCheckEnabled false, SetENOAutomatically false, UDAEnableTagReadback false
   VAR_TEMP   // added for the SCL form of the ladder/FBD networks
      _w1 : Bool;
   END_VAR
BEGIN

REGION Network 1: INPUTS
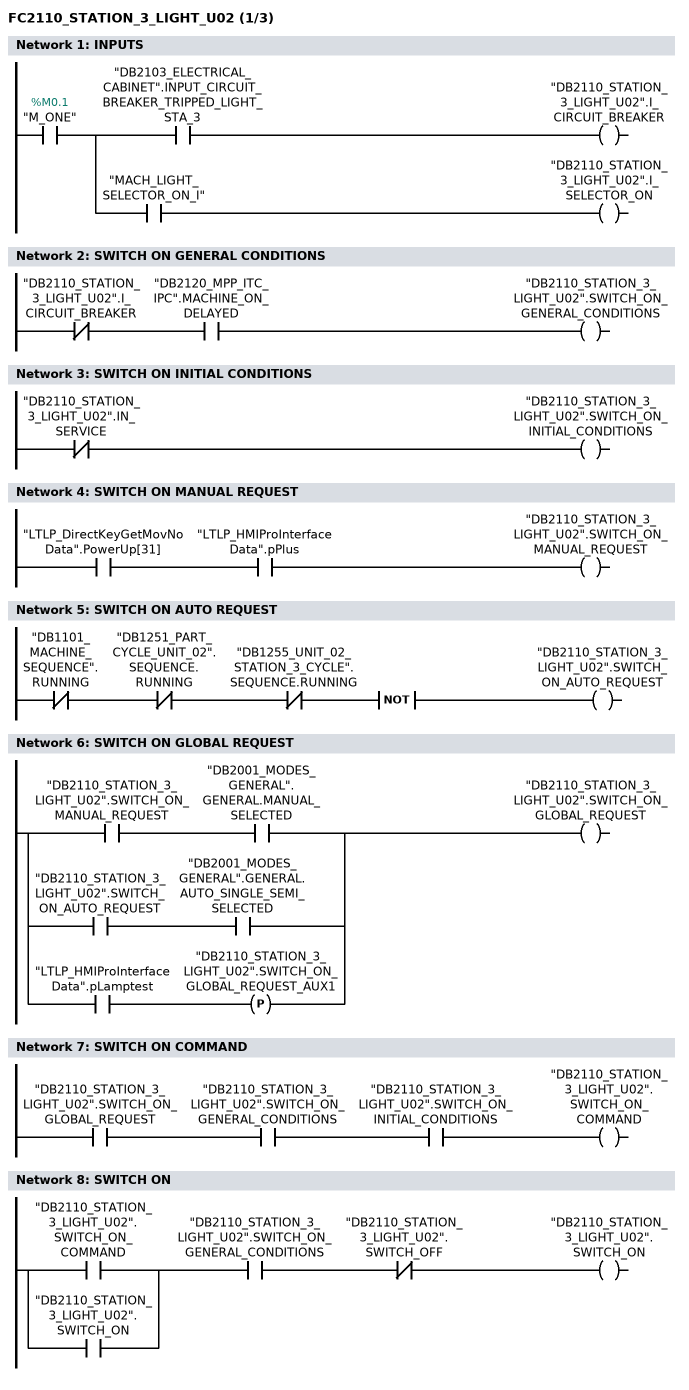
   RUNG wire#powerrail
      Contact( "M_ONE" )
      wire#w1
      Contact( "DB2103_ELECTRICAL_CABINET".INPUT_CIRCUIT_BREAKER_TRIPPED_LIGHT_STA_3 )
      Coil( "DB2110_STATION_3_LIGHT_U02".I_CIRCUIT_BREAKER )
   END_RUNG
   RUNG wire#w1
      Contact( "MACH_LIGHT_SELECTOR_ON_I" )
      Coil( "DB2110_STATION_3_LIGHT_U02".I_SELECTOR_ON )
   END_RUNG
   // the same network as SCL:
   "DB2110_STATION_3_LIGHT_U02".I_CIRCUIT_BREAKER := "M_ONE" AND "DB2103_ELECTRICAL_CABINET".INPUT_CIRCUIT_BREAKER_TRIPPED_LIGHT_STA_3;
   "DB2110_STATION_3_LIGHT_U02".I_SELECTOR_ON := "M_ONE" AND "MACH_LIGHT_SELECTOR_ON_I";
END_REGION

REGION Network 2: SWITCH ON GENERAL CONDITIONS
   RUNG wire#powerrail
      I_Contact( "DB2110_STATION_3_LIGHT_U02".I_CIRCUIT_BREAKER )
      Contact( "DB2120_MPP_ITC_IPC".MACHINE_ON_DELAYED )
      Coil( "DB2110_STATION_3_LIGHT_U02".SWITCH_ON_GENERAL_CONDITIONS )
   END_RUNG
   // the same network as SCL:
   "DB2110_STATION_3_LIGHT_U02".SWITCH_ON_GENERAL_CONDITIONS := NOT "DB2110_STATION_3_LIGHT_U02".I_CIRCUIT_BREAKER AND "DB2120_MPP_ITC_IPC".MACHINE_ON_DELAYED;
END_REGION

REGION Network 3: SWITCH ON INITIAL CONDITIONS
   RUNG wire#powerrail
      I_Contact( "DB2110_STATION_3_LIGHT_U02".IN_SERVICE )
      Coil( "DB2110_STATION_3_LIGHT_U02".SWITCH_ON_INITIAL_CONDITIONS )
   END_RUNG
   // the same network as SCL:
   "DB2110_STATION_3_LIGHT_U02".SWITCH_ON_INITIAL_CONDITIONS := NOT "DB2110_STATION_3_LIGHT_U02".IN_SERVICE;
END_REGION

REGION Network 4: SWITCH ON MANUAL REQUEST
   RUNG wire#powerrail
      Contact( "LTLP_DirectKeyGetMovNoData".PowerUp[31] )
      Contact( "LTLP_HMIProInterfaceData".pPlus )
      Coil( "DB2110_STATION_3_LIGHT_U02".SWITCH_ON_MANUAL_REQUEST )
   END_RUNG
   // the same network as SCL:
   "DB2110_STATION_3_LIGHT_U02".SWITCH_ON_MANUAL_REQUEST := "LTLP_DirectKeyGetMovNoData".PowerUp[31] AND "LTLP_HMIProInterfaceData".pPlus;
END_REGION

REGION Network 5: SWITCH ON AUTO REQUEST
   RUNG wire#powerrail
      I_Contact( "DB1101_MACHINE_SEQUENCE".RUNNING )
      I_Contact( "DB1251_PART_CYCLE_UNIT_02".SEQUENCE.RUNNING )
      I_Contact( "DB1255_UNIT_02_STATION_3_CYCLE".SEQUENCE.RUNNING )
      Not()
      Coil( "DB2110_STATION_3_LIGHT_U02".SWITCH_ON_AUTO_REQUEST )
   END_RUNG
   // the same network as SCL:
   "DB2110_STATION_3_LIGHT_U02".SWITCH_ON_AUTO_REQUEST := NOT (NOT "DB1101_MACHINE_SEQUENCE".RUNNING AND NOT "DB1251_PART_CYCLE_UNIT_02".SEQUENCE.RUNNING AND NOT "DB1255_UNIT_02_STATION_3_CYCLE".SEQUENCE.RUNNING);
END_REGION

REGION Network 6: SWITCH ON GLOBAL REQUEST
   RUNG wire#powerrail
      Contact( "DB2110_STATION_3_LIGHT_U02".SWITCH_ON_MANUAL_REQUEST )
      Contact( "DB2001_MODES_GENERAL".GENERAL.MANUAL_SELECTED )
      wire#w1
      Coil( "DB2110_STATION_3_LIGHT_U02".SWITCH_ON_GLOBAL_REQUEST )
   END_RUNG
   RUNG wire#powerrail
      Contact( "DB2110_STATION_3_LIGHT_U02".SWITCH_ON_AUTO_REQUEST )
      Contact( "DB2001_MODES_GENERAL".GENERAL.AUTO_SINGLE_SEMI_SELECTED )
   END_RUNG wire#w1
   RUNG wire#powerrail
      Contact( "LTLP_HMIProInterfaceData".pLamptest )
      P_Trig( "DB2110_STATION_3_LIGHT_U02".SWITCH_ON_GLOBAL_REQUEST_AUX1 )
   END_RUNG wire#w1
   // the same network as SCL:
   #_w1 := "LTLP_HMIProInterfaceData".pLamptest AND NOT "DB2110_STATION_3_LIGHT_U02".SWITCH_ON_GLOBAL_REQUEST_AUX1;   // rising edge
   "DB2110_STATION_3_LIGHT_U02".SWITCH_ON_GLOBAL_REQUEST_AUX1 := "LTLP_HMIProInterfaceData".pLamptest;
   "DB2110_STATION_3_LIGHT_U02".SWITCH_ON_GLOBAL_REQUEST := ("DB2110_STATION_3_LIGHT_U02".SWITCH_ON_MANUAL_REQUEST AND "DB2001_MODES_GENERAL".GENERAL.MANUAL_SELECTED) OR ("DB2110_STATION_3_LIGHT_U02".SWITCH_ON_AUTO_REQUEST AND "DB2001_MODES_GENERAL".GENERAL.AUTO_SINGLE_SEMI_SELECTED) OR #_w1;
END_REGION

REGION Network 7: SWITCH ON COMMAND
   RUNG wire#powerrail
      Contact( "DB2110_STATION_3_LIGHT_U02".SWITCH_ON_GLOBAL_REQUEST )
      Contact( "DB2110_STATION_3_LIGHT_U02".SWITCH_ON_GENERAL_CONDITIONS )
      Contact( "DB2110_STATION_3_LIGHT_U02".SWITCH_ON_INITIAL_CONDITIONS )
      Coil( "DB2110_STATION_3_LIGHT_U02".SWITCH_ON_COMMAND )
   END_RUNG
   // the same network as SCL:
   "DB2110_STATION_3_LIGHT_U02".SWITCH_ON_COMMAND := "DB2110_STATION_3_LIGHT_U02".SWITCH_ON_GLOBAL_REQUEST AND "DB2110_STATION_3_LIGHT_U02".SWITCH_ON_GENERAL_CONDITIONS AND "DB2110_STATION_3_LIGHT_U02".SWITCH_ON_INITIAL_CONDITIONS;
END_REGION

REGION Network 8: SWITCH ON
   RUNG wire#powerrail
      Contact( "DB2110_STATION_3_LIGHT_U02".SWITCH_ON_COMMAND )
      wire#w1
      Contact( "DB2110_STATION_3_LIGHT_U02".SWITCH_ON_GENERAL_CONDITIONS )
      I_Contact( "DB2110_STATION_3_LIGHT_U02".SWITCH_OFF )
      Coil( "DB2110_STATION_3_LIGHT_U02".SWITCH_ON )
   END_RUNG
   RUNG wire#powerrail
      Contact( "DB2110_STATION_3_LIGHT_U02".SWITCH_ON )
   END_RUNG wire#w1
   // the same network as SCL:
   "DB2110_STATION_3_LIGHT_U02".SWITCH_ON := ("DB2110_STATION_3_LIGHT_U02".SWITCH_ON_COMMAND OR "DB2110_STATION_3_LIGHT_U02".SWITCH_ON) AND "DB2110_STATION_3_LIGHT_U02".SWITCH_ON_GENERAL_CONDITIONS AND NOT "DB2110_STATION_3_LIGHT_U02".SWITCH_OFF;
END_REGION

REGION Network 9: IN SERVICE
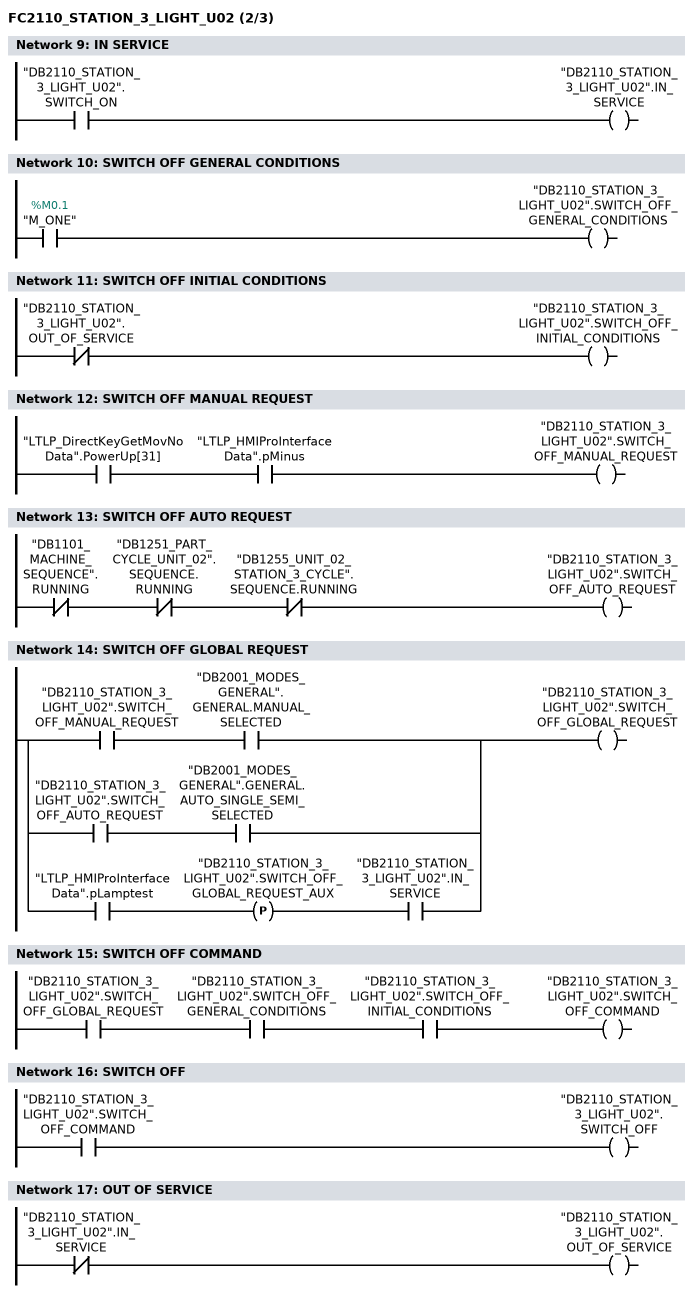
   RUNG wire#powerrail
      Contact( "DB2110_STATION_3_LIGHT_U02".SWITCH_ON )
      Coil( "DB2110_STATION_3_LIGHT_U02".IN_SERVICE )
   END_RUNG
   // the same network as SCL:
   "DB2110_STATION_3_LIGHT_U02".IN_SERVICE := "DB2110_STATION_3_LIGHT_U02".SWITCH_ON;
END_REGION

REGION Network 10: SWITCH OFF GENERAL CONDITIONS
   RUNG wire#powerrail
      Contact( "M_ONE" )
      Coil( "DB2110_STATION_3_LIGHT_U02".SWITCH_OFF_GENERAL_CONDITIONS )
   END_RUNG
   // the same network as SCL:
   "DB2110_STATION_3_LIGHT_U02".SWITCH_OFF_GENERAL_CONDITIONS := "M_ONE";
END_REGION

REGION Network 11: SWITCH OFF INITIAL CONDITIONS
   RUNG wire#powerrail
      I_Contact( "DB2110_STATION_3_LIGHT_U02".OUT_OF_SERVICE )
      Coil( "DB2110_STATION_3_LIGHT_U02".SWITCH_OFF_INITIAL_CONDITIONS )
   END_RUNG
   // the same network as SCL:
   "DB2110_STATION_3_LIGHT_U02".SWITCH_OFF_INITIAL_CONDITIONS := NOT "DB2110_STATION_3_LIGHT_U02".OUT_OF_SERVICE;
END_REGION

REGION Network 12: SWITCH OFF MANUAL REQUEST
   RUNG wire#powerrail
      Contact( "LTLP_DirectKeyGetMovNoData".PowerUp[31] )
      Contact( "LTLP_HMIProInterfaceData".pMinus )
      Coil( "DB2110_STATION_3_LIGHT_U02".SWITCH_OFF_MANUAL_REQUEST )
   END_RUNG
   // the same network as SCL:
   "DB2110_STATION_3_LIGHT_U02".SWITCH_OFF_MANUAL_REQUEST := "LTLP_DirectKeyGetMovNoData".PowerUp[31] AND "LTLP_HMIProInterfaceData".pMinus;
END_REGION

REGION Network 13: SWITCH OFF AUTO REQUEST
   RUNG wire#powerrail
      I_Contact( "DB1101_MACHINE_SEQUENCE".RUNNING )
      I_Contact( "DB1251_PART_CYCLE_UNIT_02".SEQUENCE.RUNNING )
      I_Contact( "DB1255_UNIT_02_STATION_3_CYCLE".SEQUENCE.RUNNING )
      Coil( "DB2110_STATION_3_LIGHT_U02".SWITCH_OFF_AUTO_REQUEST )
   END_RUNG
   // the same network as SCL:
   "DB2110_STATION_3_LIGHT_U02".SWITCH_OFF_AUTO_REQUEST := NOT "DB1101_MACHINE_SEQUENCE".RUNNING AND NOT "DB1251_PART_CYCLE_UNIT_02".SEQUENCE.RUNNING AND NOT "DB1255_UNIT_02_STATION_3_CYCLE".SEQUENCE.RUNNING;
END_REGION

REGION Network 14: SWITCH OFF GLOBAL REQUEST
   RUNG wire#powerrail
      Contact( "DB2110_STATION_3_LIGHT_U02".SWITCH_OFF_MANUAL_REQUEST )
      Contact( "DB2001_MODES_GENERAL".GENERAL.MANUAL_SELECTED )
      wire#w1
      Coil( "DB2110_STATION_3_LIGHT_U02".SWITCH_OFF_GLOBAL_REQUEST )
   END_RUNG
   RUNG wire#powerrail
      Contact( "DB2110_STATION_3_LIGHT_U02".SWITCH_OFF_AUTO_REQUEST )
      Contact( "DB2001_MODES_GENERAL".GENERAL.AUTO_SINGLE_SEMI_SELECTED )
   END_RUNG wire#w1
   RUNG wire#powerrail
      Contact( "LTLP_HMIProInterfaceData".pLamptest )
      P_Trig( "DB2110_STATION_3_LIGHT_U02".SWITCH_OFF_GLOBAL_REQUEST_AUX )
      Contact( "DB2110_STATION_3_LIGHT_U02".IN_SERVICE )
   END_RUNG wire#w1
   // the same network as SCL:
   #_w1 := "LTLP_HMIProInterfaceData".pLamptest AND NOT "DB2110_STATION_3_LIGHT_U02".SWITCH_OFF_GLOBAL_REQUEST_AUX;   // rising edge
   "DB2110_STATION_3_LIGHT_U02".SWITCH_OFF_GLOBAL_REQUEST_AUX := "LTLP_HMIProInterfaceData".pLamptest;
   "DB2110_STATION_3_LIGHT_U02".SWITCH_OFF_GLOBAL_REQUEST := ("DB2110_STATION_3_LIGHT_U02".SWITCH_OFF_MANUAL_REQUEST AND "DB2001_MODES_GENERAL".GENERAL.MANUAL_SELECTED) OR ("DB2110_STATION_3_LIGHT_U02".SWITCH_OFF_AUTO_REQUEST AND "DB2001_MODES_GENERAL".GENERAL.AUTO_SINGLE_SEMI_SELECTED) OR (#_w1 AND "DB2110_STATION_3_LIGHT_U02".IN_SERVICE);
END_REGION

REGION Network 15: SWITCH OFF COMMAND
   RUNG wire#powerrail
      Contact( "DB2110_STATION_3_LIGHT_U02".SWITCH_OFF_GLOBAL_REQUEST )
      Contact( "DB2110_STATION_3_LIGHT_U02".SWITCH_OFF_GENERAL_CONDITIONS )
      Contact( "DB2110_STATION_3_LIGHT_U02".SWITCH_OFF_INITIAL_CONDITIONS )
      Coil( "DB2110_STATION_3_LIGHT_U02".SWITCH_OFF_COMMAND )
   END_RUNG
   // the same network as SCL:
   "DB2110_STATION_3_LIGHT_U02".SWITCH_OFF_COMMAND := "DB2110_STATION_3_LIGHT_U02".SWITCH_OFF_GLOBAL_REQUEST AND "DB2110_STATION_3_LIGHT_U02".SWITCH_OFF_GENERAL_CONDITIONS AND "DB2110_STATION_3_LIGHT_U02".SWITCH_OFF_INITIAL_CONDITIONS;
END_REGION

REGION Network 16: SWITCH OFF
   RUNG wire#powerrail
      Contact( "DB2110_STATION_3_LIGHT_U02".SWITCH_OFF_COMMAND )
      Coil( "DB2110_STATION_3_LIGHT_U02".SWITCH_OFF )
   END_RUNG
   // the same network as SCL:
   "DB2110_STATION_3_LIGHT_U02".SWITCH_OFF := "DB2110_STATION_3_LIGHT_U02".SWITCH_OFF_COMMAND;
END_REGION

REGION Network 17: OUT OF SERVICE
   RUNG wire#powerrail
      I_Contact( "DB2110_STATION_3_LIGHT_U02".IN_SERVICE )
      Coil( "DB2110_STATION_3_LIGHT_U02".OUT_OF_SERVICE )
   END_RUNG
   // the same network as SCL:
   "DB2110_STATION_3_LIGHT_U02".OUT_OF_SERVICE := NOT "DB2110_STATION_3_LIGHT_U02".IN_SERVICE;
END_REGION

REGION Network 18: HMI STATUS
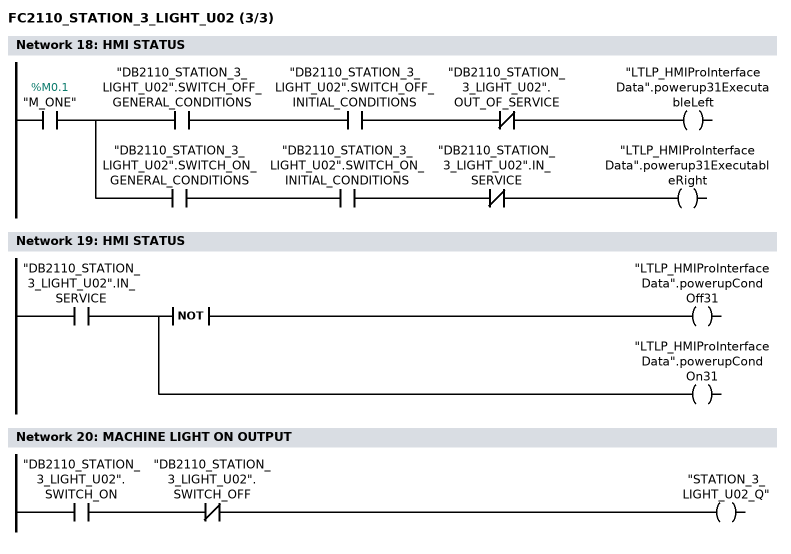
   RUNG wire#powerrail
      Contact( "M_ONE" )
      wire#w1
      Contact( "DB2110_STATION_3_LIGHT_U02".SWITCH_OFF_GENERAL_CONDITIONS )
      Contact( "DB2110_STATION_3_LIGHT_U02".SWITCH_OFF_INITIAL_CONDITIONS )
      I_Contact( "DB2110_STATION_3_LIGHT_U02".OUT_OF_SERVICE )
      Coil( "LTLP_HMIProInterfaceData".powerup31ExecutableLeft )
   END_RUNG
   RUNG wire#w1
      Contact( "DB2110_STATION_3_LIGHT_U02".SWITCH_ON_GENERAL_CONDITIONS )
      Contact( "DB2110_STATION_3_LIGHT_U02".SWITCH_ON_INITIAL_CONDITIONS )
      I_Contact( "DB2110_STATION_3_LIGHT_U02".IN_SERVICE )
      Coil( "LTLP_HMIProInterfaceData".powerup31ExecutableRight )
   END_RUNG
   // the same network as SCL:
   "LTLP_HMIProInterfaceData".powerup31ExecutableLeft := "M_ONE" AND "DB2110_STATION_3_LIGHT_U02".SWITCH_OFF_GENERAL_CONDITIONS AND "DB2110_STATION_3_LIGHT_U02".SWITCH_OFF_INITIAL_CONDITIONS AND NOT "DB2110_STATION_3_LIGHT_U02".OUT_OF_SERVICE;
   "LTLP_HMIProInterfaceData".powerup31ExecutableRight := "M_ONE" AND "DB2110_STATION_3_LIGHT_U02".SWITCH_ON_GENERAL_CONDITIONS AND "DB2110_STATION_3_LIGHT_U02".SWITCH_ON_INITIAL_CONDITIONS AND NOT "DB2110_STATION_3_LIGHT_U02".IN_SERVICE;
END_REGION

REGION Network 19: HMI STATUS
   RUNG wire#powerrail
      Contact( "DB2110_STATION_3_LIGHT_U02".IN_SERVICE )
      wire#w1
      Not()
      Coil( "LTLP_HMIProInterfaceData".powerupCondOff31 )
   END_RUNG
   RUNG wire#w1
      Coil( "LTLP_HMIProInterfaceData".powerupCondOn31 )
   END_RUNG
   // the same network as SCL:
   "LTLP_HMIProInterfaceData".powerupCondOff31 := NOT "DB2110_STATION_3_LIGHT_U02".IN_SERVICE;
   "LTLP_HMIProInterfaceData".powerupCondOn31 := "DB2110_STATION_3_LIGHT_U02".IN_SERVICE;
END_REGION

REGION Network 20: MACHINE LIGHT ON OUTPUT
   RUNG wire#powerrail
      Contact( "DB2110_STATION_3_LIGHT_U02".SWITCH_ON )
      I_Contact( "DB2110_STATION_3_LIGHT_U02".SWITCH_OFF )
      Coil( "STATION_3_LIGHT_U02_Q" )
   END_RUNG
   // the same network as SCL:
   "STATION_3_LIGHT_U02_Q" := "DB2110_STATION_3_LIGHT_U02".SWITCH_ON AND NOT "DB2110_STATION_3_LIGHT_U02".SWITCH_OFF;
END_REGION
END_FUNCTION

FUNCTION "FC2122_HT10" : Void   // FC2122, LAD
{ S7_Optimized_Access := 'TRUE' }
AUTHOR : ETXETAR
VERSION : 1.0
// stored: AutoNumber false, IsIECCheckEnabled false, SetENOAutomatically false, UDAEnableTagReadback false
   VAR CONSTANT
      FC_NUMBER : DInt := 2122;   // FC NUMEBR
   END_VAR
   VAR_TEMP   // added for the SCL form of the ladder/FBD networks
      _w1 : Bool;
      _w2 : Bool;
      _w3 : Bool;
   END_VAR
BEGIN

REGION Network 1: INPUT HT10 EMERGENCY STOP
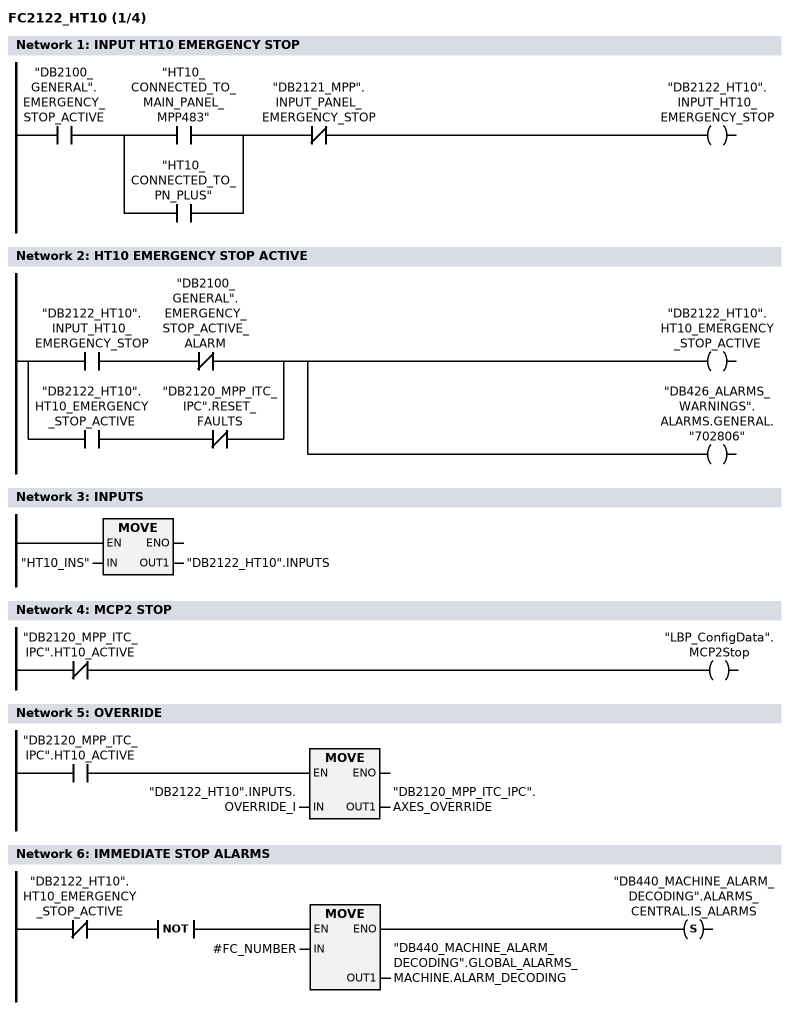
   RUNG wire#powerrail
      Contact( "DB2100_GENERAL".EMERGENCY_STOP_ACTIVE )
      wire#w1
      Contact( "HT10_CONNECTED_TO_MAIN_PANEL_MPP483" )
      wire#w2
      I_Contact( "DB2121_MPP".INPUT_PANEL_EMERGENCY_STOP )
      Coil( "DB2122_HT10".INPUT_HT10_EMERGENCY_STOP )
   END_RUNG
   RUNG wire#w1
      Contact( "HT10_CONNECTED_TO_PN_PLUS" )
   END_RUNG wire#w2
   // the same network as SCL:
   "DB2122_HT10".INPUT_HT10_EMERGENCY_STOP := "DB2100_GENERAL".EMERGENCY_STOP_ACTIVE AND ("HT10_CONNECTED_TO_MAIN_PANEL_MPP483" OR "HT10_CONNECTED_TO_PN_PLUS") AND NOT "DB2121_MPP".INPUT_PANEL_EMERGENCY_STOP;
END_REGION

REGION Network 2: HT10 EMERGENCY STOP ACTIVE
   RUNG wire#powerrail
      Contact( "DB2122_HT10".INPUT_HT10_EMERGENCY_STOP )
      I_Contact( "DB2100_GENERAL".EMERGENCY_STOP_ACTIVE_ALARM )
      wire#w1
      Coil( "DB2122_HT10".HT10_EMERGENCY_STOP_ACTIVE )
   END_RUNG
   RUNG wire#powerrail
      Contact( "DB2122_HT10".HT10_EMERGENCY_STOP_ACTIVE )
      I_Contact( "DB2120_MPP_ITC_IPC".RESET_FAULTS )
   END_RUNG wire#w1
   RUNG wire#w1
      Coil( "DB426_ALARMS_WARNINGS".ALARMS.GENERAL."702806" )
   END_RUNG
   // the same network as SCL:
   "DB2122_HT10".HT10_EMERGENCY_STOP_ACTIVE := ("DB2122_HT10".INPUT_HT10_EMERGENCY_STOP AND NOT "DB2100_GENERAL".EMERGENCY_STOP_ACTIVE_ALARM) OR ("DB2122_HT10".HT10_EMERGENCY_STOP_ACTIVE AND NOT "DB2120_MPP_ITC_IPC".RESET_FAULTS);
   "DB426_ALARMS_WARNINGS".ALARMS.GENERAL."702806" := "DB2122_HT10".HT10_EMERGENCY_STOP_ACTIVE;
END_REGION

REGION Network 3: INPUTS
   RUNG wire#powerrail
      Move(in := "HT10_INS", out1 => "DB2122_HT10".INPUTS)
   END_RUNG
   // the same network as SCL:
   "DB2122_HT10".INPUTS := "HT10_INS";
END_REGION

REGION Network 4: MCP2 STOP
   RUNG wire#powerrail
      I_Contact( "DB2120_MPP_ITC_IPC".HT10_ACTIVE )
      Coil( "LBP_ConfigData".MCP2Stop )
   END_RUNG
   // the same network as SCL:
   "LBP_ConfigData".MCP2Stop := NOT "DB2120_MPP_ITC_IPC".HT10_ACTIVE;
END_REGION

REGION Network 5: OVERRIDE
   RUNG wire#powerrail
      Contact( "DB2120_MPP_ITC_IPC".HT10_ACTIVE )
      Move(in := "DB2122_HT10".INPUTS.OVERRIDE_I, out1 => "DB2120_MPP_ITC_IPC".AXES_OVERRIDE)
   END_RUNG
   // the same network as SCL:
   IF "DB2120_MPP_ITC_IPC".HT10_ACTIVE THEN
       "DB2120_MPP_ITC_IPC".AXES_OVERRIDE := "DB2122_HT10".INPUTS.OVERRIDE_I;
   END_IF;
END_REGION

REGION Network 6: IMMEDIATE STOP ALARMS
   RUNG wire#powerrail
      I_Contact( "DB2122_HT10".HT10_EMERGENCY_STOP_ACTIVE )
      Not()
      { S7_GenerateENO := "TRUE" } Move(in := #FC_NUMBER, out1 => "DB440_MACHINE_ALARM_DECODING".GLOBAL_ALARMS_MACHINE.ALARM_DECODING)
      S_Coil( "DB440_MACHINE_ALARM_DECODING".ALARMS_CENTRAL.IS_ALARMS )
   END_RUNG
   // the same network as SCL:
   // ENO of a box is taken as its EN; it also drops when the box reports an error
   IF NOT (NOT "DB2122_HT10".HT10_EMERGENCY_STOP_ACTIVE) THEN
       "DB440_MACHINE_ALARM_DECODING".GLOBAL_ALARMS_MACHINE.ALARM_DECODING := #FC_NUMBER;
       "DB440_MACHINE_ALARM_DECODING".ALARMS_CENTRAL.IS_ALARMS := TRUE;
   END_IF;
END_REGION

